(* CODESYS project JCMC40A24BCtrl-V10.project

Project tree, tasks and I/O mapping:
  Device : JCMC 40A, JiaCheng Technology, version 3.5.4.0
    application Application
      libraries: Standard, * (System); SysFile, 3.5.5.0 (System); Util, 3.5.1.0 (System); JCMC_Ctrl, 3.5.5.160 (JiaCheng Technology); CmpJCPBasicLib, 2.1.1 (JiaCheng Technology)
      task MainTask (cyclic, interval t#10ms, priority 6) calls initCan, INIT_JCMC_Ctrl_EXT, INIT_JCMC_Ctrl, PLC_PRG
      task CAN (cyclic, interval t#10ms, priority 7) calls transmit2EngineECM
      program PLC_PRG [ST]
      global variables GVL
      global variables GVL_RETAIN
      program INIT_JCMC_Ctrl [FBD]
      data type RetainFileST
      program INIT_JCMC_Ctrl_EXT [FBD]
      data type Input24BST
      data type Input40AST
      data type Output40AST
      program handleInput24B [ST]
      program handleInput40A [ST]
      data type FaultST
      program faultHandle [ST]
      data type Output24BST
      data type SystemStatusST
      data type SystemConfigureST
      program functionTest [ST]
      program resetTestST [ST]
      data type DspSystemST
      data type DspTestST
      data type CtlTestST
      program chooseWorkMode [ST]
      program panelControl [ST]
      program workflowCore [ST]
      program workflowOther [ST]: ACT, Step0_ACT_active, Step1_ACT_active, Step2_ACT_active, Step3_ACT_active, Step4_ACT_active, Step5_ACT_active
      program engineControl [ST]
      data type TipsST
      program handleOutput40A [ST]
      program handleOutput24B [ST]
      program initCan [ST]
      program receiveFromHMI [ST]
      program receiveFromEngineECM [ST]
      program receiveFromECU [ST]
      program receiveFromVoiceAlarm [ST]
      program receiveFromSiliconePanel [ST]
      data type PanelST
      data type MultipacketParameter
      program transmit2HMI [ST]
      program transmit2SiliconePanel [ST]
      program transmit2EngineECM [ST]
      program parameterConfigure [ST]
      program tipsHandle [ST]
    IoDrvJCMC40A : IoDrvJCMC40A-24B, JiaCheng Technology, version 11.22.33.158
        unmapped channels: AIN_IX0, FIN_IX1, PWM_IX2, PWM_IX3, PWMi_IX4, IX5, %IW3 AI1, %IW4 AI2, AI3, AI4, AI5, AI6, AI7, AI8, FI1, FI2, FI3, FI4, FI5, FI6, FI7, FI8, PWM3i_Cur1, PWM3i_Cur2, PWM3i_Cur3, PWM3i_Cur4, PWM8i_Cur1, PWM8i_Cur2, PWM8i_Cur3, PWM8i_Cur4, PWM_QX0, PWM_QX1, PWMi_QX2, QX3, IX0, %IB73 PWM_IX1, PWM_IX2, IX3, AI1, AI2,
          AI3, AI4, FI1, FI2, FI3, FI4, PWM3i_Cur1, PWM3i_Cur2, PWM3i_Cur3, PWM3i_Cur4, PWM3i_Cur5, PWM3i_Cur6, PWM8i_Cur1, PWM8i_Cur2, PWM_QX0, PWMi_QX1, 5V_QX2
  text list GlobalTextList
  5ce3da45-db07-42e7-a21c-a00fff4ed8f6|C:\Users\guest1\Pictures\e84f1261c6d4c0a418f2bf4200fd030d.jpg
  5ce3da45-db07-42e7-a21c-a00fff4ed8f6|C:\Users\guest1\Pictures\aaa.bmp
  5ce3da45-db07-42e7-a21c-a00fff4ed8f6|C:\Users\guest1\Pictures\320x240.bmp
  5ce3da45-db07-42e7-a21c-a00fff4ed8f6|visu\navigationspanel320x160.jpg
  5ce3da45-db07-42e7-a21c-a00fff4ed8f6|visu\navigationspanel320x160.bmp
  image pool ImagePool
*)

// Device/Application/RetainFileST
TYPE RetainFileST :(*RetanFile区域总大小 3072byte,实际可用大小3071byte,另外1byte由RTS使用*)
STRUCT
	dataB:BYTE;
	dataW:WORD;
	dataD:DWORD;
	dataArray:ARRAY[0..3064] OF BYTE;
END_STRUCT
END_TYPE

// Device/Application/Input24BST
TYPE Input24BST :
STRUCT
	returnOilFilterBlockUp: BOOL; //回油过滤堵塞
	highPressureFilterBlockUp: BOOL;  //高压油滤堵塞
	reverseCar: BOOL; //倒车
	coolingTankWaterLevel: WORD; //冷却水箱液位
	waitingStartLamp: BOOL; //等待启动灯
	alarmLamp: BOOL; //警告故障灯
	stopEngineLamp: BOOL; //停机故障灯
	generatorWork: BOOL; //发电机发电
END_STRUCT
END_TYPE

// Device/Application/Input40AST
 TYPE Input40AST :
    STRUCT 
	   dumpsterPressure: WORD;  //垃圾箱负压
	   suctionBucketPressure: WORD; //吸桶负压
	   frontWaterTankPressure: WORD; //前水箱水压
	   backWaterTankPressure: WORD; //后水箱水压
	   diaphragmPumpPressure: BOOL; //隔膜泵压力正常
	   hydraulicOilLevel: BOOL; //液压油位低
	   frontWaterTankWaterLevel: WORD; //前水箱低水位
	   backWaterTankWaterLevel: WORD; //后清水箱水位
	   backup01: BOOL; //备用
	   bilgeTankWaterLevel: BOOL; //污水箱高水位
	   mainWateraValve: BOOL; //总水阀接近开关
	   cleanValve: BOOL; //吹净阀接近开关
	   backDoor: BOOL;  //后门接近开关
	   leftRod: BOOL; //左侧撑杆接近开关
	   rightRod: BOOL; //右侧撑杆接近开关
	   waterUnloadValve: BOOL; //水路卸荷阀接近开关
    END_STRUCT
  END_TYPE

// Device/Application/Output40AST
TYPE Output40AST :
STRUCT
	connectWaterValve:BOOL; //连通水阀关闭
	closeFrontTank:BOOL; //前水箱关闭
	cLoseBackTank:BOOL; //后水箱关闭
	engineStart:BOOL; //发动机启动
	diaphragmPumpStart:BOOL; //喷雾降尘泵启动
	backup01: BOOL; //备用
	engineStop:BOOL; //发动机停止
	sweeperLowSpeed:BOOL; //扫盘低速
	sweeperMiddleSpeed:BOOL; //扫盘中速
	oilUnloadValve:BOOL; //油路卸荷阀
	leftAllSweep:BOOL; //左/全扫
	rightSweep:BOOL; //右扫
	rightAllSweep:BOOL; //右/全扫
	tankDown:BOOL; //箱体降
	tankUp:BOOL; //箱体升
	suctionNozzleUp:BOOL; //吸嘴升
	leftBackSprinkle:BOOL; //左后洒
	rightBackSprinkle:BOOL; //右后洒
	tankDoorOpen:BOOL; //箱门开
	waterPumpConnect :BOOL; //水泵啮合
	leftFrontSprinkle:BOOL; //左前冲
	rightFrontSprinkle:BOOL; //右前冲
	suctionNozzleDown:BOOL; //吸嘴降
	tankDoorClose:BOOL; //箱门关
END_STRUCT
END_TYPE
(*
VAR_OUTPUT
	//wselfSprayRodOpen: BIT;
	//leftSweeperUp: BIT;
	//rightSprayRodSwingOut: BIT;
END_VAR
*)

// Device/Application/FaultST
TYPE FaultST :
STRUCT
	alarmLamp:BOOL; //发动机警告故障
    stopEngineLamp:BOOL;   //发动机停机故障
	coolingTankWaterLevelLow:BOOL;	//冷却水箱液位低
	waterUnloadValveNotClose:BOOL;	//水路卸荷阀未关闭
	waterUnloadValveNotOpen:BOOL;	//水路卸荷阀未打开
	bilgeTankFull:BOOL;	//污水满
	returnOilFilterBlockUp:BOOL;	//回油过滤堵塞
	hHighPressureFilterBlockUp:BOOL;	//高压油滤堵塞
	hydraulicOilLevelLow:BOOL;	//液压油位低
	frontTankWaterLevelLow:BOOL;	//前水箱缺水
	backTankWaterLevelLow:BOOL;	//后水箱缺水
	tankWaterLevelLow:BOOL;	//水箱缺水
	reverseCarStop:BOOL;	//倒车故障停机
	waterFullStop:BOOL;	//污水满故障停机
	highPressurePumpOverSpeedAlarm:BOOL;	//高压水泵超速报警
	highPressurePumpOverSpeedStop:BOOL;	//高压水泵超速停止
	diaphragmPumpPressure:BOOL;	//喷雾降尘泵故障
END_STRUCT
END_TYPE

// Device/Application/Output24BST
TYPE Output24BST :
STRUCT
	waterUnloadValveOpen :BOOL; //卸荷球阀打开
	auxiliaryValveOpen :BOOL; //辅助球阀喷水
	leftSprayRodOpen :BOOL; //左侧喷杆喷水
	selfSprayRodOpen  :BOOL; //自洁喷杆喷水
	rightSprayRodOpen  :BOOL; //右侧喷杆喷水
	centreSprayRodOpen  :BOOL; //中喷杆喷水
	engineDisconect  :BOOL;  //副发分离
	backupEngineStart  :BOOL; //备用动力
	rightSweeperDown :BOOL; //右扫降
	rightSweeperUp  :BOOL; //右扫升
	leftSweeperSwingOut :BOOL; //左扫摆出
	rightSweeperSwingOut :BOOL; //右扫摆出
	leftSprayRodSwingOut:BOOL; //左侧喷杆摆出
	rightSprayRodSwingOut :BOOL; //右侧喷杆摆出
	leftSweeperDown :BOOL; //左扫盘降
	leftSweeperUp :BOOL;  //左扫盘升
END_STRUCT
END_TYPE

// Device/Application/SystemStatusST
TYPE SystemStatusST :
STRUCT
     softVersion:WORD;//软件版本	

	systemWork:BOOL;//系统工作状态
	systemEndurance:WORD;//续航时间
	engineWork:BOOL;//发动机工作状态
	systemTest:BOOL; //系统测试状态
	backupMotorOpen:BOOL;//备用动力状态
	

	
	vehicleSpeed:WORD;//车速
	vehicleEngineSpeed:WORD;//底盘发动机转速
	distance:DWORD; //车辆行程里程
	
	keyRunPosition:BOOL; //钥匙运行档标志
	engineStart:BOOL; //发动机启动标志
	standardSpeed:BOOL;	//标准速度标志
    strongSpeed:BOOL;	//强力速度标志
    engineSetSpeed:WORD; //副发动机给定转速
	engineRealSpeed:WORD;//发动机实际转速
	engineDisconect:BOOL;//副发动机分离	
	engineCoolingTemperature:SINT;//副发水温
	engineOilPressure:BYTE;//副发油压
	engineWorkTime:DWORD;//发动机工作小时
	engineFaultSPN:DWORD; //副发当前故障SPN

	waterPumpConnect:BOOL; //高压水泵啮合标志
	
	allWashSweep:BOOL;	//全洗扫状态
	leftWashSweep:BOOL;	//左洗扫状态
	rightWashSweep:BOOL;	//右洗扫状态
	allSweep:BOOL;	//全扫路状态
	leftSweep:BOOL;	//左扫路状态
	rightSweep:BOOL;	//右扫路状态
	allWash:BOOL;	//全清洗状态
	leftWash:BOOL;	//左清洗状态
	rightWash:BOOL;	//右清洗状态
	stopWash:BOOL;	//停扫状态
	
	leftSweeperRotate:BOOL;//左扫旋转标志
	rightSweeperRotate:BOOL;//右扫旋转标志
	allSweeperRotate:BOOL;//全扫旋转标志
	leftSweeperSwingOut:BOOL;//左扫盘摆出标志
	leftSweeperDown:BOOL;//左扫盘下放标志
	rightSweeperSwingOut:BOOL;//右扫盘摆出标志
	rightSweeperDown:BOOL;//右扫盘下放标志
	suctionNozzleDown:BOOL;//吸嘴下降标志
	leftSweeperUp:BOOL;//左扫盘上升标志
	rightSweeperUp:BOOL;//右扫盘上升标志
	suctionNozzleUp:BOOL;//吸嘴上升标志
	
	auxiliaryValveOpen1:BOOL; //辅助球阀喷水标志1
	auxiliaryValveOpen2:BOOL; //辅助球阀喷水标志2
	leftSprayRodOpen1:BOOL; //左侧喷杆喷水标志1
	leftSprayRodOpen2:BOOL; //左侧喷杆喷水标志2
	selfSprayRodOpen1:BOOL; //自洁喷杆喷水标志1
	selfSprayRodOpen2:BOOL; //自洁喷杆喷水标志2
	rightSprayRodOpen1 :BOOL; //右侧喷杆喷水标志1
	rightSprayRodOpen2 :BOOL; //右侧喷杆喷水标志2
	centreSprayRodOpen1 :BOOL; //中喷杆喷水标志1
	centreSprayRodOpen2 :BOOL; //中喷杆喷水标志2
	
	leftSprayRodSwingOut :BOOL; //左侧喷杆摆出标志
	rightSprayRodSwingOut :BOOL; //右侧喷杆摆出标志
    //diaphragmPumpStart:BOOL;  //喷雾降尘泵启动标志
	
	leftFlushOpen:BOOL;	//左角冲打开标志
    rightFlushOpen:BOOL;	//右角冲打开标志
    backSprayOpen:BOOL;	//后喷雾打开标志
    sprayGun:BOOL;	//手持喷枪打开标志
	selfClean:BOOL;	//	自洁打开标志
	
    leftFrontSprinkle:BOOL;	//	左前冲打开标志
	rightFrontSprinkle:BOOL;	//	右前冲打开标志
	leftBackSprinkle:BOOL;	//	左后洒打开标志
	rightBackSprinkle:BOOL;	//	右后洒打开标志
	
	tankDoorClose:BOOL;	//垃圾箱门关标志
	tankDoorOpen:BOOL;	//垃圾箱门开标志
	tankDown:BOOL;	//垃圾箱体降标志
	tankUp:BOOL;	//垃圾箱体升标志
	sweeperSpeedLow:BOOL;	//扫盘低速标志
	sweeperSpeedMiddle:BOOL;	//扫盘中速标志
	sweeperSpeedHigh:BOOL;	//扫盘高速标志
	
	manualDrainOff:BOOL; 	//手动排水标志
	autoDrainOff:BOOL; //自动排水标志
	drainOffStart:BOOL;	//排水启动标志,目前该状态属于未启用状态
	replaceSweeper:BOOL;	//更换扫刷标志
	workLamp:BOOL;//工作灯标志
	diaphragmPump:BOOL;//隔膜泵标志
	
	AIModel:BOOL;	//智能模式标志
	CleanRoad:BOOL;	//清洁路面标志
	NormalRoad:BOOL;	//一般路面标志
	DirtyRoad:BOOL;	//污染路面标志
	
	
END_STRUCT
END_TYPE

// Device/Application/SystemConfigureST
TYPE SystemConfigureST :
STRUCT
	
	configFlag:BOOL;            //配置初始化标志
	//dspDiaphragmPump:BOOL;	//喷雾降尘泵_配置_屏输入
	dspLowPressureSystem:BOOL;	//低压水路系统_配置_屏输入
   	dspEngineStandardSpeed:WORD;	//标准速度_配置_屏输入
    dspEngineStrongSpeed:WORD;	//强力速度_配置_屏输入
    dspIncreaseStep:WORD;	//加减转速_配置_屏输入
	dspWaterPumpOverSpeedAlarm:WORD;	//高压水泵超速警报_配置_屏输入
	dspWaterPumpOverSpeedStop:WORD; 	//高压水泵超速停机_配置_屏输入
	dspEngineIdlingSpeed:WORD;	//发动机怠速_配置_屏输入
    dspSweeperSpeed:WORD; //扫盘转速_配置_屏输入
    dspAIModel:BOOL;	//智能模式_配置_屏输入
    dspRoadCondition:WORD;	//路面情况_配置_屏输入
    dspEngineMaxSpeed:WORD;	//发动机最高速_配置_屏输入
	dspWaterPumpConnect:BOOL; //水泵离合器_配置_屏输入

END_STRUCT
END_TYPE

// Device/Application/DspSystemST
TYPE DspSystemST :
STRUCT
	dspAllWashSweep:BOOL;	//全洗扫_屏输入
	dspLeftWashSweep:BOOL;	//左洗扫_屏输入
	dspRightWashSweep:BOOL;	//右洗扫_屏输入
	dspAllSweep:BOOL;	//全扫路_屏输入
	dspLeftSweep:BOOL;	//左扫路_屏输入
	dspRightSweep:BOOL;	//右扫路_屏输入
	dspAllWash:BOOL;	//全清洗_屏输入
	dspLeftWash:BOOL;	//左清洗_屏输入
	dspRightWash:BOOL;	//右清洗_屏输入
	dspStopWash:BOOL;	//停扫_屏输入
	
	dspEngineStart:BOOL;	//发动机启动_屏输入
	dspEngineStop:BOOL;	//发动机停止/运行_屏输入
	
	dspSpeedUp:BOOL;	//转速增加_屏输入
	dspSpeedDown:BOOL;	//转速降低_屏输入
	dspStandardSpeed:BOOL;	//标准速度_屏输入
	dspStrongSpeed:BOOL;	//强力速度_屏输入
	dspAIModel:BOOL;	//智能模式_屏输入
	dspCleanRoad:BOOL;	//清洁路面_屏输入
	dspNormalRoad:BOOL;	//一般路面_屏输入
	dspDirtyRoad:BOOL;	//污染路面_屏输入
	
	dspTankDoorClose:BOOL;	//垃圾箱门关_屏输入
	dspTankDoorOpen:BOOL;	//垃圾箱门开_屏输入
	dspTankDown:BOOL;	//垃圾箱体降_屏输入
	dspTankUp:BOOL;	//垃圾箱体升_屏输入
	dspSweeperSpeedLow:BOOL;	//扫盘低速_屏输入
	dspSweeperSpeedMiddle:BOOL;	//扫盘中速_屏输入
	dspSweeperSpeedHigh:BOOL;	//扫盘高速_屏输入
	
	dspWaterPumpDisconnect:BOOL;//水泵离合器_屏输入
	dspLeftFlush:BOOL;	//左角冲_屏输入
	dspRightFlush:BOOL;	//右角冲_屏输入
	dspBackSpray:BOOL;	//后喷雾_屏输入
	dspSprayGun:BOOL;	//手持喷枪_屏输入
	dspSelfClean:BOOL;	//自洁_屏输入
	
	dspLeftFrontSprinkle:BOOL;	//左前冲_屏输入
	dspRightFrontSprinkle:BOOL;	//右前冲_屏输入
	dspLeftBackSprinkle:BOOL;	//左后洒_屏输入
	dspRightBackSprinkle:BOOL;	//右后洒_屏输入
	
	dspManualDrainOff:BOOL; 	//手动排水_屏输入
	dspAutoDrainOff:BOOL; //自动排水_屏输入
	dspDrainOffStart:BOOL;	//排水启动_屏输入,目前该按钮属于未启动状态
	dspLeftSprayRodDrainOff:BOOL;	//左喷杆排水_屏输入
	dspRightSprayRodDrainOff:BOOL;	//右喷杆排水_屏输入
	dspAuxiliarySystemDrainOff:BOOL;	//辅助排水_屏输入
	dspSelfCleanDrainOff:BOOL;	//自洁排水_屏输入
	dspCentreSprayRodDrainOff:BOOL;	//中喷杆排水_屏输入
	dspReplaceSweeper:BOOL;	//更换扫刷_屏输入
	dspWorkLamp:BOOL;//工作灯_屏输入
	dspDiaphragmPump:BOOL;//隔膜泵_屏输入
	
	dspTestStart:BOOL;	//功能测试_屏输入
END_STRUCT
END_TYPE

// Device/Application/DspTestST
TYPE DspTestST :
STRUCT
	dspEngineDisconnectTest:BOOL;	//副发分离_测试_屏输入
	dspConnectWaterValveTest:BOOL;	//连通水阀_测试_屏输入
	dspCloseFrontTankTest:BOOL;	//前水箱水阀_测试_屏输入
	dspCLoseBackTankTest:BOOL;	//后水箱水阀_测试_屏输入
	dspSweeperSpeedLowTest:BOOL;	//扫盘低速_测试_屏输入
	dspSweeperSpeedMiddleTest:BOOL;	//扫盘中速_测试_屏输入
	dspLeftSweeperRotateTest:BOOL;	//左扫旋转_测试_屏输入
	dspRightSweeperRotateTest:BOOL;	//右扫旋转_测试_屏输入
	dspAllSweeperRotateTest:BOOL;	//全扫旋转_测试_屏输入
	dspTankDownTest:BOOL;	//箱体降_测试_屏输入
	dspTankUpTest:BOOL;	//箱体升_测试_屏输入
	dspSuctionNozzleDownTest:BOOL;	//吸嘴降_测试_屏输入
	dspSuctionNozzleUpTest:BOOL;	//吸嘴升_测试_屏输入
	dspTankDoorOpenTest:BOOL; //箱门开_测试_屏输入
	dspTankDoorCloseTest:BOOL;	//箱门关_测试_屏输入
	dspLeftSweeperDownTest:BOOL;	//左扫盘下放_测试_屏输入
	dspLeftSweeperUpTest:BOOL;	//左扫盘回收_测试_屏输入
	dspRightSweeperDownTest:BOOL;	//右扫盘下放_测试_屏输入
	dspRightSweeperUpTest:BOOL;	//右扫盘回收_测试_屏输入
	dspLeftSweeperSwingOutTest:BOOL;	//左扫盘摆出_测试_屏输入
	dspRightSweeperSwingOutTest:BOOL;	//右扫盘摆出_测试_屏输入
	dspLeftSprayRodSwingOutTest:BOOL;	//左喷杆摆出_测试_屏输入
	dspRightSprayRodSwingOutTest:BOOL;	//右喷杆摆出_测试_屏输入
	dspLeftSprayRodOpenTest:BOOL;	//左喷杆喷水_测试_屏输入
	dspRightSprayRodOpenTest:BOOL;	//右喷杆喷水_测试_屏输入
	dspCentreSprayRodOpenTest:BOOL;	//中喷杆喷水_测试_屏输入
	dspAuxiliaryValueTest:BOOL;	//辅助球阀打开_测试_屏输入
	dspSelfCleanTest:BOOL;	//自洁打开_测试_屏输入
	dspWaterPumpConnectTest:BOOL;//高压水泵啮合_测试_屏输入
	dspDiaphragmPumpStartTest:BOOL;	//喷雾降尘泵_测试_屏输入
    dspLeftFrontSprinkleTest:BOOL;	//	左前冲_测试_屏输入
	dspRightFrontSprinkleTest:BOOL;	//	右前冲_测试_屏输入
	dspLeftBackSprinkleTest:BOOL;	//	左后洒_测试_屏输入
	dspRightBackSprinkleTest:BOOL;	//	右后洒_测试_屏输入

END_STRUCT
END_TYPE

// Device/Application/CtlTestST
TYPE CtlTestST :
STRUCT
	ctlEngineDisconnectTest:BOOL;	//副发分离_测试_控制器
    ctlConnectWaterValveTest:BOOL;	//连通水阀_测试_控制器
    ctlCloseFrontTankTest:BOOL;	//前水箱水阀_测试_控制器
    ctlCLoseBackTankTest:BOOL;	//后水箱水阀_测试_控制器
    ctlSweeperSpeedLowTest:BOOL;	//扫盘低速_测试_控制器
	ctlSweeperSpeedMiddleTest:BOOL;	//扫盘中速_测试_控制器
	ctlLeftSweeperRotateTest:BOOL;	//左扫旋转_测试_控制器
	ctlRightSweeperRotateTest:BOOL;	//右扫旋转_测试_控制器
	ctlAllSweeperRotateTest:BOOL;	//全扫旋转_测试_控制器
	ctlTankDownTest:BOOL;	//箱体降_测试_控制器
	ctlTankUpTest:BOOL;	//箱体升_测试_控制器
	ctlSuctionNozzleDownTest:BOOL;	//吸嘴降_测试_控制器
	ctlSuctionNozzleUpTest:BOOL;	//吸嘴升_测试_控制器
	ctlTankDoorOpenTest:BOOL;	//箱门开_测试_控制器
	ctlTankDoorCloseTest:BOOL;	//箱门关_测试_控制器
	ctlLeftSweeperDownTest:BOOL;	//左扫盘下放_测试_控制器
	ctlLeftSweeperUpTest:BOOL;	//左扫盘回收_测试_控制器
	ctlRightSweeperDownTest:BOOL;	//右扫盘下放_测试_控制器
	ctlRightSweeperUpTest:BOOL;	//右扫盘回收_测试_控制器
	ctlLeftSweeperSwingOutTest:BOOL;	//左扫盘摆出_测试_控制器
	ctlRightSweeperSwingOutTest:BOOL;	//右扫盘摆出_测试_控制器
	ctlLeftSprayRodSwingOutTest:BOOL;	//左喷杆摆出_测试_控制器
	ctlRightSprayRodSwingOutTest:BOOL;	//右喷杆摆出_测试_控制器
	ctlLeftSprayRodOpenTest:BOOL;	//左喷杆喷水_测试_控制器
	ctlRightSprayRodOpenTest:BOOL;	//右喷杆喷水_测试_控制器
	ctlCentreSprayRodOpenTest:BOOL;	//中喷杆喷水_测试_控制器
	ctlAuxiliaryValueTest:BOOL;	//辅助球阀打开_测试_控制器
	ctlSelfCleanTest:BOOL;	//自洁打开_测试_控制器
	ctlWaterPumpConnectTest:BOOL;	//高压水泵啮合_测试_控制器
	ctlDiaphragmPumpStartTest:BOOL;	//喷雾降尘泵_测试_控制器
	ctlLeftFrontSprinkleTest:BOOL;	//	左前冲_测试_控制器
	ctlRightFrontSprinkleTest:BOOL;	//	右前冲_测试_控制器
	ctlLeftBackSprinkleTest:BOOL;	//	左后洒_测试_控制器
	ctlRightBackSprinkleTest:BOOL;	//	右后洒_测试_控制器
END_STRUCT
END_TYPE

// Device/Application/TipsST
TYPE TipsST :
STRUCT
	closeTest:BOOL;	//请关闭测试
    reverseCar:BOOL;	//正在倒车中
	startEngineFirst:BOOL;	//请先打开发动机
	backupMotorOpen:BOOL;	//备用动力打开
	testOpen:BOOL;	//测试打开
	highPressurePumpDisconnect:BOOL;	//高压水泵未啮合
	tankDoorNotOpen:BOOL; //箱门未打开
	leftRodUp:BOOL;	//左支撑杆未放下
	rightRodUp:BOOL;	//右支撑杆未放下
	mainWateraValveNotOpen:BOOL;	//总水阀未打开
	cleanValveNotClose:BOOL;	//吹净球阀未关闭
    stopEngineFirst:BOOL; //请先关闭发动机
	
	
	//临时变量
	highPressurePumpDisconnect1:BOOL;	//左右全洗扫、清洗按钮，高压水泵未啮合
	highPressurePumpDisconnect2:BOOL;	//硅胶面板喷枪、自洁按钮，高压水泵未啮合
	highPressurePumpDisconnect3:BOOL;	//触摸屏喷枪、自洁、左前冲、右前冲、后喷雾按钮，高压水泵未啮合
	mainWateraValveNotOpen1:BOOL;	//左右全洗扫、清洗按钮，总水阀未打开
	mainWateraValveNotOpen2:BOOL;	//硅胶面板喷枪、自洁按钮，总水阀未打开
	mainWateraValveNotOpen3:BOOL;	//触摸屏喷枪、自洁、左前冲、右前冲、后喷雾按钮，总水阀未打开
	mainWateraValveNotOpen4:BOOL;	//离合器按钮，总水阀未打开
	cleanValveNotClose1:BOOL;	//左右全洗扫、清洗按钮，吹净球阀未关闭
	cleanValveNotClose2:BOOL;	//硅胶面板喷枪、自洁按钮，吹净球阀未关闭
	cleanValveNotClose3:BOOL;	//触摸屏喷枪、自洁、左前冲、右前冲、后喷雾按钮，吹净球阀未关闭
	cleanValveNotClose4:BOOL;	//离合器按钮，吹净球阀未关闭
END_STRUCT
END_TYPE

// Device/Application/PanelST
TYPE PanelST :
STRUCT
	tankDoorClose:BOOL;	//垃圾箱门关_硅胶面板输入
	tankDoorOpen:BOOL;	//垃圾箱门开_硅胶面板输入
	tankDown:BOOL;	//垃圾箱体降_硅胶面板输入
	tankUp:BOOL;	//垃圾箱体升_硅胶面板输入
	leftSweeperOutAndDown:BOOL;	//左扫盘摆出下降_硅胶面板输入
	leftSweeperUpAndIn:BOOL;	//左扫盘上升回收_硅胶面板输入
	rightSweeperOutAndDown:BOOL;	//右扫盘下放_硅胶面板输入
	rightSweeperUpAndIn:BOOL;	//右扫盘回收_硅胶面板输入
	suctionNozzleDown:BOOL;	//吸嘴降_测试_硅胶面板输入
	suctionNozzleUp:BOOL;	//吸嘴升_硅胶面板输入
	selfClean:BOOL;	//自洁打开_硅胶面板输入
	sprayGun:BOOL;	//手持喷枪_硅胶面板输入
	sprayRodOutOrIn:BOOL;  //喷杆伸缩_硅胶面板输入
	backupMotor:BOOL; //备用动力_硅胶面板输入
	workLamp:BOOL; //工作灯_硅胶面板输入
	backlight:BOOL; //背光灯_硅胶面板输入
	
	tankDoorCloseFlag:BOOL;	//垃圾箱门关_硅胶面板_返回标志
	tankDoorOpenFlag:BOOL;	//垃圾箱门开_硅胶面板_返回标志
	tankDownFlag:BOOL;	//垃圾箱体降_硅胶面板_返回标志
	tankUpFlag:BOOL;	//垃圾箱体升_硅胶面板_返回标志
	leftSweeperOutAndDownFlag:BOOL;	//左扫盘下放_硅胶面板_返回标志
	leftSweeperUpAndInFlag:BOOL;	//左扫盘回收_硅胶面板_返回标志
	rightSweeperOutAndDownFlag:BOOL;	//右扫盘下放_硅胶面板_返回标志
	rightSweeperUpAndInFlag:BOOL;	//右扫盘回收_硅胶面板_返回标志
	suctionNozzleDownFlag:BOOL;	//吸嘴降_测试_硅胶面板_返回标志
	suctionNozzleUpFlag:BOOL;	//吸嘴升_硅胶面板_返回标志
	selfCleanFlag:BOOL;	//自洁打开_硅胶面板_返回标志
	sprayGunFlag:BOOL;	//手持喷枪_硅胶面板_返回标志
	sprayRodOutOrInFlag:BOOL;  //喷杆伸缩_硅胶面板_返回标志
	backupMotorFlag:BOOL; //备用动力_硅胶面板_返回标志
	workLampFlag:BOOL; //工作灯_硅胶面板_返回标志
	backlightFlag:BOOL; //背光灯_硅胶面板_返回标志
END_STRUCT
END_TYPE

// Device/Application/MultipacketParameter
TYPE MultipacketParameter :
STRUCT
	packageTotalNum:WORD;//数据包数量，2-255
	byteTotalNum:WORD; //字节数，9-1785
	PGN:DWORD; //参数群编号
	Data: ARRAY[0..79] OF  BYTE; //数据,当packageNum>10，丢弃数据
END_STRUCT
END_TYPE

// Device/Application/GVL
VAR_GLOBAL		

	isOK: BOOL;	
// 40A板卡输入输出端口
    diDumpsterPressure AT %IW3 :WORD;  //垃圾箱负压
	diSuctionBucketPressure AT %IW4 :WORD; //吸桶负压
	diFrontWaterTankPressure AT %IW5 :WORD; //前水箱水压
	diBackWaterTankPressure AT %IW6 :WORD; //后水箱水压
	diDiaphragmPumpPressure AT %IX0.4 :BOOL; //隔膜泵压力正常
	diHydraulicOilLevel AT %IX0.5 :BOOL; //液压油位低
	diFrontWaterTankWaterLevel AT %IW9 :WORD; //前水箱低水位
	diBackWaterTankWaterLevel AT %IW10 :WORD; //后清水箱水位
	diBackup01 AT %IX1.0 :BOOL; //备用
	diBilgeTankWaterLevel AT %IX1.1 :BOOL; //污水箱高水位
	diMainWateraValve AT %IX1.2 :BOOL; //总水阀接近开关
	diCleanValve AT %IX1.3 :BOOL; //吹净阀接近开关
	diBackDoor AT %IX1.4 :BOOL;  //后门接近开关
	diLeftRod AT %IX1.5 :BOOL; //左侧撑杆接近开关
	diRightRod AT %IX1.6 :BOOL; //右侧撑杆接近开关
	diWaterUnloadValve AT %IX1.7 :BOOL; //水路卸荷阀接近开关
	doConnectWaterValve AT %QX0.0 :BOOL; //连通水阀关闭
	doCloseFrontTank AT %QX0.1 :BOOL; //前水箱关闭
	doCLoseBackTank AT %QX0.2 :BOOL; //后水箱关闭
	doEngineStart AT %QX0.3 :BOOL; //发动机启动
	doDiaphragmPumpStart AT %QX0.4 :BOOL; //隔膜泵启动
	doBackup01 AT %QX0.5 : BOOL; //备用
	doEngineStop AT %QX0.6 :BOOL; //发动机停止
	doSweeperLowSpeed AT %QX0.7 :BOOL; //扫盘低速
	doSweeperMiddleSpeed AT %QX1.0 :BOOL; //扫盘中速
	doOilUnloadValve AT %QX1.1 :BOOL; //油路卸荷阀
	doLeftAllSweep AT %QX1.2 :BOOL; //左/全扫
	doRightSweep AT %QX1.3 :BOOL; //右扫
	doRightAllSweep AT %QX1.4 :BOOL; //右/全扫
	doTankDown AT %QX1.5 :BOOL; //箱体降
	doTankUp AT %QX1.6 :BOOL; //箱体升
	doSuctionNozzleUp AT %QX1.7 :BOOL; //吸嘴升
	doLeftBackSprinkle AT %QX2.0 :BOOL; //左后洒
	doRightBackSprinkle AT %QX2.1 :BOOL; //右后洒
	doTankDoorOpen AT %QX2.2 :BOOL; //箱门开
	doWaterPumpConnect AT %QX2.3 :BOOL; //水泵啮合
	doLeftFrontSprinkle AT %QX2.4 :BOOL; //左前冲
	doRightFrontSprinkle AT %QX2.5 :BOOL; //右前冲
	doSuctionNozzleDown AT %QX2.6 :BOOL; //吸嘴降
	doTankDoorClose AT %QX2.7 :BOOL; //箱门关
	
//24B板块输入输出端口	
    diReturnOilFilterBlockUp AT %IX72.0 :BOOL; //回油过滤堵塞
	diHighPressureFilterBlockUp AT %IX72.1 :BOOL;  //高压油滤堵塞
	diReverseCar AT %IX72.2 :BOOL; //倒车
	diCoolingTankWaterLevel AT %ID22 :WORD; //冷却水箱液位
	diWaitingStartLamp AT %IX72.4 :BOOL; //等待启动灯
	diAlarmLamp AT %IX72.5 :BOOL; //警告故障灯
	diStopEngineLamp AT %IX72.6 :BOOL; //停机故障灯
	diGeneratorWork  AT %IX7.7 :BOOL; //发电机发电
	doWaterUnloadValveOpen AT %QX4.0 :BOOL; //卸荷球阀打开
	doAuxiliaryValveOpen AT %QX4.1 :BOOL; //辅助球阀喷水
	doLeftSprayRodOpen AT %QX4.2 :BOOL; //左侧喷杆喷水
	doSelfSprayRodOpen AT %QX4.3 :BOOL; //自洁喷杆喷水
	doRightSprayRodOpen AT %QX4.4 :BOOL; //右侧喷杆喷水
	doCentreSprayRodOpen AT %QX4.5 :BOOL; //中喷杆喷水
	doEngineDisconect AT %QX4.6 :BOOL;  //副发分离
	doBackupEngineStart AT %QX4.7 :BOOL; //备用动力
	doRightSweeperDown AT %QX5.0 :BOOL; //右扫降
	doRightSweeperUp AT %QX5.1 :BOOL; //右扫升
	doLeftSweeperSwingOut AT %QX5.2 :BOOL; //左扫摆出
	doRightSweeperSwingOut AT %QX5.3 :BOOL; //右扫摆出
	doLeftSprayRodSwingOut AT %QX5.4 :BOOL; //左侧喷杆摆出
	doRightSprayRodSwingOut AT %QX5.5 :BOOL; //右侧喷杆摆出
	doLeftSweeperDown AT %QX5.6 :BOOL; //左扫盘降
	doLeftSweeperUp AT %QX5.7 :BOOL;  //左扫盘升
 
    input40A: Input40AST;//处理后的40A板卡的输入信号  
    input24B: Input24BST;//处理后的40A板卡的输入信号
    output40A: Output40AST; //40A板卡输出信号
    output24B: Output24BST; //24B板卡输出信号
    dspSystemInput:DspSystemST;//车载控制屏系统输入
    dspTestInput:DspTestST; //车载控制屏测试输入
    systemStatus: SystemStatusST;//系统工作状态
    ctlTestFlag:CtlTestST; //控制器测试状态
    faultST: FaultST;  //系统故障
    tipsST:TipsST;     //系统提示
	panelInput:PanelST; //硅胶面板控制信号
END_VAR

// Device/Application/GVL_RETAIN
VAR_GLOBAL RETAIN
	bufRETAIN: DWORD:= 0;
//	bufRETAIN2: BYTE:= 0;
	pbufRetain: POINTER TO DWORD:=ADR(bufretain);
	xx: POINTER TO POINTER TO DWORD:=ADR(pbufRetain);
    systemConfig:SystemConfigureST; //系统配置

END_VAR

// Device/Application/initCan
PROGRAM initCan
VAR
	initCAN: JCMC_Ctrl.CAN;
	initCAN_EXT: JCMC_Ctrl.CAN_EXT;
END_VAR

IF JCMC_Ctrl.INIT THEN   //可以不用，调试再试验
	initCAN(CHANNEL:=1,ENABLE:=TRUE,START:=TRUE,EXTENDED_MODE:=TRUE,BAUDRATE:=250);//40A,CAN1初始化，波特率250KB，扩展帧
	initCAN(CHANNEL:=2,ENABLE:=TRUE,START:=TRUE,EXTENDED_MODE:=TRUE,BAUDRATE:=250);//40A,CAN2初始化，波特率250KB，扩展帧

	initCAN_EXT(CHANNEL:=1,ENABLE:=TRUE,START:=TRUE,EXTENDED_MODE:=TRUE,BAUDRATE:=250);//24B,CAN1初始化，波特率250KB，扩展帧,发送频率不要低于20ms
	initCAN_EXT(CHANNEL:=2,ENABLE:=TRUE,START:=TRUE,EXTENDED_MODE:=TRUE,BAUDRATE:=250);//24B,CAN2初始化，波特率250KB，扩展帧,送频率不要低于20ms
END_IF

END_PROGRAM

// Device/Application/INIT_JCMC_Ctrl_EXT
PROGRAM INIT_JCMC_Ctrl_EXT
VAR
	JCMC_Ctrl_EXT_INIT_0: JCMC_Ctrl.JCMC_Ctrl_INIT_EXT;
	isOK:BOOL:=FALSE;
END_VAR

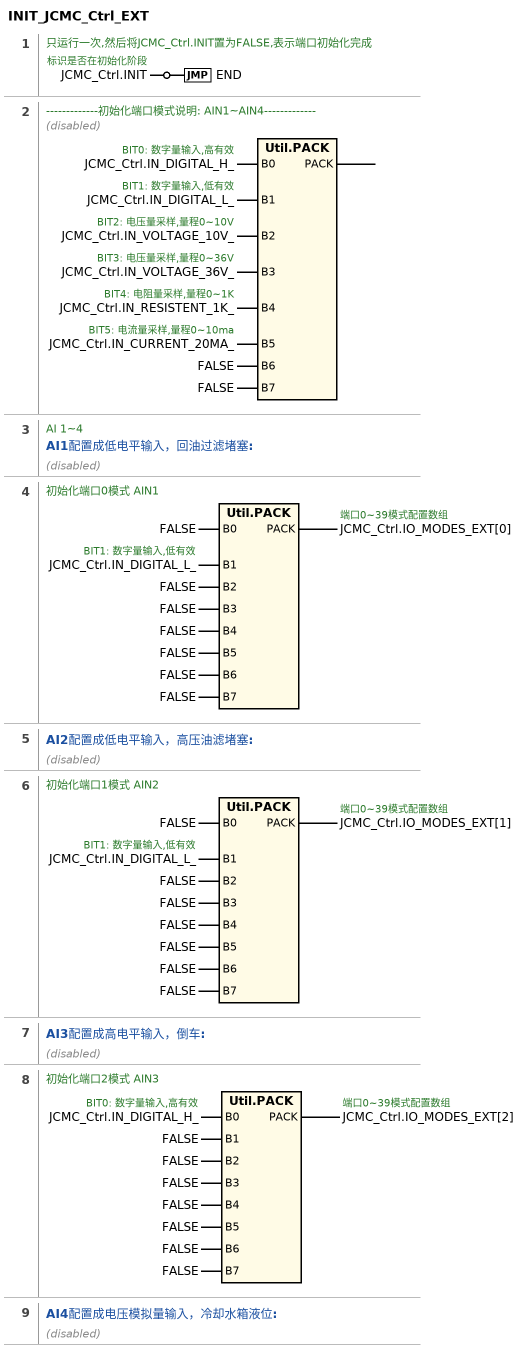
// NETWORK 1
// 只运行一次,然后将JCMC_Ctrl.INIT置为FALSE,表示端口初始化完成
//   JCMC_Ctrl.INIT: 标识是否在初始化阶段
IF NOT JCMC_Ctrl.INIT THEN JMP END; END_IF

// NETWORK 2 (disabled)
// -------------初始化端口模式说明: AIN1~AIN4-------------
//   JCMC_Ctrl.IN_DIGITAL_H_: BIT0: 数字量输入,高有效
//   JCMC_Ctrl.IN_DIGITAL_L_: BIT1: 数字量输入,低有效
//   JCMC_Ctrl.IN_VOLTAGE_10V_: BIT2: 电压量采样,量程0~10V
//   JCMC_Ctrl.IN_VOLTAGE_36V_: BIT3: 电压量采样,量程0~36V
//   JCMC_Ctrl.IN_RESISTENT_1K_: BIT4: 电阻量采样,量程0~1K
//   JCMC_Ctrl.IN_CURRENT_20MA_: BIT5: 电流量采样,量程0~10ma
// ??? := Util.PACK(B0 := JCMC_Ctrl.IN_DIGITAL_H_, B1 := JCMC_Ctrl.IN_DIGITAL_L_, B2 := JCMC_Ctrl.IN_VOLTAGE_10V_, B3 := JCMC_Ctrl.IN_VOLTAGE_36V_, B4 := JCMC_Ctrl.IN_RESISTENT_1K_, B5 := JCMC_Ctrl.IN_CURRENT_20MA_, B6 := FALSE, B7 := FALSE);

// NETWORK 3 (disabled)
// AI 1~4
// label: AI1配置成低电平输入，回油过滤堵塞

// NETWORK 4
// 初始化端口0模式 AIN1
//   JCMC_Ctrl.IN_DIGITAL_L_: BIT1: 数字量输入,低有效
//   JCMC_Ctrl.IO_MODES_EXT[0]: 端口0~39模式配置数组
JCMC_Ctrl.IO_MODES_EXT[0] := Util.PACK(B0 := FALSE, B1 := JCMC_Ctrl.IN_DIGITAL_L_, B2 := FALSE, B3 := FALSE, B4 := FALSE, B5 := FALSE, B6 := FALSE, B7 := FALSE);

// NETWORK 5 (disabled)
// label: AI2配置成低电平输入，高压油滤堵塞

// NETWORK 6
// 初始化端口1模式 AIN2
//   JCMC_Ctrl.IN_DIGITAL_L_: BIT1: 数字量输入,低有效
//   JCMC_Ctrl.IO_MODES_EXT[1]: 端口0~39模式配置数组
JCMC_Ctrl.IO_MODES_EXT[1] := Util.PACK(B0 := FALSE, B1 := JCMC_Ctrl.IN_DIGITAL_L_, B2 := FALSE, B3 := FALSE, B4 := FALSE, B5 := FALSE, B6 := FALSE, B7 := FALSE);

// NETWORK 7 (disabled)
// label: AI3配置成高电平输入，倒车

// NETWORK 8
// 初始化端口2模式 AIN3
//   JCMC_Ctrl.IN_DIGITAL_H_: BIT0: 数字量输入,高有效
//   JCMC_Ctrl.IO_MODES_EXT[2]: 端口0~39模式配置数组
JCMC_Ctrl.IO_MODES_EXT[2] := Util.PACK(B0 := JCMC_Ctrl.IN_DIGITAL_H_, B1 := FALSE, B2 := FALSE, B3 := FALSE, B4 := FALSE, B5 := FALSE, B6 := FALSE, B7 := FALSE);

// NETWORK 9 (disabled)
// label: AI4配置成电压模拟量输入，冷却水箱液位

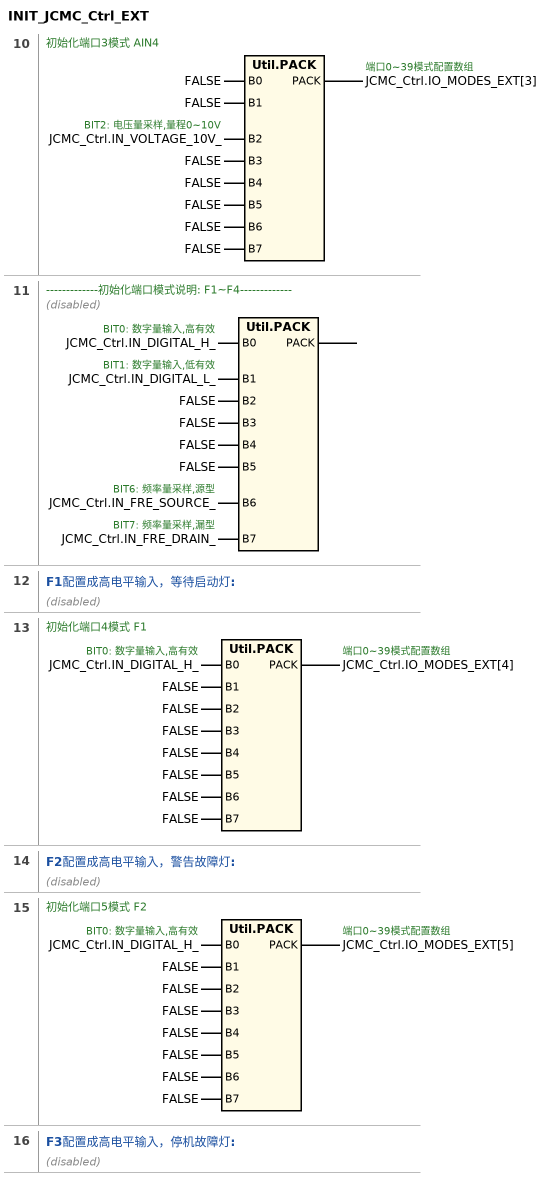
// NETWORK 10
// 初始化端口3模式 AIN4
//   JCMC_Ctrl.IN_VOLTAGE_10V_: BIT2: 电压量采样,量程0~10V
//   JCMC_Ctrl.IO_MODES_EXT[3]: 端口0~39模式配置数组
JCMC_Ctrl.IO_MODES_EXT[3] := Util.PACK(B0 := FALSE, B1 := FALSE, B2 := JCMC_Ctrl.IN_VOLTAGE_10V_, B3 := FALSE, B4 := FALSE, B5 := FALSE, B6 := FALSE, B7 := FALSE);

// NETWORK 11 (disabled)
// -------------初始化端口模式说明: F1~F4-------------
//   JCMC_Ctrl.IN_DIGITAL_H_: BIT0: 数字量输入,高有效
//   JCMC_Ctrl.IN_DIGITAL_L_: BIT1: 数字量输入,低有效
//   JCMC_Ctrl.IN_FRE_SOURCE_: BIT6: 频率量采样,源型
//   JCMC_Ctrl.IN_FRE_DRAIN_: BIT7: 频率量采样,漏型
// ??? := Util.PACK(B0 := JCMC_Ctrl.IN_DIGITAL_H_, B1 := JCMC_Ctrl.IN_DIGITAL_L_, B2 := FALSE, B3 := FALSE, B4 := FALSE, B5 := FALSE, B6 := JCMC_Ctrl.IN_FRE_SOURCE_, B7 := JCMC_Ctrl.IN_FRE_DRAIN_);

// NETWORK 12 (disabled)
// label: F1配置成高电平输入，等待启动灯

// NETWORK 13
// 初始化端口4模式 F1
//   JCMC_Ctrl.IN_DIGITAL_H_: BIT0: 数字量输入,高有效
//   JCMC_Ctrl.IO_MODES_EXT[4]: 端口0~39模式配置数组
JCMC_Ctrl.IO_MODES_EXT[4] := Util.PACK(B0 := JCMC_Ctrl.IN_DIGITAL_H_, B1 := FALSE, B2 := FALSE, B3 := FALSE, B4 := FALSE, B5 := FALSE, B6 := FALSE, B7 := FALSE);

// NETWORK 14 (disabled)
// label: F2配置成高电平输入，警告故障灯

// NETWORK 15
// 初始化端口5模式 F2
//   JCMC_Ctrl.IN_DIGITAL_H_: BIT0: 数字量输入,高有效
//   JCMC_Ctrl.IO_MODES_EXT[5]: 端口0~39模式配置数组
JCMC_Ctrl.IO_MODES_EXT[5] := Util.PACK(B0 := JCMC_Ctrl.IN_DIGITAL_H_, B1 := FALSE, B2 := FALSE, B3 := FALSE, B4 := FALSE, B5 := FALSE, B6 := FALSE, B7 := FALSE);

// NETWORK 16 (disabled)
// label: F3配置成高电平输入，停机故障灯

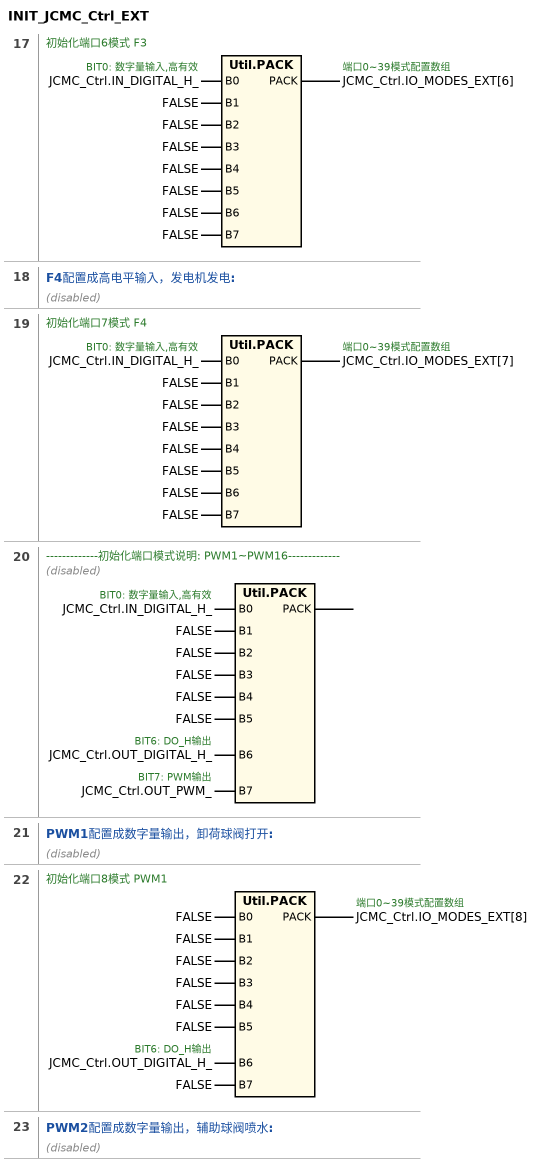
// NETWORK 17
// 初始化端口6模式 F3
//   JCMC_Ctrl.IN_DIGITAL_H_: BIT0: 数字量输入,高有效
//   JCMC_Ctrl.IO_MODES_EXT[6]: 端口0~39模式配置数组
JCMC_Ctrl.IO_MODES_EXT[6] := Util.PACK(B0 := JCMC_Ctrl.IN_DIGITAL_H_, B1 := FALSE, B2 := FALSE, B3 := FALSE, B4 := FALSE, B5 := FALSE, B6 := FALSE, B7 := FALSE);

// NETWORK 18 (disabled)
// label: F4配置成高电平输入，发电机发电

// NETWORK 19
// 初始化端口7模式 F4
//   JCMC_Ctrl.IN_DIGITAL_H_: BIT0: 数字量输入,高有效
//   JCMC_Ctrl.IO_MODES_EXT[7]: 端口0~39模式配置数组
JCMC_Ctrl.IO_MODES_EXT[7] := Util.PACK(B0 := JCMC_Ctrl.IN_DIGITAL_H_, B1 := FALSE, B2 := FALSE, B3 := FALSE, B4 := FALSE, B5 := FALSE, B6 := FALSE, B7 := FALSE);

// NETWORK 20 (disabled)
// -------------初始化端口模式说明: PWM1~PWM16-------------
//   JCMC_Ctrl.IN_DIGITAL_H_: BIT0: 数字量输入,高有效
//   JCMC_Ctrl.OUT_DIGITAL_H_: BIT6: DO_H输出
//   JCMC_Ctrl.OUT_PWM_: BIT7: PWM输出
// ??? := Util.PACK(B0 := JCMC_Ctrl.IN_DIGITAL_H_, B1 := FALSE, B2 := FALSE, B3 := FALSE, B4 := FALSE, B5 := FALSE, B6 := JCMC_Ctrl.OUT_DIGITAL_H_, B7 := JCMC_Ctrl.OUT_PWM_);

// NETWORK 21 (disabled)
// label: PWM1配置成数字量输出，卸荷球阀打开

// NETWORK 22
// 初始化端口8模式 PWM1
//   JCMC_Ctrl.OUT_DIGITAL_H_: BIT6: DO_H输出
//   JCMC_Ctrl.IO_MODES_EXT[8]: 端口0~39模式配置数组
JCMC_Ctrl.IO_MODES_EXT[8] := Util.PACK(B0 := FALSE, B1 := FALSE, B2 := FALSE, B3 := FALSE, B4 := FALSE, B5 := FALSE, B6 := JCMC_Ctrl.OUT_DIGITAL_H_, B7 := FALSE);

// NETWORK 23 (disabled)
// label: PWM2配置成数字量输出，辅助球阀喷水

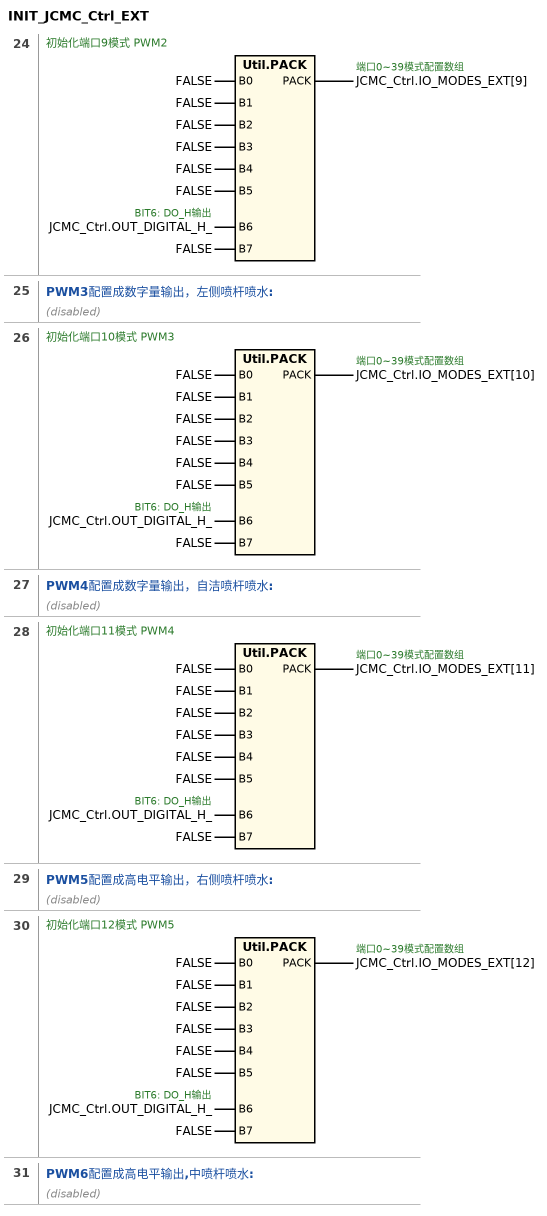
// NETWORK 24
// 初始化端口9模式 PWM2
//   JCMC_Ctrl.OUT_DIGITAL_H_: BIT6: DO_H输出
//   JCMC_Ctrl.IO_MODES_EXT[9]: 端口0~39模式配置数组
JCMC_Ctrl.IO_MODES_EXT[9] := Util.PACK(B0 := FALSE, B1 := FALSE, B2 := FALSE, B3 := FALSE, B4 := FALSE, B5 := FALSE, B6 := JCMC_Ctrl.OUT_DIGITAL_H_, B7 := FALSE);

// NETWORK 25 (disabled)
// label: PWM3配置成数字量输出，左侧喷杆喷水

// NETWORK 26
// 初始化端口10模式 PWM3
//   JCMC_Ctrl.OUT_DIGITAL_H_: BIT6: DO_H输出
//   JCMC_Ctrl.IO_MODES_EXT[10]: 端口0~39模式配置数组
JCMC_Ctrl.IO_MODES_EXT[10] := Util.PACK(B0 := FALSE, B1 := FALSE, B2 := FALSE, B3 := FALSE, B4 := FALSE, B5 := FALSE, B6 := JCMC_Ctrl.OUT_DIGITAL_H_, B7 := FALSE);

// NETWORK 27 (disabled)
// label: PWM4配置成数字量输出，自洁喷杆喷水

// NETWORK 28
// 初始化端口11模式 PWM4
//   JCMC_Ctrl.OUT_DIGITAL_H_: BIT6: DO_H输出
//   JCMC_Ctrl.IO_MODES_EXT[11]: 端口0~39模式配置数组
JCMC_Ctrl.IO_MODES_EXT[11] := Util.PACK(B0 := FALSE, B1 := FALSE, B2 := FALSE, B3 := FALSE, B4 := FALSE, B5 := FALSE, B6 := JCMC_Ctrl.OUT_DIGITAL_H_, B7 := FALSE);

// NETWORK 29 (disabled)
// label: PWM5配置成高电平输出，右侧喷杆喷水

// NETWORK 30
// 初始化端口12模式 PWM5
//   JCMC_Ctrl.OUT_DIGITAL_H_: BIT6: DO_H输出
//   JCMC_Ctrl.IO_MODES_EXT[12]: 端口0~39模式配置数组
JCMC_Ctrl.IO_MODES_EXT[12] := Util.PACK(B0 := FALSE, B1 := FALSE, B2 := FALSE, B3 := FALSE, B4 := FALSE, B5 := FALSE, B6 := JCMC_Ctrl.OUT_DIGITAL_H_, B7 := FALSE);

// NETWORK 31 (disabled)
// label: PWM6配置成高电平输出,中喷杆喷水

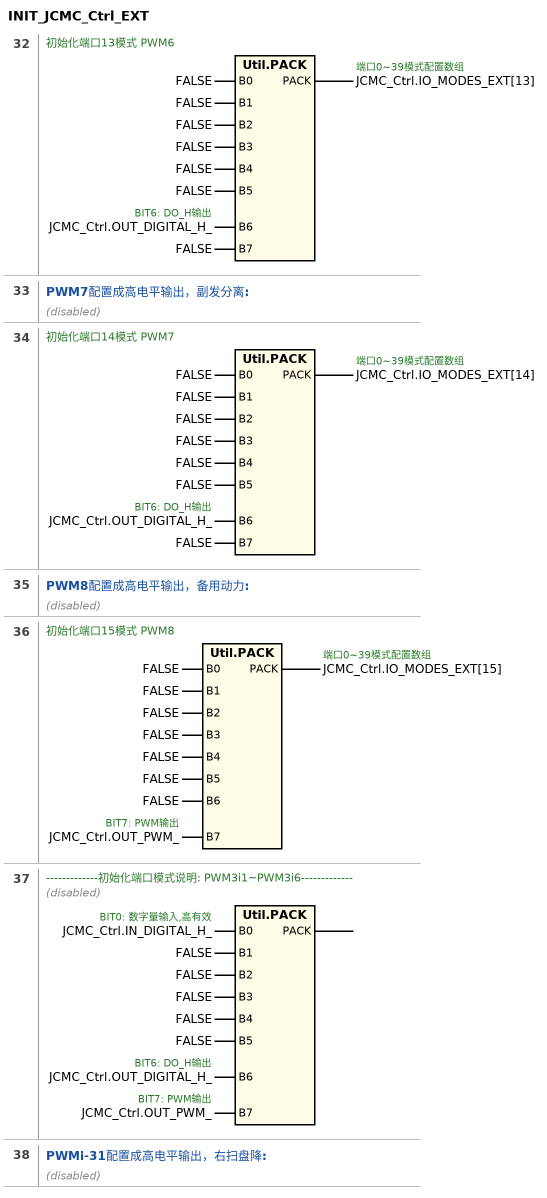
// NETWORK 32
// 初始化端口13模式 PWM6
//   JCMC_Ctrl.OUT_DIGITAL_H_: BIT6: DO_H输出
//   JCMC_Ctrl.IO_MODES_EXT[13]: 端口0~39模式配置数组
JCMC_Ctrl.IO_MODES_EXT[13] := Util.PACK(B0 := FALSE, B1 := FALSE, B2 := FALSE, B3 := FALSE, B4 := FALSE, B5 := FALSE, B6 := JCMC_Ctrl.OUT_DIGITAL_H_, B7 := FALSE);

// NETWORK 33 (disabled)
// label: PWM7配置成高电平输出，副发分离

// NETWORK 34
// 初始化端口14模式 PWM7
//   JCMC_Ctrl.OUT_DIGITAL_H_: BIT6: DO_H输出
//   JCMC_Ctrl.IO_MODES_EXT[14]: 端口0~39模式配置数组
JCMC_Ctrl.IO_MODES_EXT[14] := Util.PACK(B0 := FALSE, B1 := FALSE, B2 := FALSE, B3 := FALSE, B4 := FALSE, B5 := FALSE, B6 := JCMC_Ctrl.OUT_DIGITAL_H_, B7 := FALSE);

// NETWORK 35 (disabled)
// label: PWM8配置成高电平输出，备用动力

// NETWORK 36
// 初始化端口15模式 PWM8
//   JCMC_Ctrl.OUT_PWM_: BIT7: PWM输出
//   JCMC_Ctrl.IO_MODES_EXT[15]: 端口0~39模式配置数组
JCMC_Ctrl.IO_MODES_EXT[15] := Util.PACK(B0 := FALSE, B1 := FALSE, B2 := FALSE, B3 := FALSE, B4 := FALSE, B5 := FALSE, B6 := FALSE, B7 := JCMC_Ctrl.OUT_PWM_);

// NETWORK 37 (disabled)
// -------------初始化端口模式说明: PWM3i1~PWM3i6-------------
//   JCMC_Ctrl.IN_DIGITAL_H_: BIT0: 数字量输入,高有效
//   JCMC_Ctrl.OUT_DIGITAL_H_: BIT6: DO_H输出
//   JCMC_Ctrl.OUT_PWM_: BIT7: PWM输出
// ??? := Util.PACK(B0 := JCMC_Ctrl.IN_DIGITAL_H_, B1 := FALSE, B2 := FALSE, B3 := FALSE, B4 := FALSE, B5 := FALSE, B6 := JCMC_Ctrl.OUT_DIGITAL_H_, B7 := JCMC_Ctrl.OUT_PWM_);

// NETWORK 38 (disabled)
// label: PWMi-31配置成高电平输出，右扫盘降

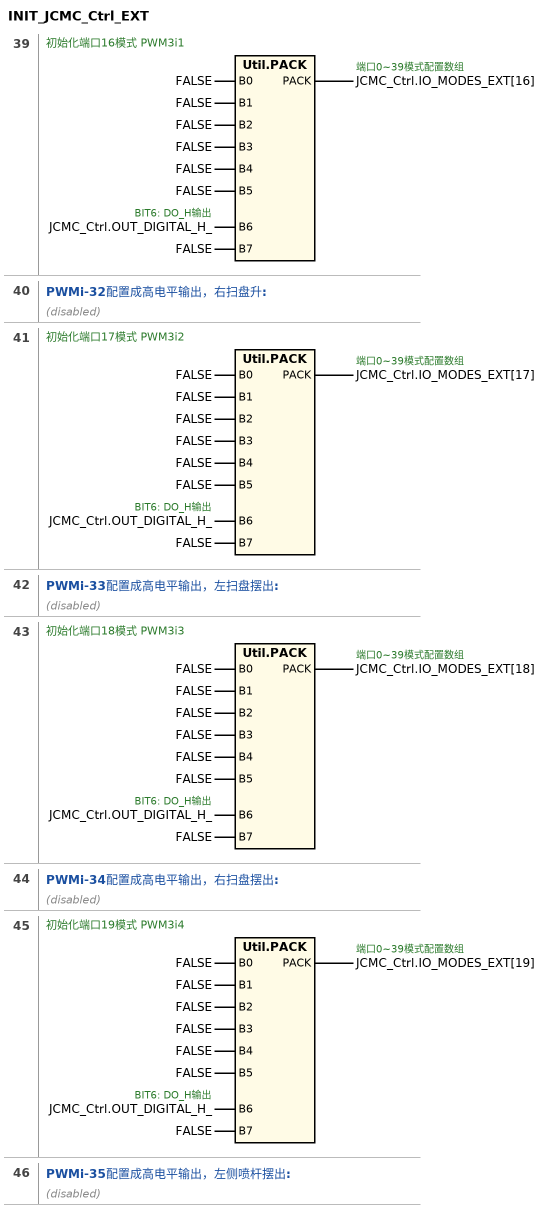
// NETWORK 39
// 初始化端口16模式 PWM3i1
//   JCMC_Ctrl.OUT_DIGITAL_H_: BIT6: DO_H输出
//   JCMC_Ctrl.IO_MODES_EXT[16]: 端口0~39模式配置数组
JCMC_Ctrl.IO_MODES_EXT[16] := Util.PACK(B0 := FALSE, B1 := FALSE, B2 := FALSE, B3 := FALSE, B4 := FALSE, B5 := FALSE, B6 := JCMC_Ctrl.OUT_DIGITAL_H_, B7 := FALSE);

// NETWORK 40 (disabled)
// label: PWMi-32配置成高电平输出，右扫盘升

// NETWORK 41
// 初始化端口17模式 PWM3i2
//   JCMC_Ctrl.OUT_DIGITAL_H_: BIT6: DO_H输出
//   JCMC_Ctrl.IO_MODES_EXT[17]: 端口0~39模式配置数组
JCMC_Ctrl.IO_MODES_EXT[17] := Util.PACK(B0 := FALSE, B1 := FALSE, B2 := FALSE, B3 := FALSE, B4 := FALSE, B5 := FALSE, B6 := JCMC_Ctrl.OUT_DIGITAL_H_, B7 := FALSE);

// NETWORK 42 (disabled)
// label: PWMi-33配置成高电平输出，左扫盘摆出

// NETWORK 43
// 初始化端口18模式 PWM3i3
//   JCMC_Ctrl.OUT_DIGITAL_H_: BIT6: DO_H输出
//   JCMC_Ctrl.IO_MODES_EXT[18]: 端口0~39模式配置数组
JCMC_Ctrl.IO_MODES_EXT[18] := Util.PACK(B0 := FALSE, B1 := FALSE, B2 := FALSE, B3 := FALSE, B4 := FALSE, B5 := FALSE, B6 := JCMC_Ctrl.OUT_DIGITAL_H_, B7 := FALSE);

// NETWORK 44 (disabled)
// label: PWMi-34配置成高电平输出，右扫盘摆出

// NETWORK 45
// 初始化端口19模式 PWM3i4
//   JCMC_Ctrl.OUT_DIGITAL_H_: BIT6: DO_H输出
//   JCMC_Ctrl.IO_MODES_EXT[19]: 端口0~39模式配置数组
JCMC_Ctrl.IO_MODES_EXT[19] := Util.PACK(B0 := FALSE, B1 := FALSE, B2 := FALSE, B3 := FALSE, B4 := FALSE, B5 := FALSE, B6 := JCMC_Ctrl.OUT_DIGITAL_H_, B7 := FALSE);

// NETWORK 46 (disabled)
// label: PWMi-35配置成高电平输出，左侧喷杆摆出

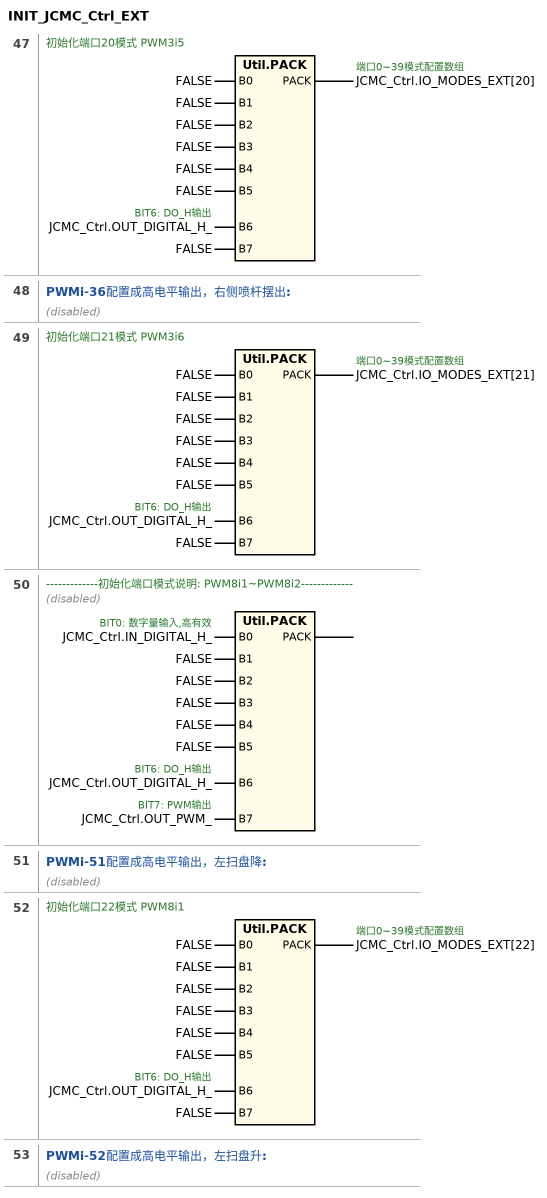
// NETWORK 47
// 初始化端口20模式 PWM3i5
//   JCMC_Ctrl.OUT_DIGITAL_H_: BIT6: DO_H输出
//   JCMC_Ctrl.IO_MODES_EXT[20]: 端口0~39模式配置数组
JCMC_Ctrl.IO_MODES_EXT[20] := Util.PACK(B0 := FALSE, B1 := FALSE, B2 := FALSE, B3 := FALSE, B4 := FALSE, B5 := FALSE, B6 := JCMC_Ctrl.OUT_DIGITAL_H_, B7 := FALSE);

// NETWORK 48 (disabled)
// label: PWMi-36配置成高电平输出，右侧喷杆摆出

// NETWORK 49
// 初始化端口21模式 PWM3i6
//   JCMC_Ctrl.OUT_DIGITAL_H_: BIT6: DO_H输出
//   JCMC_Ctrl.IO_MODES_EXT[21]: 端口0~39模式配置数组
JCMC_Ctrl.IO_MODES_EXT[21] := Util.PACK(B0 := FALSE, B1 := FALSE, B2 := FALSE, B3 := FALSE, B4 := FALSE, B5 := FALSE, B6 := JCMC_Ctrl.OUT_DIGITAL_H_, B7 := FALSE);

// NETWORK 50 (disabled)
// -------------初始化端口模式说明: PWM8i1~PWM8i2-------------
//   JCMC_Ctrl.IN_DIGITAL_H_: BIT0: 数字量输入,高有效
//   JCMC_Ctrl.OUT_DIGITAL_H_: BIT6: DO_H输出
//   JCMC_Ctrl.OUT_PWM_: BIT7: PWM输出
// ??? := Util.PACK(B0 := JCMC_Ctrl.IN_DIGITAL_H_, B1 := FALSE, B2 := FALSE, B3 := FALSE, B4 := FALSE, B5 := FALSE, B6 := JCMC_Ctrl.OUT_DIGITAL_H_, B7 := JCMC_Ctrl.OUT_PWM_);

// NETWORK 51 (disabled)
// label: PWMi-51配置成高电平输出，左扫盘降

// NETWORK 52
// 初始化端口22模式 PWM8i1
//   JCMC_Ctrl.OUT_DIGITAL_H_: BIT6: DO_H输出
//   JCMC_Ctrl.IO_MODES_EXT[22]: 端口0~39模式配置数组
JCMC_Ctrl.IO_MODES_EXT[22] := Util.PACK(B0 := FALSE, B1 := FALSE, B2 := FALSE, B3 := FALSE, B4 := FALSE, B5 := FALSE, B6 := JCMC_Ctrl.OUT_DIGITAL_H_, B7 := FALSE);

// NETWORK 53 (disabled)
// label: PWMi-52配置成高电平输出，左扫盘升

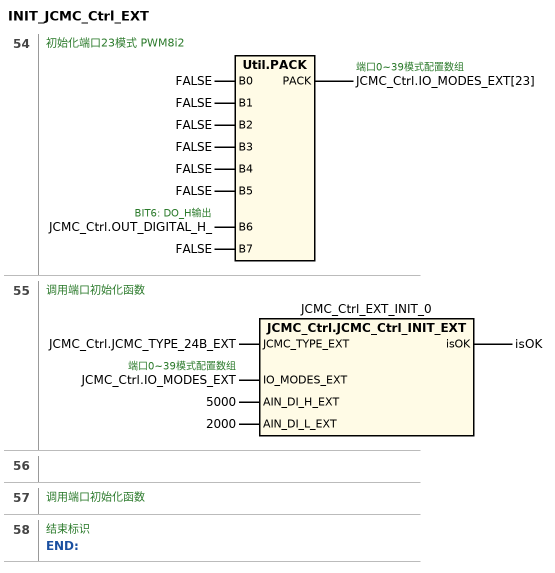
// NETWORK 54
// 初始化端口23模式 PWM8i2
//   JCMC_Ctrl.OUT_DIGITAL_H_: BIT6: DO_H输出
//   JCMC_Ctrl.IO_MODES_EXT[23]: 端口0~39模式配置数组
JCMC_Ctrl.IO_MODES_EXT[23] := Util.PACK(B0 := FALSE, B1 := FALSE, B2 := FALSE, B3 := FALSE, B4 := FALSE, B5 := FALSE, B6 := JCMC_Ctrl.OUT_DIGITAL_H_, B7 := FALSE);

// NETWORK 55
// 调用端口初始化函数
//   JCMC_Ctrl.IO_MODES_EXT: 端口0~39模式配置数组
JCMC_Ctrl_EXT_INIT_0(
    JCMC_TYPE_EXT := JCMC_Ctrl.JCMC_TYPE_24B_EXT,
    IO_MODES_EXT := JCMC_Ctrl.IO_MODES_EXT,
    AIN_DI_H_EXT := 5000,
    AIN_DI_L_EXT := 2000); // JCMC_Ctrl.JCMC_Ctrl_INIT_EXT
isOK := JCMC_Ctrl_EXT_INIT_0.isOK;

// NETWORK 56

// NETWORK 57
// 调用端口初始化函数

// NETWORK 58
// 结束标识
END: ;

END_PROGRAM

// Device/Application/INIT_JCMC_Ctrl
PROGRAM INIT_JCMC_Ctrl
VAR
	JCMC_Ctrl_INIT_0: JCMC_Ctrl.JCMC_Ctrl_INIT;
END_VAR

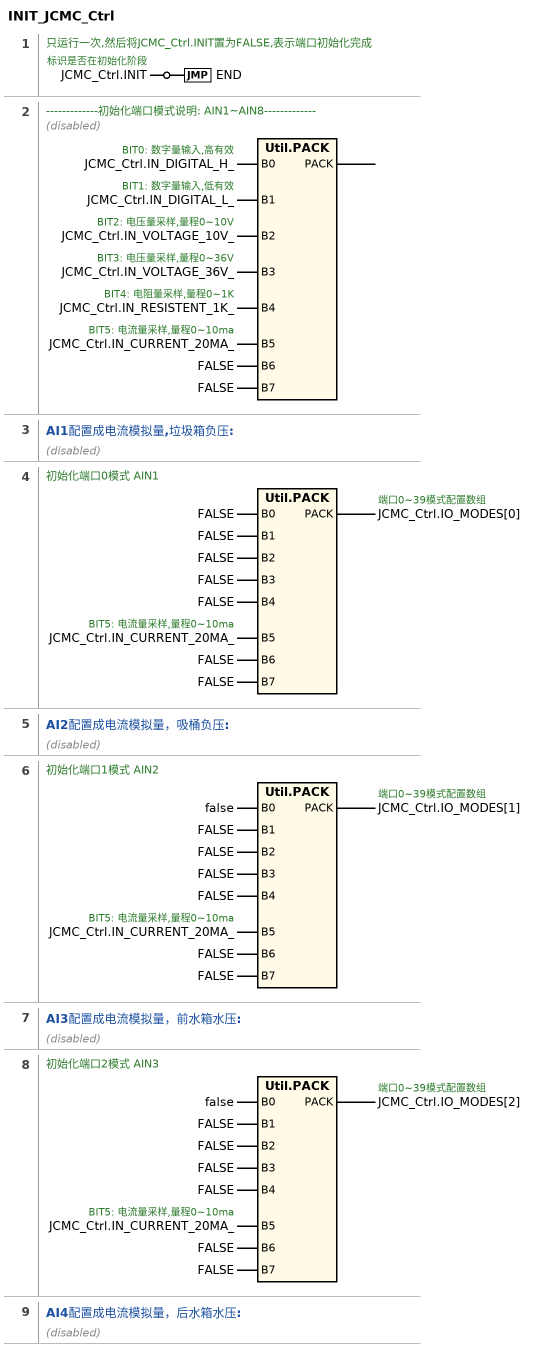
// NETWORK 1
// 只运行一次,然后将JCMC_Ctrl.INIT置为FALSE,表示端口初始化完成
//   JCMC_Ctrl.INIT: 标识是否在初始化阶段
IF NOT JCMC_Ctrl.INIT THEN JMP END; END_IF

// NETWORK 2 (disabled)
// -------------初始化端口模式说明: AIN1~AIN8-------------
//   JCMC_Ctrl.IN_DIGITAL_H_: BIT0: 数字量输入,高有效
//   JCMC_Ctrl.IN_DIGITAL_L_: BIT1: 数字量输入,低有效
//   JCMC_Ctrl.IN_VOLTAGE_10V_: BIT2: 电压量采样,量程0~10V
//   JCMC_Ctrl.IN_VOLTAGE_36V_: BIT3: 电压量采样,量程0~36V
//   JCMC_Ctrl.IN_RESISTENT_1K_: BIT4: 电阻量采样,量程0~1K
//   JCMC_Ctrl.IN_CURRENT_20MA_: BIT5: 电流量采样,量程0~10ma
// ??? := Util.PACK(B0 := JCMC_Ctrl.IN_DIGITAL_H_, B1 := JCMC_Ctrl.IN_DIGITAL_L_, B2 := JCMC_Ctrl.IN_VOLTAGE_10V_, B3 := JCMC_Ctrl.IN_VOLTAGE_36V_, B4 := JCMC_Ctrl.IN_RESISTENT_1K_, B5 := JCMC_Ctrl.IN_CURRENT_20MA_, B6 := FALSE, B7 := FALSE);

// NETWORK 3 (disabled)
// label: AI1配置成电流模拟量,垃圾箱负压

// NETWORK 4
// 初始化端口0模式 AIN1
//   JCMC_Ctrl.IN_CURRENT_20MA_: BIT5: 电流量采样,量程0~10ma
//   JCMC_Ctrl.IO_MODES[0]: 端口0~39模式配置数组
JCMC_Ctrl.IO_MODES[0] := Util.PACK(B0 := FALSE, B1 := FALSE, B2 := FALSE, B3 := FALSE, B4 := FALSE, B5 := JCMC_Ctrl.IN_CURRENT_20MA_, B6 := FALSE, B7 := FALSE);

// NETWORK 5 (disabled)
// label: AI2配置成电流模拟量，吸桶负压

// NETWORK 6
// 初始化端口1模式 AIN2
//   JCMC_Ctrl.IN_CURRENT_20MA_: BIT5: 电流量采样,量程0~10ma
//   JCMC_Ctrl.IO_MODES[1]: 端口0~39模式配置数组
JCMC_Ctrl.IO_MODES[1] := Util.PACK(B0 := false, B1 := FALSE, B2 := FALSE, B3 := FALSE, B4 := FALSE, B5 := JCMC_Ctrl.IN_CURRENT_20MA_, B6 := FALSE, B7 := FALSE);

// NETWORK 7 (disabled)
// label: AI3配置成电流模拟量，前水箱水压

// NETWORK 8
// 初始化端口2模式 AIN3
//   JCMC_Ctrl.IN_CURRENT_20MA_: BIT5: 电流量采样,量程0~10ma
//   JCMC_Ctrl.IO_MODES[2]: 端口0~39模式配置数组
JCMC_Ctrl.IO_MODES[2] := Util.PACK(B0 := false, B1 := FALSE, B2 := FALSE, B3 := FALSE, B4 := FALSE, B5 := JCMC_Ctrl.IN_CURRENT_20MA_, B6 := FALSE, B7 := FALSE);

// NETWORK 9 (disabled)
// label: AI4配置成电流模拟量，后水箱水压

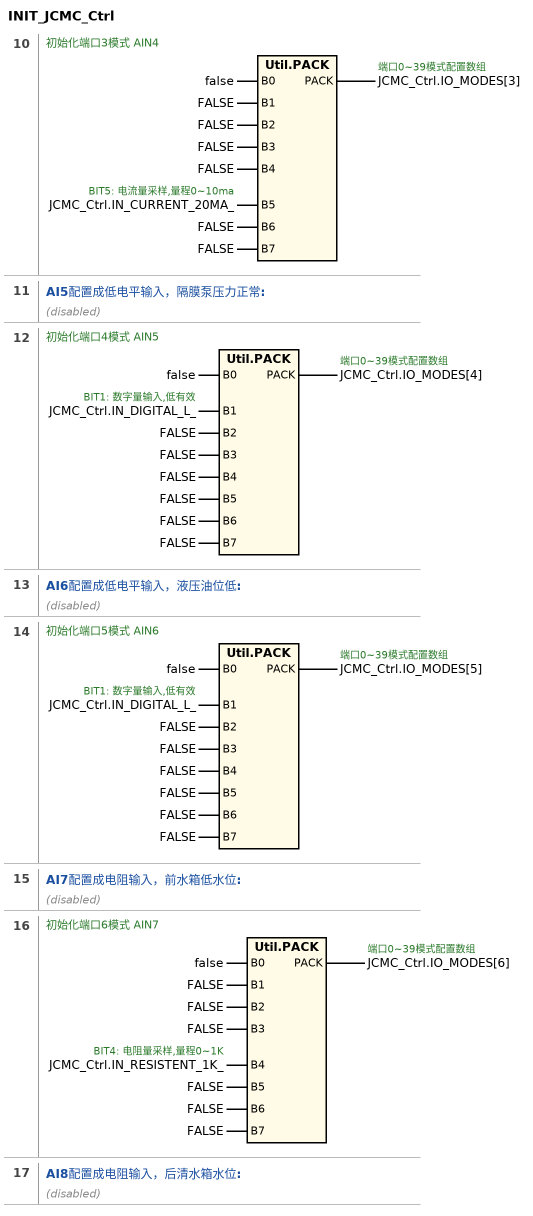
// NETWORK 10
// 初始化端口3模式 AIN4
//   JCMC_Ctrl.IN_CURRENT_20MA_: BIT5: 电流量采样,量程0~10ma
//   JCMC_Ctrl.IO_MODES[3]: 端口0~39模式配置数组
JCMC_Ctrl.IO_MODES[3] := Util.PACK(B0 := false, B1 := FALSE, B2 := FALSE, B3 := FALSE, B4 := FALSE, B5 := JCMC_Ctrl.IN_CURRENT_20MA_, B6 := FALSE, B7 := FALSE);

// NETWORK 11 (disabled)
// label: AI5配置成低电平输入，隔膜泵压力正常

// NETWORK 12
// 初始化端口4模式 AIN5
//   JCMC_Ctrl.IN_DIGITAL_L_: BIT1: 数字量输入,低有效
//   JCMC_Ctrl.IO_MODES[4]: 端口0~39模式配置数组
JCMC_Ctrl.IO_MODES[4] := Util.PACK(B0 := false, B1 := JCMC_Ctrl.IN_DIGITAL_L_, B2 := FALSE, B3 := FALSE, B4 := FALSE, B5 := FALSE, B6 := FALSE, B7 := FALSE);

// NETWORK 13 (disabled)
// label: AI6配置成低电平输入，液压油位低

// NETWORK 14
// 初始化端口5模式 AIN6
//   JCMC_Ctrl.IN_DIGITAL_L_: BIT1: 数字量输入,低有效
//   JCMC_Ctrl.IO_MODES[5]: 端口0~39模式配置数组
JCMC_Ctrl.IO_MODES[5] := Util.PACK(B0 := false, B1 := JCMC_Ctrl.IN_DIGITAL_L_, B2 := FALSE, B3 := FALSE, B4 := FALSE, B5 := FALSE, B6 := FALSE, B7 := FALSE);

// NETWORK 15 (disabled)
// label: AI7配置成电阻输入，前水箱低水位

// NETWORK 16
// 初始化端口6模式 AIN7
//   JCMC_Ctrl.IN_RESISTENT_1K_: BIT4: 电阻量采样,量程0~1K
//   JCMC_Ctrl.IO_MODES[6]: 端口0~39模式配置数组
JCMC_Ctrl.IO_MODES[6] := Util.PACK(B0 := false, B1 := FALSE, B2 := FALSE, B3 := FALSE, B4 := JCMC_Ctrl.IN_RESISTENT_1K_, B5 := FALSE, B6 := FALSE, B7 := FALSE);

// NETWORK 17 (disabled)
// label: AI8配置成电阻输入，后清水箱水位

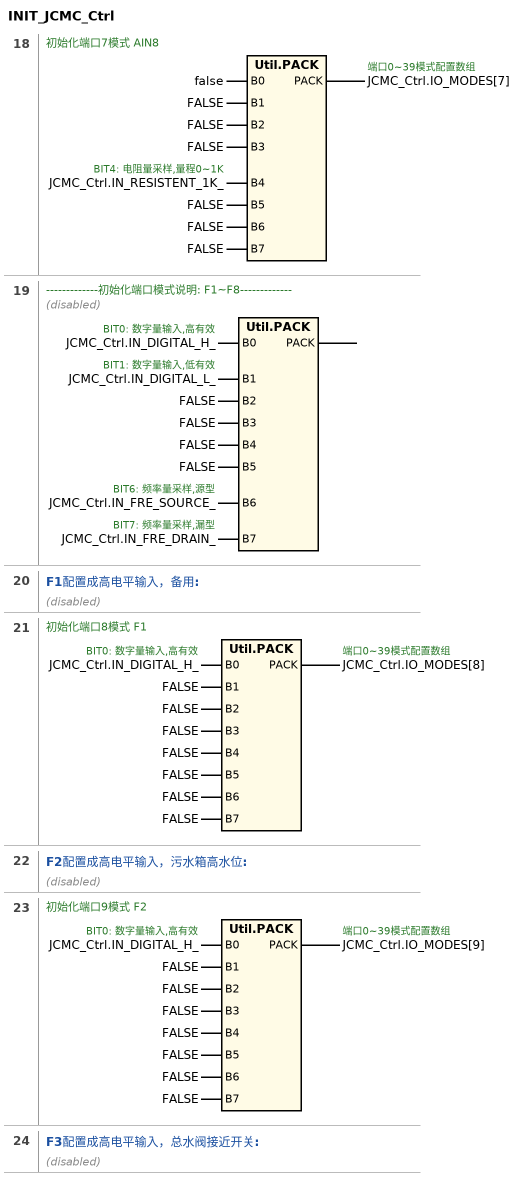
// NETWORK 18
// 初始化端口7模式 AIN8
//   JCMC_Ctrl.IN_RESISTENT_1K_: BIT4: 电阻量采样,量程0~1K
//   JCMC_Ctrl.IO_MODES[7]: 端口0~39模式配置数组
JCMC_Ctrl.IO_MODES[7] := Util.PACK(B0 := false, B1 := FALSE, B2 := FALSE, B3 := FALSE, B4 := JCMC_Ctrl.IN_RESISTENT_1K_, B5 := FALSE, B6 := FALSE, B7 := FALSE);

// NETWORK 19 (disabled)
// -------------初始化端口模式说明: F1~F8-------------
//   JCMC_Ctrl.IN_DIGITAL_H_: BIT0: 数字量输入,高有效
//   JCMC_Ctrl.IN_DIGITAL_L_: BIT1: 数字量输入,低有效
//   JCMC_Ctrl.IN_FRE_SOURCE_: BIT6: 频率量采样,源型
//   JCMC_Ctrl.IN_FRE_DRAIN_: BIT7: 频率量采样,漏型
// ??? := Util.PACK(B0 := JCMC_Ctrl.IN_DIGITAL_H_, B1 := JCMC_Ctrl.IN_DIGITAL_L_, B2 := FALSE, B3 := FALSE, B4 := FALSE, B5 := FALSE, B6 := JCMC_Ctrl.IN_FRE_SOURCE_, B7 := JCMC_Ctrl.IN_FRE_DRAIN_);

// NETWORK 20 (disabled)
// label: F1配置成高电平输入，备用

// NETWORK 21
// 初始化端口8模式 F1
//   JCMC_Ctrl.IN_DIGITAL_H_: BIT0: 数字量输入,高有效
//   JCMC_Ctrl.IO_MODES[8]: 端口0~39模式配置数组
JCMC_Ctrl.IO_MODES[8] := Util.PACK(B0 := JCMC_Ctrl.IN_DIGITAL_H_, B1 := FALSE, B2 := FALSE, B3 := FALSE, B4 := FALSE, B5 := FALSE, B6 := FALSE, B7 := FALSE);

// NETWORK 22 (disabled)
// label: F2配置成高电平输入，污水箱高水位

// NETWORK 23
// 初始化端口9模式 F2
//   JCMC_Ctrl.IN_DIGITAL_H_: BIT0: 数字量输入,高有效
//   JCMC_Ctrl.IO_MODES[9]: 端口0~39模式配置数组
JCMC_Ctrl.IO_MODES[9] := Util.PACK(B0 := JCMC_Ctrl.IN_DIGITAL_H_, B1 := FALSE, B2 := FALSE, B3 := FALSE, B4 := FALSE, B5 := FALSE, B6 := FALSE, B7 := FALSE);

// NETWORK 24 (disabled)
// label: F3配置成高电平输入，总水阀接近开关

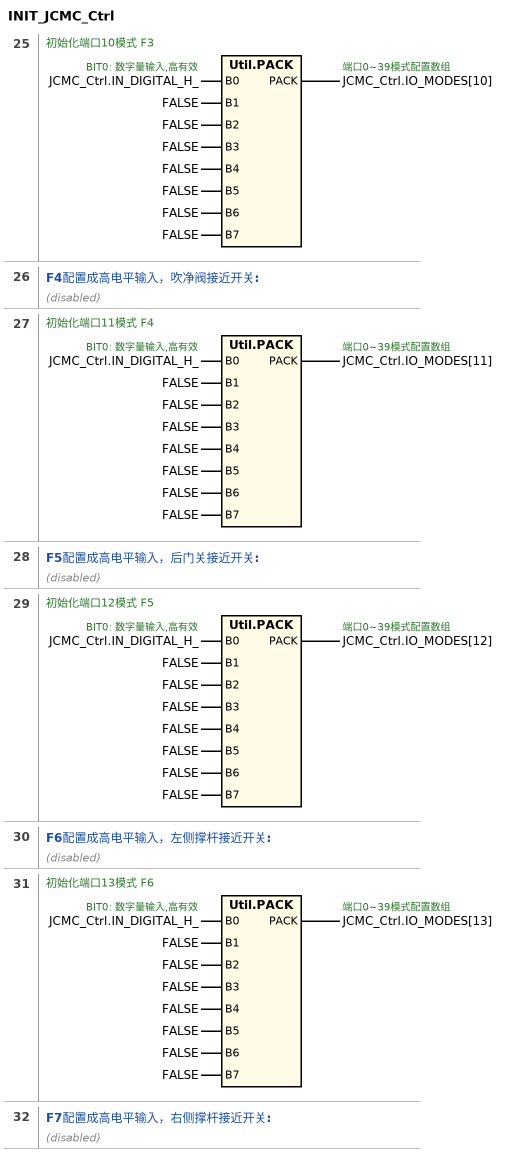
// NETWORK 25
// 初始化端口10模式 F3
//   JCMC_Ctrl.IN_DIGITAL_H_: BIT0: 数字量输入,高有效
//   JCMC_Ctrl.IO_MODES[10]: 端口0~39模式配置数组
JCMC_Ctrl.IO_MODES[10] := Util.PACK(B0 := JCMC_Ctrl.IN_DIGITAL_H_, B1 := FALSE, B2 := FALSE, B3 := FALSE, B4 := FALSE, B5 := FALSE, B6 := FALSE, B7 := FALSE);

// NETWORK 26 (disabled)
// label: F4配置成高电平输入，吹净阀接近开关

// NETWORK 27
// 初始化端口11模式 F4
//   JCMC_Ctrl.IN_DIGITAL_H_: BIT0: 数字量输入,高有效
//   JCMC_Ctrl.IO_MODES[11]: 端口0~39模式配置数组
JCMC_Ctrl.IO_MODES[11] := Util.PACK(B0 := JCMC_Ctrl.IN_DIGITAL_H_, B1 := FALSE, B2 := FALSE, B3 := FALSE, B4 := FALSE, B5 := FALSE, B6 := FALSE, B7 := FALSE);

// NETWORK 28 (disabled)
// label: F5配置成高电平输入，后门关接近开关

// NETWORK 29
// 初始化端口12模式 F5
//   JCMC_Ctrl.IN_DIGITAL_H_: BIT0: 数字量输入,高有效
//   JCMC_Ctrl.IO_MODES[12]: 端口0~39模式配置数组
JCMC_Ctrl.IO_MODES[12] := Util.PACK(B0 := JCMC_Ctrl.IN_DIGITAL_H_, B1 := FALSE, B2 := FALSE, B3 := FALSE, B4 := FALSE, B5 := FALSE, B6 := FALSE, B7 := FALSE);

// NETWORK 30 (disabled)
// label: F6配置成高电平输入，左侧撑杆接近开关

// NETWORK 31
// 初始化端口13模式 F6
//   JCMC_Ctrl.IN_DIGITAL_H_: BIT0: 数字量输入,高有效
//   JCMC_Ctrl.IO_MODES[13]: 端口0~39模式配置数组
JCMC_Ctrl.IO_MODES[13] := Util.PACK(B0 := JCMC_Ctrl.IN_DIGITAL_H_, B1 := FALSE, B2 := FALSE, B3 := FALSE, B4 := FALSE, B5 := FALSE, B6 := FALSE, B7 := FALSE);

// NETWORK 32 (disabled)
// label: F7配置成高电平输入，右侧撑杆接近开关

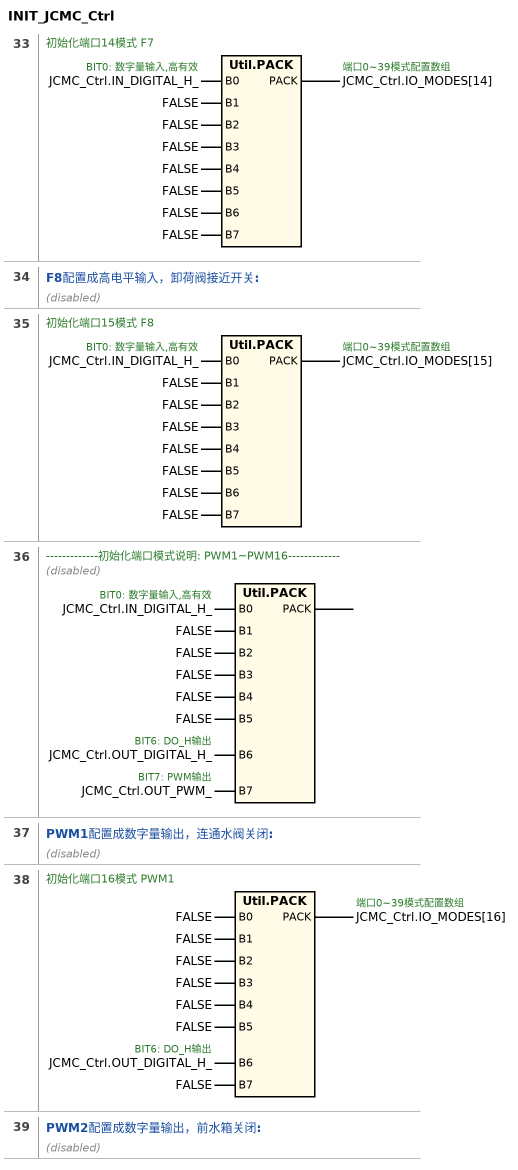
// NETWORK 33
// 初始化端口14模式 F7
//   JCMC_Ctrl.IN_DIGITAL_H_: BIT0: 数字量输入,高有效
//   JCMC_Ctrl.IO_MODES[14]: 端口0~39模式配置数组
JCMC_Ctrl.IO_MODES[14] := Util.PACK(B0 := JCMC_Ctrl.IN_DIGITAL_H_, B1 := FALSE, B2 := FALSE, B3 := FALSE, B4 := FALSE, B5 := FALSE, B6 := FALSE, B7 := FALSE);

// NETWORK 34 (disabled)
// label: F8配置成高电平输入，卸荷阀接近开关

// NETWORK 35
// 初始化端口15模式 F8
//   JCMC_Ctrl.IN_DIGITAL_H_: BIT0: 数字量输入,高有效
//   JCMC_Ctrl.IO_MODES[15]: 端口0~39模式配置数组
JCMC_Ctrl.IO_MODES[15] := Util.PACK(B0 := JCMC_Ctrl.IN_DIGITAL_H_, B1 := FALSE, B2 := FALSE, B3 := FALSE, B4 := FALSE, B5 := FALSE, B6 := FALSE, B7 := FALSE);

// NETWORK 36 (disabled)
// -------------初始化端口模式说明: PWM1~PWM16-------------
//   JCMC_Ctrl.IN_DIGITAL_H_: BIT0: 数字量输入,高有效
//   JCMC_Ctrl.OUT_DIGITAL_H_: BIT6: DO_H输出
//   JCMC_Ctrl.OUT_PWM_: BIT7: PWM输出
// ??? := Util.PACK(B0 := JCMC_Ctrl.IN_DIGITAL_H_, B1 := FALSE, B2 := FALSE, B3 := FALSE, B4 := FALSE, B5 := FALSE, B6 := JCMC_Ctrl.OUT_DIGITAL_H_, B7 := JCMC_Ctrl.OUT_PWM_);

// NETWORK 37 (disabled)
// label: PWM1配置成数字量输出，连通水阀关闭

// NETWORK 38
// 初始化端口16模式 PWM1
//   JCMC_Ctrl.OUT_DIGITAL_H_: BIT6: DO_H输出
//   JCMC_Ctrl.IO_MODES[16]: 端口0~39模式配置数组
JCMC_Ctrl.IO_MODES[16] := Util.PACK(B0 := FALSE, B1 := FALSE, B2 := FALSE, B3 := FALSE, B4 := FALSE, B5 := FALSE, B6 := JCMC_Ctrl.OUT_DIGITAL_H_, B7 := FALSE);

// NETWORK 39 (disabled)
// label: PWM2配置成数字量输出，前水箱关闭

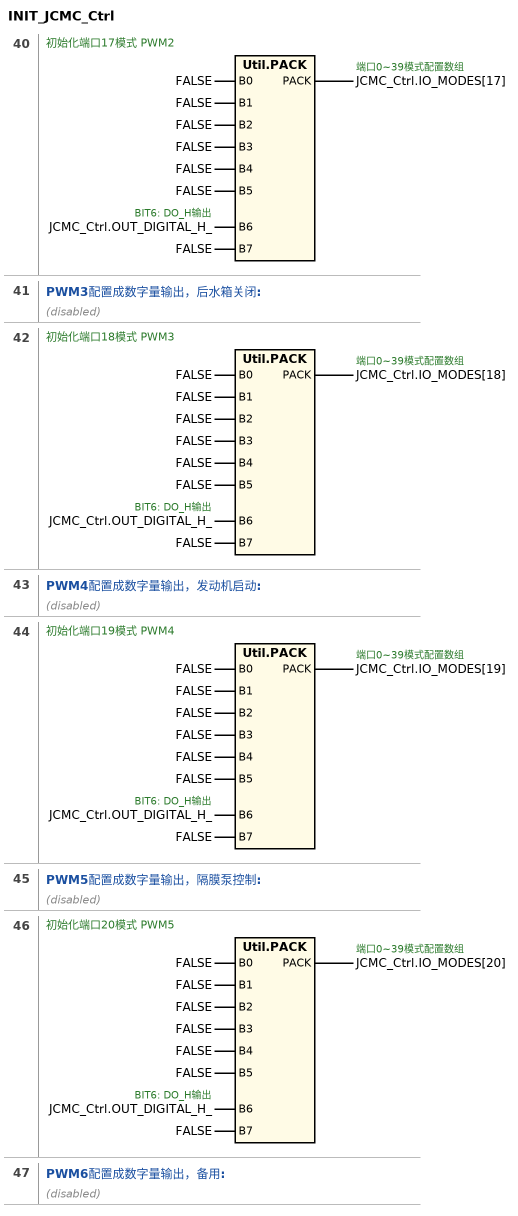
// NETWORK 40
// 初始化端口17模式 PWM2
//   JCMC_Ctrl.OUT_DIGITAL_H_: BIT6: DO_H输出
//   JCMC_Ctrl.IO_MODES[17]: 端口0~39模式配置数组
JCMC_Ctrl.IO_MODES[17] := Util.PACK(B0 := FALSE, B1 := FALSE, B2 := FALSE, B3 := FALSE, B4 := FALSE, B5 := FALSE, B6 := JCMC_Ctrl.OUT_DIGITAL_H_, B7 := FALSE);

// NETWORK 41 (disabled)
// label: PWM3配置成数字量输出，后水箱关闭

// NETWORK 42
// 初始化端口18模式 PWM3
//   JCMC_Ctrl.OUT_DIGITAL_H_: BIT6: DO_H输出
//   JCMC_Ctrl.IO_MODES[18]: 端口0~39模式配置数组
JCMC_Ctrl.IO_MODES[18] := Util.PACK(B0 := FALSE, B1 := FALSE, B2 := FALSE, B3 := FALSE, B4 := FALSE, B5 := FALSE, B6 := JCMC_Ctrl.OUT_DIGITAL_H_, B7 := FALSE);

// NETWORK 43 (disabled)
// label: PWM4配置成数字量输出，发动机启动

// NETWORK 44
// 初始化端口19模式 PWM4
//   JCMC_Ctrl.OUT_DIGITAL_H_: BIT6: DO_H输出
//   JCMC_Ctrl.IO_MODES[19]: 端口0~39模式配置数组
JCMC_Ctrl.IO_MODES[19] := Util.PACK(B0 := FALSE, B1 := FALSE, B2 := FALSE, B3 := FALSE, B4 := FALSE, B5 := FALSE, B6 := JCMC_Ctrl.OUT_DIGITAL_H_, B7 := FALSE);

// NETWORK 45 (disabled)
// label: PWM5配置成数字量输出，隔膜泵控制

// NETWORK 46
// 初始化端口20模式 PWM5
//   JCMC_Ctrl.OUT_DIGITAL_H_: BIT6: DO_H输出
//   JCMC_Ctrl.IO_MODES[20]: 端口0~39模式配置数组
JCMC_Ctrl.IO_MODES[20] := Util.PACK(B0 := FALSE, B1 := FALSE, B2 := FALSE, B3 := FALSE, B4 := FALSE, B5 := FALSE, B6 := JCMC_Ctrl.OUT_DIGITAL_H_, B7 := FALSE);

// NETWORK 47 (disabled)
// label: PWM6配置成数字量输出，备用

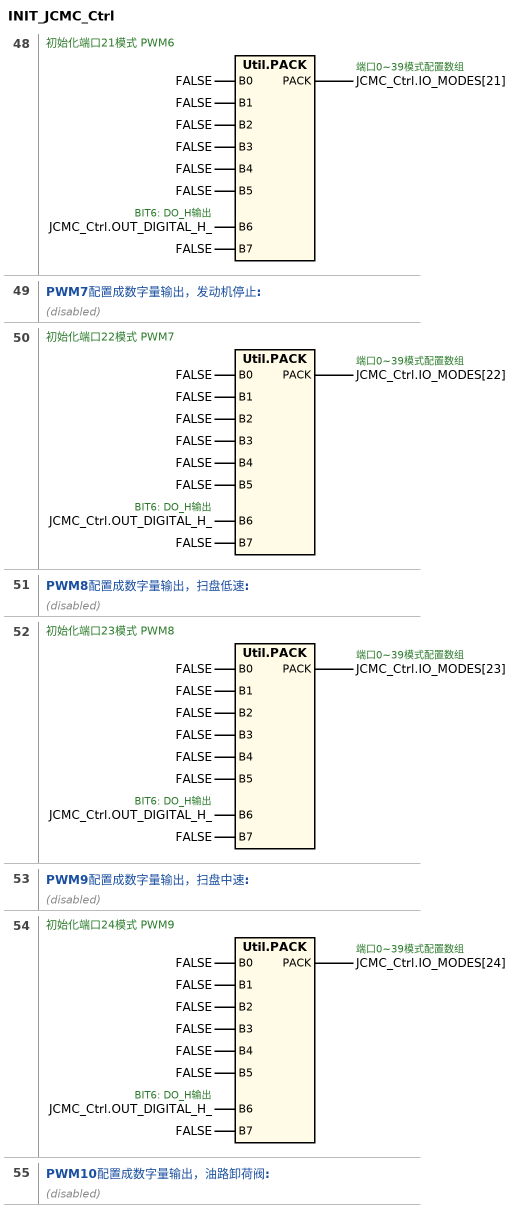
// NETWORK 48
// 初始化端口21模式 PWM6
//   JCMC_Ctrl.OUT_DIGITAL_H_: BIT6: DO_H输出
//   JCMC_Ctrl.IO_MODES[21]: 端口0~39模式配置数组
JCMC_Ctrl.IO_MODES[21] := Util.PACK(B0 := FALSE, B1 := FALSE, B2 := FALSE, B3 := FALSE, B4 := FALSE, B5 := FALSE, B6 := JCMC_Ctrl.OUT_DIGITAL_H_, B7 := FALSE);

// NETWORK 49 (disabled)
// label: PWM7配置成数字量输出，发动机停止

// NETWORK 50
// 初始化端口22模式 PWM7
//   JCMC_Ctrl.OUT_DIGITAL_H_: BIT6: DO_H输出
//   JCMC_Ctrl.IO_MODES[22]: 端口0~39模式配置数组
JCMC_Ctrl.IO_MODES[22] := Util.PACK(B0 := FALSE, B1 := FALSE, B2 := FALSE, B3 := FALSE, B4 := FALSE, B5 := FALSE, B6 := JCMC_Ctrl.OUT_DIGITAL_H_, B7 := FALSE);

// NETWORK 51 (disabled)
// label: PWM8配置成数字量输出，扫盘低速

// NETWORK 52
// 初始化端口23模式 PWM8
//   JCMC_Ctrl.OUT_DIGITAL_H_: BIT6: DO_H输出
//   JCMC_Ctrl.IO_MODES[23]: 端口0~39模式配置数组
JCMC_Ctrl.IO_MODES[23] := Util.PACK(B0 := FALSE, B1 := FALSE, B2 := FALSE, B3 := FALSE, B4 := FALSE, B5 := FALSE, B6 := JCMC_Ctrl.OUT_DIGITAL_H_, B7 := FALSE);

// NETWORK 53 (disabled)
// label: PWM9配置成数字量输出，扫盘中速

// NETWORK 54
// 初始化端口24模式 PWM9
//   JCMC_Ctrl.OUT_DIGITAL_H_: BIT6: DO_H输出
//   JCMC_Ctrl.IO_MODES[24]: 端口0~39模式配置数组
JCMC_Ctrl.IO_MODES[24] := Util.PACK(B0 := FALSE, B1 := FALSE, B2 := FALSE, B3 := FALSE, B4 := FALSE, B5 := FALSE, B6 := JCMC_Ctrl.OUT_DIGITAL_H_, B7 := FALSE);

// NETWORK 55 (disabled)
// label: PWM10配置成数字量输出，油路卸荷阀

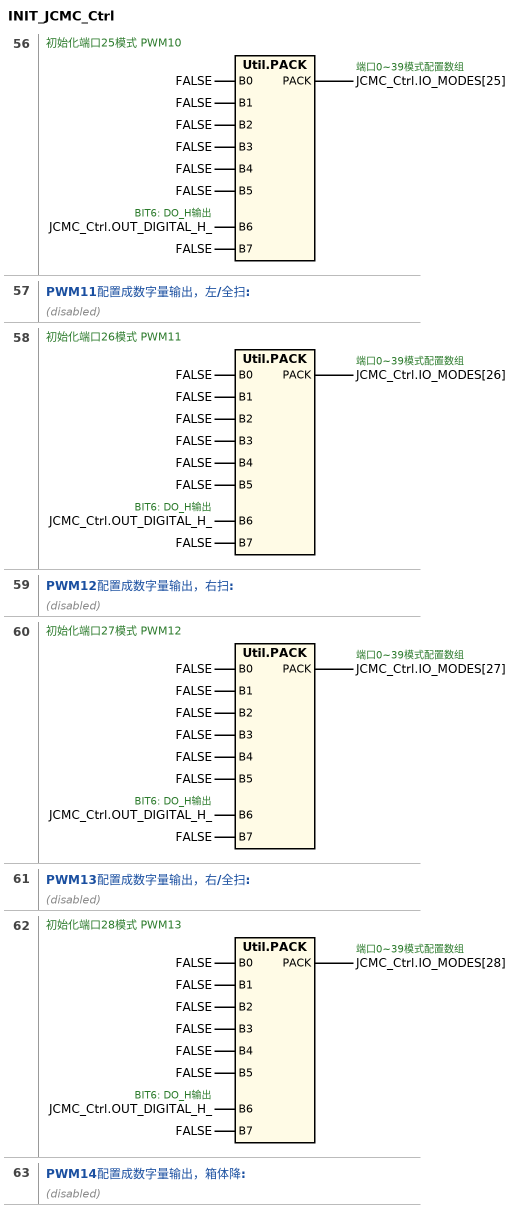
// NETWORK 56
// 初始化端口25模式 PWM10
//   JCMC_Ctrl.OUT_DIGITAL_H_: BIT6: DO_H输出
//   JCMC_Ctrl.IO_MODES[25]: 端口0~39模式配置数组
JCMC_Ctrl.IO_MODES[25] := Util.PACK(B0 := FALSE, B1 := FALSE, B2 := FALSE, B3 := FALSE, B4 := FALSE, B5 := FALSE, B6 := JCMC_Ctrl.OUT_DIGITAL_H_, B7 := FALSE);

// NETWORK 57 (disabled)
// label: PWM11配置成数字量输出，左/全扫

// NETWORK 58
// 初始化端口26模式 PWM11
//   JCMC_Ctrl.OUT_DIGITAL_H_: BIT6: DO_H输出
//   JCMC_Ctrl.IO_MODES[26]: 端口0~39模式配置数组
JCMC_Ctrl.IO_MODES[26] := Util.PACK(B0 := FALSE, B1 := FALSE, B2 := FALSE, B3 := FALSE, B4 := FALSE, B5 := FALSE, B6 := JCMC_Ctrl.OUT_DIGITAL_H_, B7 := FALSE);

// NETWORK 59 (disabled)
// label: PWM12配置成数字量输出，右扫

// NETWORK 60
// 初始化端口27模式 PWM12
//   JCMC_Ctrl.OUT_DIGITAL_H_: BIT6: DO_H输出
//   JCMC_Ctrl.IO_MODES[27]: 端口0~39模式配置数组
JCMC_Ctrl.IO_MODES[27] := Util.PACK(B0 := FALSE, B1 := FALSE, B2 := FALSE, B3 := FALSE, B4 := FALSE, B5 := FALSE, B6 := JCMC_Ctrl.OUT_DIGITAL_H_, B7 := FALSE);

// NETWORK 61 (disabled)
// label: PWM13配置成数字量输出，右/全扫

// NETWORK 62
// 初始化端口28模式 PWM13
//   JCMC_Ctrl.OUT_DIGITAL_H_: BIT6: DO_H输出
//   JCMC_Ctrl.IO_MODES[28]: 端口0~39模式配置数组
JCMC_Ctrl.IO_MODES[28] := Util.PACK(B0 := FALSE, B1 := FALSE, B2 := FALSE, B3 := FALSE, B4 := FALSE, B5 := FALSE, B6 := JCMC_Ctrl.OUT_DIGITAL_H_, B7 := FALSE);

// NETWORK 63 (disabled)
// label: PWM14配置成数字量输出，箱体降

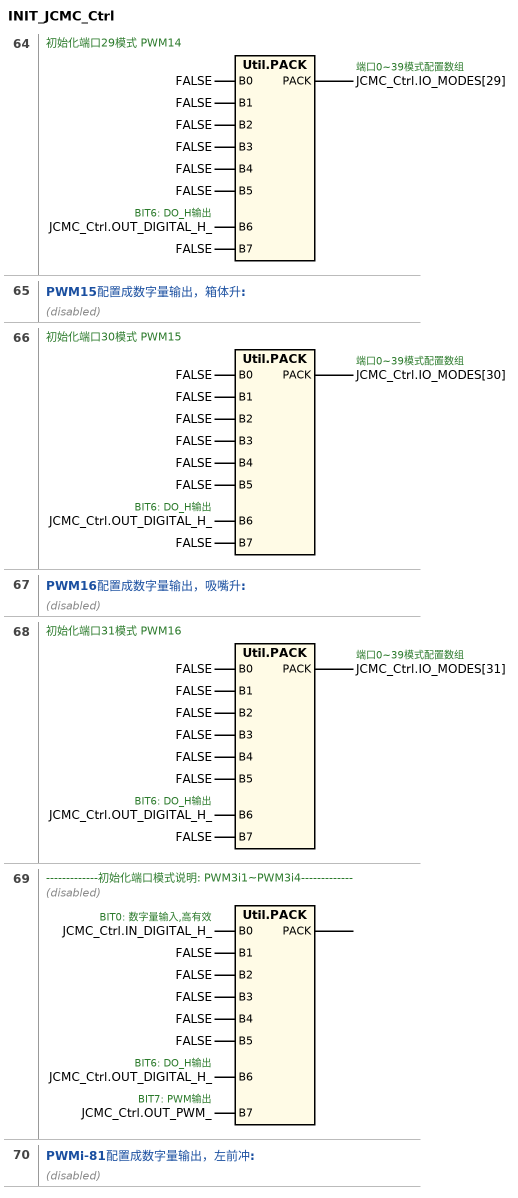
// NETWORK 64
// 初始化端口29模式 PWM14
//   JCMC_Ctrl.OUT_DIGITAL_H_: BIT6: DO_H输出
//   JCMC_Ctrl.IO_MODES[29]: 端口0~39模式配置数组
JCMC_Ctrl.IO_MODES[29] := Util.PACK(B0 := FALSE, B1 := FALSE, B2 := FALSE, B3 := FALSE, B4 := FALSE, B5 := FALSE, B6 := JCMC_Ctrl.OUT_DIGITAL_H_, B7 := FALSE);

// NETWORK 65 (disabled)
// label: PWM15配置成数字量输出，箱体升

// NETWORK 66
// 初始化端口30模式 PWM15
//   JCMC_Ctrl.OUT_DIGITAL_H_: BIT6: DO_H输出
//   JCMC_Ctrl.IO_MODES[30]: 端口0~39模式配置数组
JCMC_Ctrl.IO_MODES[30] := Util.PACK(B0 := FALSE, B1 := FALSE, B2 := FALSE, B3 := FALSE, B4 := FALSE, B5 := FALSE, B6 := JCMC_Ctrl.OUT_DIGITAL_H_, B7 := FALSE);

// NETWORK 67 (disabled)
// label: PWM16配置成数字量输出，吸嘴升

// NETWORK 68
// 初始化端口31模式 PWM16
//   JCMC_Ctrl.OUT_DIGITAL_H_: BIT6: DO_H输出
//   JCMC_Ctrl.IO_MODES[31]: 端口0~39模式配置数组
JCMC_Ctrl.IO_MODES[31] := Util.PACK(B0 := FALSE, B1 := FALSE, B2 := FALSE, B3 := FALSE, B4 := FALSE, B5 := FALSE, B6 := JCMC_Ctrl.OUT_DIGITAL_H_, B7 := FALSE);

// NETWORK 69 (disabled)
// -------------初始化端口模式说明: PWM3i1~PWM3i4-------------
//   JCMC_Ctrl.IN_DIGITAL_H_: BIT0: 数字量输入,高有效
//   JCMC_Ctrl.OUT_DIGITAL_H_: BIT6: DO_H输出
//   JCMC_Ctrl.OUT_PWM_: BIT7: PWM输出
// ??? := Util.PACK(B0 := JCMC_Ctrl.IN_DIGITAL_H_, B1 := FALSE, B2 := FALSE, B3 := FALSE, B4 := FALSE, B5 := FALSE, B6 := JCMC_Ctrl.OUT_DIGITAL_H_, B7 := JCMC_Ctrl.OUT_PWM_);

// NETWORK 70 (disabled)
// label: PWMi-81配置成数字量输出，左前冲

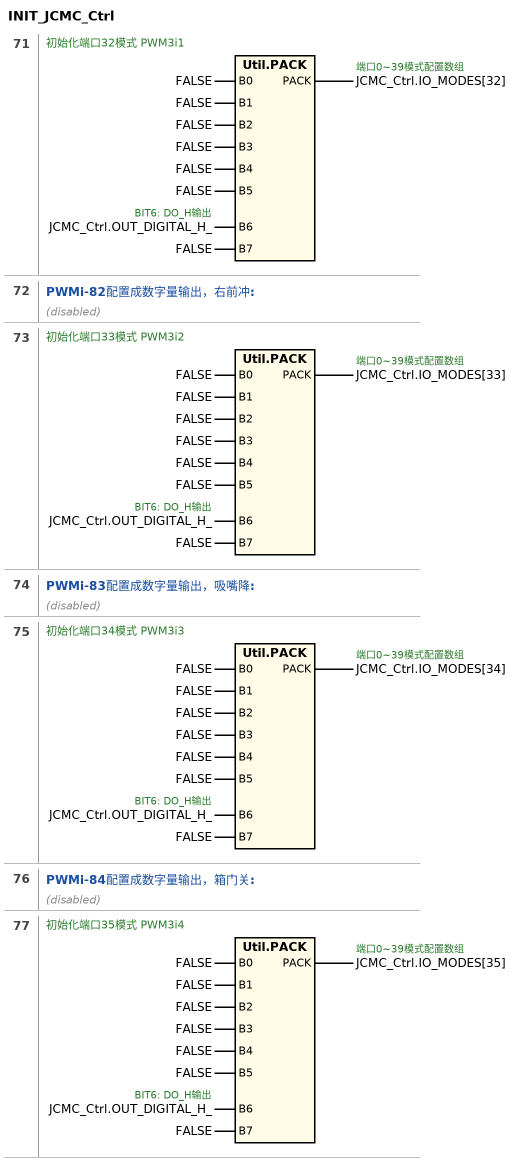
// NETWORK 71
// 初始化端口32模式 PWM3i1
//   JCMC_Ctrl.OUT_DIGITAL_H_: BIT6: DO_H输出
//   JCMC_Ctrl.IO_MODES[32]: 端口0~39模式配置数组
JCMC_Ctrl.IO_MODES[32] := Util.PACK(B0 := FALSE, B1 := FALSE, B2 := FALSE, B3 := FALSE, B4 := FALSE, B5 := FALSE, B6 := JCMC_Ctrl.OUT_DIGITAL_H_, B7 := FALSE);

// NETWORK 72 (disabled)
// label: PWMi-82配置成数字量输出，右前冲

// NETWORK 73
// 初始化端口33模式 PWM3i2
//   JCMC_Ctrl.OUT_DIGITAL_H_: BIT6: DO_H输出
//   JCMC_Ctrl.IO_MODES[33]: 端口0~39模式配置数组
JCMC_Ctrl.IO_MODES[33] := Util.PACK(B0 := FALSE, B1 := FALSE, B2 := FALSE, B3 := FALSE, B4 := FALSE, B5 := FALSE, B6 := JCMC_Ctrl.OUT_DIGITAL_H_, B7 := FALSE);

// NETWORK 74 (disabled)
// label: PWMi-83配置成数字量输出，吸嘴降

// NETWORK 75
// 初始化端口34模式 PWM3i3
//   JCMC_Ctrl.OUT_DIGITAL_H_: BIT6: DO_H输出
//   JCMC_Ctrl.IO_MODES[34]: 端口0~39模式配置数组
JCMC_Ctrl.IO_MODES[34] := Util.PACK(B0 := FALSE, B1 := FALSE, B2 := FALSE, B3 := FALSE, B4 := FALSE, B5 := FALSE, B6 := JCMC_Ctrl.OUT_DIGITAL_H_, B7 := FALSE);

// NETWORK 76 (disabled)
// label: PWMi-84配置成数字量输出，箱门关

// NETWORK 77
// 初始化端口35模式 PWM3i4
//   JCMC_Ctrl.OUT_DIGITAL_H_: BIT6: DO_H输出
//   JCMC_Ctrl.IO_MODES[35]: 端口0~39模式配置数组
JCMC_Ctrl.IO_MODES[35] := Util.PACK(B0 := FALSE, B1 := FALSE, B2 := FALSE, B3 := FALSE, B4 := FALSE, B5 := FALSE, B6 := JCMC_Ctrl.OUT_DIGITAL_H_, B7 := FALSE);

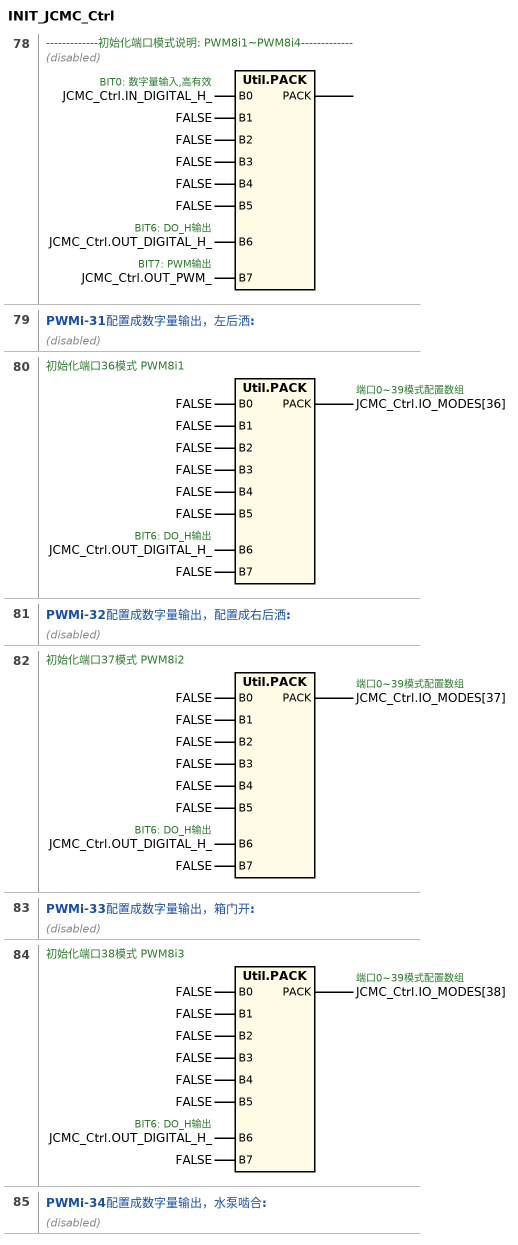
// NETWORK 78 (disabled)
// -------------初始化端口模式说明: PWM8i1~PWM8i4-------------
//   JCMC_Ctrl.IN_DIGITAL_H_: BIT0: 数字量输入,高有效
//   JCMC_Ctrl.OUT_DIGITAL_H_: BIT6: DO_H输出
//   JCMC_Ctrl.OUT_PWM_: BIT7: PWM输出
// ??? := Util.PACK(B0 := JCMC_Ctrl.IN_DIGITAL_H_, B1 := FALSE, B2 := FALSE, B3 := FALSE, B4 := FALSE, B5 := FALSE, B6 := JCMC_Ctrl.OUT_DIGITAL_H_, B7 := JCMC_Ctrl.OUT_PWM_);

// NETWORK 79 (disabled)
// label: PWMi-31配置成数字量输出，左后洒

// NETWORK 80
// 初始化端口36模式 PWM8i1
//   JCMC_Ctrl.OUT_DIGITAL_H_: BIT6: DO_H输出
//   JCMC_Ctrl.IO_MODES[36]: 端口0~39模式配置数组
JCMC_Ctrl.IO_MODES[36] := Util.PACK(B0 := FALSE, B1 := FALSE, B2 := FALSE, B3 := FALSE, B4 := FALSE, B5 := FALSE, B6 := JCMC_Ctrl.OUT_DIGITAL_H_, B7 := FALSE);

// NETWORK 81 (disabled)
// label: PWMi-32配置成数字量输出，配置成右后洒

// NETWORK 82
// 初始化端口37模式 PWM8i2
//   JCMC_Ctrl.OUT_DIGITAL_H_: BIT6: DO_H输出
//   JCMC_Ctrl.IO_MODES[37]: 端口0~39模式配置数组
JCMC_Ctrl.IO_MODES[37] := Util.PACK(B0 := FALSE, B1 := FALSE, B2 := FALSE, B3 := FALSE, B4 := FALSE, B5 := FALSE, B6 := JCMC_Ctrl.OUT_DIGITAL_H_, B7 := FALSE);

// NETWORK 83 (disabled)
// label: PWMi-33配置成数字量输出，箱门开

// NETWORK 84
// 初始化端口38模式 PWM8i3
//   JCMC_Ctrl.OUT_DIGITAL_H_: BIT6: DO_H输出
//   JCMC_Ctrl.IO_MODES[38]: 端口0~39模式配置数组
JCMC_Ctrl.IO_MODES[38] := Util.PACK(B0 := FALSE, B1 := FALSE, B2 := FALSE, B3 := FALSE, B4 := FALSE, B5 := FALSE, B6 := JCMC_Ctrl.OUT_DIGITAL_H_, B7 := FALSE);

// NETWORK 85 (disabled)
// label: PWMi-34配置成数字量输出，水泵啮合

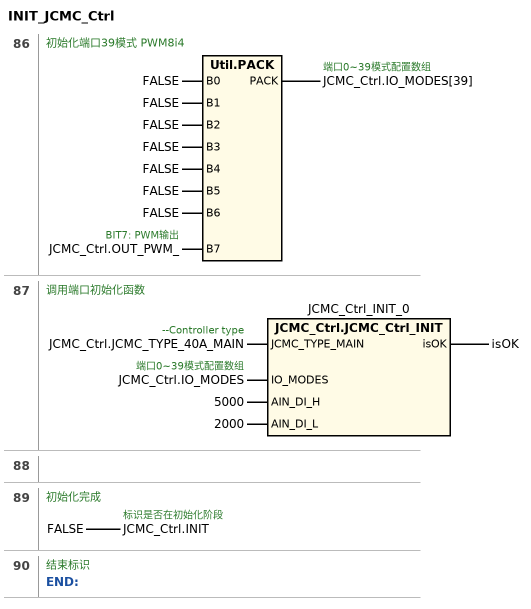
// NETWORK 86
// 初始化端口39模式 PWM8i4
//   JCMC_Ctrl.OUT_PWM_: BIT7: PWM输出
//   JCMC_Ctrl.IO_MODES[39]: 端口0~39模式配置数组
JCMC_Ctrl.IO_MODES[39] := Util.PACK(B0 := FALSE, B1 := FALSE, B2 := FALSE, B3 := FALSE, B4 := FALSE, B5 := FALSE, B6 := FALSE, B7 := JCMC_Ctrl.OUT_PWM_);

// NETWORK 87
// 调用端口初始化函数
//   JCMC_Ctrl.JCMC_TYPE_40A_MAIN: --Controller type
//   JCMC_Ctrl.IO_MODES: 端口0~39模式配置数组
JCMC_Ctrl_INIT_0(
    JCMC_TYPE_MAIN := JCMC_Ctrl.JCMC_TYPE_40A_MAIN,
    IO_MODES := JCMC_Ctrl.IO_MODES,
    AIN_DI_H := 5000,
    AIN_DI_L := 2000); // JCMC_Ctrl.JCMC_Ctrl_INIT
isOK := JCMC_Ctrl_INIT_0.isOK;

// NETWORK 88

// NETWORK 89
// 初始化完成
//   JCMC_Ctrl.INIT: 标识是否在初始化阶段
JCMC_Ctrl.INIT := FALSE;

// NETWORK 90
// 结束标识
END: ;

END_PROGRAM

// Device/Application/PLC_PRG
PROGRAM PLC_PRG
VAR
	sysTick: DWORD:=0;
END_VAR

sysTick := sysTick + 1;

parameterConfigure();    //系统配置
handleInput40A();   //40A板卡输入信号处理
handleInput24B();   //24B板卡输入信号处理
receiveFromHMI();  //接收HMI信息
receiveFromEngineECM();//接收副发动机信息
receiveFromECU();//接收底盘ECU信息
receiveFromSiliconePanel();//接收硅胶面板信息

faultHandle();   //系统故障处理
engineControl(); //发动机启停控制
IF systemStatus.systemTest THEN
	functionTest();  //功能测试
	ELSE
	resetTestST();  //复位测试状态
END_IF
chooseWorkMode(); //选择工作模式
workflowCore();  //核心工艺流程
workflowOther(); //其他流程控制
panelControl();//硅胶面板控制

tipsHandle();//提示信息处理
handleOutput40A();//40A板卡输出信号处理
handleOutput24B();//24B板卡输出信号处理
transmit2HMI();//发送给HMI信息
transmit2SiliconePanel();//发送给硅胶面板信息

END_PROGRAM

// Device/Application/parameterConfigure
PROGRAM parameterConfigure
VAR
	runOneTime:BOOL :=FALSE;
END_VAR

IF (NOT runOneTime) THEN
    systemStatus.softVersion:= 101;	//12位表示小版本，第3位表示大版本，其他高位保留
	IF NOT systemConfig.configFlag THEN	
	//systemConfig.dspDiaphragmPump:= 1;  //喷雾降尘泵配置，默认打开
	systemConfig.dspWaterPumpConnect:= 0;  //水泵离合器配置，默认关闭
	systemConfig.dspLowPressureSystem:=1;	//低压水路系统配置，默认打开
   	systemConfig.dspEngineStandardSpeed:=1450;	//标准速度配置
    systemConfig.dspEngineStrongSpeed:=1750;	//强力速度_配置_屏输入
    systemConfig.dspIncreaseStep:=50;	//加减转速_配置_屏输入
	systemConfig.dspWaterPumpOverSpeedAlarm:=1850;	//高压水泵超速警报_配置_屏输入
	systemConfig.dspWaterPumpOverSpeedStop:=1950; 	//高压水泵超速停机_配置_屏输入
	systemConfig.dspEngineIdlingSpeed:=850;	//发动机怠速_配置_屏输入
    systemConfig.dspSweeperSpeed:=0; //扫盘转速_配置_屏输入,默认高速
	systemConfig.dspAIModel:=0; //智能模式_配置_屏输入,默认关闭
	systemConfig.dspRoadCondition:=0;////路面情况_配置_屏输入,默认一般路面
	systemConfig.dspEngineMaxSpeed:=2500;	//发动机最高速_配置_屏输入
	systemConfig.configFlag:=TRUE;
	END_IF
	runOneTime:= TRUE;
END_IF

END_PROGRAM

// Device/Application/handleInput40A
PROGRAM handleInput40A
VAR
	ton1:TON; //总水阀接近开关滤波
	ton2:TON; //总水阀接近开关滤波
	ton3:TON; //吹净阀接近开关滤波
	ton4:TON; //吹净阀接近开关滤波
	ton5:TON; //后门接近开关滤波
	ton6:TON; //后门接近开关滤波
	ton7:TON; //左撑杆接近开关滤波
	ton8:TON; //左撑杆接近开关滤波
	ton9:TON; //右撑杆接近开关滤波
	ton10:TON; //右撑杆接近开关滤波
	ton11:TON; //水路卸荷阀接近开关滤波
	ton12:TON; //水路卸荷阀接近开关滤波
	ton13:TON; //污水箱高水位滤波
	ton14:TON; //液压油位低
END_VAR

       input40A.dumpsterPressure:= 625*(diDumpsterPressure-4000);  //垃圾箱负压(帕斯卡），4-20ma转换
	   input40A.suctionBucketPressure:= 625*(diSuctionBucketPressure-4000); //吸桶负压(帕斯卡），4-20ma转换
	   input40A.frontWaterTankPressure:= 1250*(diFrontWaterTankPressure-4000); //前水箱水压(帕斯卡），4-20ma转换
	   input40A.backWaterTankPressure:= 1250*(diBackWaterTankPressure-4000); //后水箱水压(帕斯卡），4-20ma转换
	   input40A.diaphragmPumpPressure:= diDiaphragmPumpPressure; //隔膜泵压力正常	   
	   ton14(IN:=diHydraulicOilLevel,PT:=T#5S,Q=>input40A.hydraulicOilLevel); //液压油位低,5s滤波
	   input40A.frontWaterTankWaterLevel:= diFrontWaterTankWaterLevel; //前水箱低水位,0-10k
	   input40A.backWaterTankWaterLevel:= diBackWaterTankWaterLevel; //后清水箱水位,0-10k
	   input40A.backup01:= diBackup01; //备用	   
	   ton13(IN:=diBilgeTankWaterLevel,PT:=T#6S,Q=>input40A.bilgeTankWaterLevel);//污水箱高水位,6s滤波
       //总水阀接近开关,1S滤波
	   ton1(IN:=diMainWateraValve,PT:=T#1S);
	   ton2(IN:=NOT diMainWateraValve,PT:=T#1S);
	   input40A.mainWateraValve:= (ton1.Q OR input40A.mainWateraValve) AND (NOT ton2.Q); 
	   //吹净阀接近开关,1S滤波
	   ton3(IN:=diCleanValve,PT:=T#1S);
	   ton4(IN:=NOT diCleanValve,PT:=T#1S);
	   input40A.cleanValve:= (ton3.Q OR input40A.cleanValve) AND (NOT ton4.Q); 
	   //后门接近开关,1S滤波
	   ton5(IN:=diBackDoor,PT:=T#1S);
	   ton6(IN:=NOT diBackDoor,PT:=T#1S);
	   input40A.backDoor:= (ton5.Q OR input40A.backDoor) AND (NOT ton6.Q);  
	   //左侧撑杆接近开关,1S滤波
	   ton7(IN:=diLeftRod,PT:=T#1S);
	   ton8(IN:=NOT diLeftRod,PT:=T#1S);
	   input40A.leftRod:= (ton7.Q OR input40A.leftRod) AND (NOT ton8.Q);
	   //右侧撑杆接近开关,1S滤波
	   ton9(IN:=diRightRod,PT:=T#1S);
	   ton10(IN:=NOT diRightRod,PT:=T#1S);
	   input40A.rightRod:= (ton9.Q OR input40A.rightRod) AND (NOT ton10.Q); 
	   //水路卸荷阀接近开关,1s滤波
	   ton11(IN:=diWaterUnloadValve,PT:=T#1S);
	   ton12(IN:=NOT diWaterUnloadValve,PT:=T#1S);
	   input40A.waterUnloadValve:= (ton11.Q OR input40A.waterUnloadValve) AND (NOT ton12.Q);

END_PROGRAM

// Device/Application/handleInput24B
PROGRAM handleInput24B
VAR
	ton1:TON; //回油过滤堵塞
	ton2:TON; //高压油滤堵塞
END_VAR

    ton1(IN:=diReturnOilFilterBlockUp,PT:=T#5S,Q=>input24B.returnOilFilterBlockUp); //回油过滤堵塞,5S滤波
	ton2(IN:=diHighPressureFilterBlockUp,PT:=T#5S,Q=>input24B.highPressureFilterBlockUp);  //高压油滤堵塞,5s滤波
	input24B.reverseCar:= diReverseCar; //倒车
	input24B.coolingTankWaterLevel:=diCoolingTankWaterLevel; //冷却水箱液位,0-10v信号,0.75-1.75水位正常，3.25-4.25V水位低，>4.5对电短路，<0.5开路对地
	input24B.waitingStartLamp:= diWaitingStartLamp; //等待启动灯
	input24B.alarmLamp:=diAlarmLamp; //警告故障灯
	input24B.stopEngineLamp:= diStopEngineLamp; //停机故障灯
	input24B.generatorWork:= diGeneratorWork; //发电机发电

END_PROGRAM

// Device/Application/receiveFromHMI
PROGRAM receiveFromHMI
VAR
	rcvCAN1: JCMC_Ctrl.CAN_RECEIVE;//触摸屏发送报文1，控制器CAN1接收，0x0C002A4F
	rcvCAN2: JCMC_Ctrl.CAN_RECEIVE;//触摸屏发送报文2，控制器CAN1接收，0x0C012A4F
	rcvCAN3: JCMC_Ctrl.CAN_RECEIVE;//触摸屏发送报文3，控制器CAN1接收，0x0C032A4F
	rcvCAN4: JCMC_Ctrl.CAN_RECEIVE;//触摸屏发送报文4，控制器CAN1接收，0x0C042A4F
	rcvCAN5: JCMC_Ctrl.CAN_RECEIVE;//触摸屏发送报文5，控制器CAN1接收，0x0C052A4F
	
	rcvBuf1:JCMC_Ctrl.CanMsgST;//0x0C002A4F报文数据
	rcvBuf2:JCMC_Ctrl.CanMsgST;//0x0C012A4F报文数据
	rcvBuf3:JCMC_Ctrl.CanMsgST;//0x0C032A4F报文数据
	rcvBuf4:JCMC_Ctrl.CanMsgST;//0x0C042A4F报文数据
	rcvBuf5:JCMC_Ctrl.CanMsgST;//0x0C052A4F报文数据
END_VAR

//JCMC_Ctrl.CAN_RECEIVE该功能块的作用，从控制器CAN缓存池里面取出等于设置ID号的数据，缓存池里面可以存32个ID号的数据，每个ID号的数据不大于3条，每执行一次该功能块，缓存池数据减少一条。
//触摸屏发送报文1，控制器CAN1接收，0x0C002A4F
rcvBuf1.ID:=16#0C002A4F;
rcvCAN1(CHANNEL:=1, CONFIG:=TRUE,CLEAR:=FALSE,ID:=rcvBuf1.ID);//CAN1,不清空缓存

IF (rcvCAN1.AVAILABLE>0)  THEN
	 rcvBuf1.Data:=rcvCAN1.DATA;
	 //解析0x0C002A4F报文数据
	dspSystemInput.dspAllWashSweep := rcvBuf1.Data[0].0;	//全洗扫_屏输入
	dspSystemInput.dspLeftWashSweep:= rcvBuf1.Data[0].1;	//左洗扫_屏输入
	dspSystemInput.dspRightWashSweep:= rcvBuf1.Data[0].2;	//右洗扫_屏输入
	dspSystemInput.dspAllSweep:= rcvBuf1.Data[0].3;	//全扫路_屏输入
	dspSystemInput.dspLeftSweep:= rcvBuf1.Data[0].4;	//左扫路_屏输入
	dspSystemInput.dspRightSweep:= rcvBuf1.Data[0].5;	//右扫路_屏输入
	dspSystemInput.dspAllWash:= rcvBuf1.Data[0].6;	//全清洗_屏输入
	dspSystemInput.dspLeftWash:= rcvBuf1.Data[0].7;	//左清洗_屏输入

	dspSystemInput.dspRightWash:= rcvBuf1.Data[1].0;	//右清洗_屏输入
	dspSystemInput.dspStopWash:= rcvBuf1.Data[1].1;	//停扫_屏输入
	dspSystemInput.dspEngineStart:= rcvBuf1.Data[1].2;	//发动机启动_屏输入
	dspSystemInput.dspEngineStop:= rcvBuf1.Data[1].3;	//发动机停止/运行_屏输入	
	dspSystemInput.dspSpeedUp:= rcvBuf1.Data[1].4;	//转速增加_屏输入
	dspSystemInput.dspSpeedDown:= rcvBuf1.Data[1].5;	//转速降低_屏输入
	dspSystemInput.dspStandardSpeed:= rcvBuf1.Data[1].6;	//标准速度_屏输入
	dspSystemInput.dspStrongSpeed:= rcvBuf1.Data[1].7;	//强力速度_屏输入

	dspSystemInput.dspTankDoorClose:= rcvBuf1.Data[2].0;	//垃圾箱门关_屏输入
	dspSystemInput.dspTankDoorOpen:= rcvBuf1.Data[2].1;	//垃圾箱门开_屏输入
	dspSystemInput.dspTankUp:= rcvBuf1.Data[2].2;	//垃圾箱体升_屏输入
	dspSystemInput.dspTankDown:= rcvBuf1.Data[2].3;	//垃圾箱体降_屏输入
	dspSystemInput.dspSelfClean:= rcvBuf1.Data[2].5;	//自洁_屏输入

	dspSystemInput.dspSweeperSpeedLow:=rcvBuf1.Data[3].0;	//扫盘低速_屏输入
	dspSystemInput.dspSweeperSpeedMiddle:=rcvBuf1.Data[3].1;	//扫盘中速_屏输入
	dspSystemInput.dspSweeperSpeedHigh:=rcvBuf1.Data[3].2;	//扫盘高速_屏输入
	dspSystemInput.dspLeftFlush:=rcvBuf1.Data[3].4;	//左角冲_屏输入
	dspSystemInput.dspRightFlush:=rcvBuf1.Data[3].5;	//右角冲_屏输入
	dspSystemInput.dspBackSpray:=rcvBuf1.Data[3].6;	//后喷雾_屏输入
	dspSystemInput.dspSprayGun:=rcvBuf1.Data[3].7;	//手持喷枪_屏输入

	dspSystemInput.dspDrainOffStart:=rcvBuf1.Data[4].0;	//排水启动_屏输入,目前该按钮属于未启动状态
	dspSystemInput.dspAutoDrainOff:=rcvBuf1.Data[4].1;	 //自动排水_屏输入	
	dspSystemInput.dspManualDrainOff:=rcvBuf1.Data[4].2;	//手动排水_屏输入	
	dspSystemInput.dspLeftSprayRodDrainOff:=rcvBuf1.Data[4].3;	//左喷杆排水_屏输入
	dspSystemInput.dspRightSprayRodDrainOff:=rcvBuf1.Data[4].4;	//右喷杆排水_屏输入
	dspSystemInput.dspAuxiliarySystemDrainOff:=rcvBuf1.Data[4].5;	//辅助排水_屏输入
	dspSystemInput.dspSelfCleanDrainOff:=rcvBuf1.Data[4].6;	//自洁排水_屏输入
	dspSystemInput.dspCentreSprayRodDrainOff:=rcvBuf1.Data[4].7;	//中喷杆排水_屏输入

	dspSystemInput.dspLeftFrontSprinkle:=rcvBuf1.Data[5].0;	//左前冲_屏输入
	dspSystemInput.dspRightFrontSprinkle:=rcvBuf1.Data[5].1;	//右前冲_屏输入
	dspSystemInput.dspLeftBackSprinkle:=rcvBuf1.Data[5].2;	//左后洒_屏输入
	dspSystemInput.dspRightBackSprinkle:=rcvBuf1.Data[5].3;	//右后洒_屏输入

	dspSystemInput.dspTestStart:=rcvBuf1.Data[6].0;	//功能测试_屏输入
	dspSystemInput.dspReplaceSweeper:=rcvBuf1.Data[6].1;	//更换扫刷_屏输入
	dspSystemInput.dspAIModel:=rcvBuf1.Data[6].2;	//智能模式_屏输入
	dspSystemInput.dspCleanRoad:=rcvBuf1.Data[6].3;	//清洁路面_屏输入
	dspSystemInput.dspNormalRoad:=rcvBuf1.Data[6].4;	//一般路面_屏输入
	dspSystemInput.dspDirtyRoad:=rcvBuf1.Data[6].5;	//污染路面_屏输入
END_IF 
//IF rcvCAN1.OVERFLOW = 1 THEN
//		rcvCAN1(CHANNEL:=1, CONFIG:=TRUE,CLEAR:=FALSE,ID:=rcvBuf1.ID);
//END_IF



//触摸屏发送报文2，控制器CAN1接收，0x0C012A4F
rcvBuf2.ID:=16#0C012A4F;
rcvCAN2(CHANNEL:=1, CONFIG:=TRUE,CLEAR:=FALSE,ID:=rcvBuf2.ID);//CAN1,不清空缓存

IF (rcvCAN2.AVAILABLE>0)  THEN
	 rcvBuf2.Data:=rcvCAN2.DATA;
	 //解析0x0C012A4F报文数据
 	dspTestInput.dspEngineDisconnectTest:=rcvBuf2.Data[0].0;	//副发分离_测试_屏输入
 
	dspTestInput.dspSweeperSpeedMiddleTest:=rcvBuf2.Data[1].0;	//扫盘中速_测试_屏输入
	dspTestInput.dspSweeperSpeedLowTest:=rcvBuf2.Data[1].1;	//扫盘低速_测试_屏输入
	dspTestInput.dspLeftSweeperRotateTest:=rcvBuf2.Data[1].2;	//左扫旋转_测试_屏输入
	dspTestInput.dspRightSweeperRotateTest:=rcvBuf2.Data[1].3;	//右扫旋转_测试_屏输入
	dspTestInput.dspAllSweeperRotateTest:=rcvBuf2.Data[1].4;	//全扫旋转_测试_屏输入
	dspTestInput.dspTankDownTest:=rcvBuf2.Data[1].5;	//箱体降_测试_屏输入
	dspTestInput.dspTankUpTest:=rcvBuf2.Data[1].6;	//箱体升_测试_屏输入
	dspTestInput.dspSuctionNozzleDownTest:=rcvBuf2.Data[1].7;	//吸嘴降_测试_屏输入

	dspTestInput.dspSuctionNozzleUpTest:=rcvBuf2.Data[2].0;	//吸嘴升_测试_屏输入
	dspTestInput.dspTankDoorOpenTest:=rcvBuf2.Data[2].1; //箱门开_测试_屏输入
	dspTestInput.dspTankDoorCloseTest:=rcvBuf2.Data[2].2;	//箱门关_测试_屏输入

	dspTestInput.dspLeftSweeperDownTest:=rcvBuf2.Data[3].0;	//左扫盘下放_测试_屏输入
	dspTestInput.dspLeftSweeperUpTest:=rcvBuf2.Data[3].1;	//左扫盘回收_测试_屏输入
	dspTestInput.dspRightSweeperDownTest:=rcvBuf2.Data[3].2;	//右扫盘下放_测试_屏输入
	dspTestInput.dspRightSweeperUpTest:=rcvBuf2.Data[3].3;	//右扫盘回收_测试_屏输入
	dspTestInput.dspLeftSprayRodSwingOutTest:=rcvBuf2.Data[3].4;	//左喷杆摆出_测试_屏输入
	dspTestInput.dspRightSprayRodSwingOutTest:=rcvBuf2.Data[3].5;	//右喷杆摆出_测试_屏输入
	dspTestInput.dspLeftSprayRodOpenTest:=rcvBuf2.Data[3].6;	//左喷杆喷水_测试_屏输入
	dspTestInput.dspRightSprayRodOpenTest:=rcvBuf2.Data[3].7;	//右喷杆喷水_测试_屏输入

	dspTestInput.dspCentreSprayRodOpenTest:=rcvBuf2.Data[4].0;	//中喷杆喷水_测试_屏输入
	dspTestInput.dspAuxiliaryValueTest:=rcvBuf2.Data[4].1;	//辅助球阀打开_测试_屏输入	
	dspTestInput.dspSelfCleanTest:=rcvBuf2.Data[4].2;	//自洁打开_测试_屏输入
	dspTestInput.dspWaterPumpConnectTest:=rcvBuf2.Data[4].3;//高压水泵啮合_测试_屏输入
	dspTestInput.dspDiaphragmPumpStartTest:=rcvBuf2.Data[4].4;	//喷雾降尘泵_测试_屏输入

	dspTestInput.dspConnectWaterValveTest:=rcvBuf2.Data[6].0;	//连通水阀_测试_屏输入
	dspTestInput.dspCloseFrontTankTest:=rcvBuf2.Data[6].1;	//前水箱水阀_测试_屏输入
	dspTestInput.dspCLoseBackTankTest:=rcvBuf2.Data[6].2;	//后水箱水阀_测试_屏输入
	dspTestInput.dspLeftFrontSprinkleTest:=rcvBuf2.Data[6].3;	//	左前冲_测试_屏输入
	dspTestInput.dspRightFrontSprinkleTest:=rcvBuf2.Data[6].4;	//	右前冲_测试_屏输入
	dspTestInput.dspLeftBackSprinkleTest:=rcvBuf2.Data[6].5;	//	左后洒_测试_屏输入
	dspTestInput.dspRightBackSprinkleTest:=rcvBuf2.Data[6].6;	//	右后洒_测试_屏输入
	dspTestInput.dspLeftSweeperSwingOutTest:=rcvBuf2.Data[6].7;	//左扫盘摆出_测试_屏输入
	
	dspTestInput.dspRightSweeperSwingOutTest:=rcvBuf2.Data[7].0;	//右扫盘摆出_测试_屏输入
END_IF 
//IF rcvCAN2.OVERFLOW = 1 THEN
//		rcvCAN2(CHANNEL:=1, CONFIG:=TRUE,CLEAR:=FALSE,ID:=rcvBuf2.ID);
//END_IF


	
//触摸屏发送报文3，控制器CAN1接收，0x0C032A4F
rcvBuf3.ID:=16#0C032A4F;
rcvCAN3(CHANNEL:=1, CONFIG:=TRUE,CLEAR:=FALSE,ID:=rcvBuf3.ID);//CAN1,不清空缓存

IF (rcvCAN3.AVAILABLE>0)  THEN
	 rcvBuf3.Data:=rcvCAN3.DATA;
	 //解析0x0C032A4F报文数据	
	systemConfig.dspIncreaseStep:=rcvBuf3.Data[4]+256*rcvBuf3.Data[5];	//加减转速_配置_屏输入
	//systemConfig.dspDiaphragmPump:=rcvBuf3.Data[6].0;	//喷雾降尘泵_配置_屏输入
	systemConfig.dspWaterPumpConnect:=rcvBuf3.Data[6].0;	//水泵离合器_配置_屏输入
	systemConfig.dspLowPressureSystem:=rcvBuf3.Data[6].1;	//低压水路系统_配置_屏输入	
	systemConfig.dspAIModel:=rcvBuf3.Data[6].2;	//智能模式_配置_屏输入
END_IF 
//IF rcvCAN3.OVERFLOW = 1 THEN
//		rcvCAN3(CHANNEL:=1, CONFIG:=TRUE,CLEAR:=FALSE,ID:=rcvBuf3.ID);
//END_IF



//触摸屏发送报文4，控制器CAN1接收，0x0C042A4F
rcvBuf4.ID:=16#0C042A4F;
rcvCAN4(CHANNEL:=1, CONFIG:=TRUE,CLEAR:=FALSE,ID:=rcvBuf4.ID);//CAN1,不清空缓存

IF (rcvCAN4.AVAILABLE>0)  THEN
	 rcvBuf4.Data:=rcvCAN4.DATA;
	 //解析0x0C042A4F报文数据
	systemConfig.dspEngineStandardSpeed:=(rcvBuf4.Data[0]+256*rcvBuf4.Data[1])/8;	//标准速度_配置_屏输入
	systemConfig.dspEngineStrongSpeed:=(rcvBuf4.Data[2]+256*rcvBuf4.Data[3])/8;	//强力速度_配置_屏输入
	systemConfig.dspSweeperSpeed:=rcvBuf4.Data[4]+256*rcvBuf4.Data[5]; //扫盘转速_配置_屏输入	
	systemConfig.dspRoadCondition:=rcvBuf4.Data[6]+256*rcvBuf4.Data[7];	//路面情况_配置_屏输入  
END_IF 
//IF rcvCAN4.OVERFLOW = 1 THEN
//		rcvCAN4(CHANNEL:=1, CONFIG:=TRUE,CLEAR:=FALSE,ID:=rcvBuf4.ID);
//END_IF	
	
  

//触摸屏发送报文5，控制器CAN1接收，0x0C052A4F
rcvBuf5.ID:=16#0C052A4F;
rcvCAN5(CHANNEL:=1, CONFIG:=TRUE,CLEAR:=FALSE,ID:=rcvBuf5.ID);//CAN1,不清空缓存

IF (rcvCAN5.AVAILABLE>0)  THEN
	 rcvBuf5.Data:=rcvCAN5.DATA;
	 //解析0x0C052A4F报文数据
	systemConfig.dspWaterPumpOverSpeedAlarm:=(rcvBuf5.Data[0]+256*rcvBuf5.Data[1])/8;	//高压水泵超速警报_配置_屏输入
	systemConfig.dspWaterPumpOverSpeedStop:=(rcvBuf5.Data[2]+256*rcvBuf5.Data[3])/8; 	//高压水泵超速停机_配置_屏输入
	systemConfig.dspEngineMaxSpeed:=(rcvBuf5.Data[4]+256*rcvBuf5.Data[5])/8;	//发动机最高速_配置_屏输入
	systemConfig.dspEngineIdlingSpeed:=(rcvBuf5.Data[6]+256*rcvBuf5.Data[7])/8;	//发动机怠速_配置_屏输入
END_IF 
//IF rcvCAN5.OVERFLOW = 1 THEN
//		rcvCAN5(CHANNEL:=1, CONFIG:=TRUE,CLEAR:=FALSE,ID:=rcvBuf5.ID);
//END_IF

END_PROGRAM

// Device/Application/receiveFromEngineECM
PROGRAM receiveFromEngineECM
VAR
	rcvCAN1: JCMC_Ctrl.CAN_RECEIVE;//副发ECM发送报文1，控制器CAN1接收，0x0CF00400
	rcvCAN2: JCMC_Ctrl.CAN_RECEIVE;//副发ECM发送报文2，控制器CAN1接收，0x18FEEE00
	rcvCAN3: JCMC_Ctrl.CAN_RECEIVE;//副发ECM发送报文3，控制器CAN1接收，0x18FEEF00
	rcvCAN4: JCMC_Ctrl.CAN_RECEIVE;//副发ECM发送报文4，控制器CAN1接收，0x18FEE500
	rcvCAN5: JCMC_Ctrl.CAN_RECEIVE;//副发ECM发送报文5，控制器CAN1接收，0x18FECA00
	rcvCAN6: JCMC_Ctrl.CAN_RECEIVE;//副发ECM发送报文6，控制器CAN1接收，0x18ECFF00
	rcvCAN7: JCMC_Ctrl.CAN_RECEIVE;//副发ECM发送报文7，控制器CAN1接收，0x18EBFF00
	
	rcvBuf1:JCMC_Ctrl.CanMsgST;//0x0CF00400报文数据
	rcvBuf2:JCMC_Ctrl.CanMsgST;//0x18FEEE00报文数据
	rcvBuf3:JCMC_Ctrl.CanMsgST;//0x18FEEF00报文数据
	rcvBuf4:JCMC_Ctrl.CanMsgST;//0x18FEE500报文数据
	rcvBuf5:JCMC_Ctrl.CanMsgST;//0x18FECA00报文数据
	rcvBuf6:JCMC_Ctrl.CanMsgST;//0x18ECFF00报文数据
	rcvBuf7:JCMC_Ctrl.CanMsgST;//0x18EBFF00报文数据
	
	multipacketParams: MultipacketParameter;//多包传输参数
	packageNum:WORD;//报文编号
	counter:word;//计数器
	
END_VAR

//JCMC_Ctrl.CAN_RECEIVE该功能块的作用，从控制器CAN缓存池里面取出等于设置ID号的数据，缓存池里面可以存32个ID号的数据，每个ID号的数据不大于3条，每执行一次该功能块，缓存池数据减少一条。
//副发ECM发送报文1，控制器CAN1接收，0x0CF00400
rcvBuf1.ID:=16#0CF00400;
rcvCAN1(CHANNEL:=1, CONFIG:=TRUE,CLEAR:=FALSE,ID:=rcvBuf1.ID);//CAN1,不清空缓存

IF (rcvCAN1.AVAILABLE>0)  THEN
	 rcvBuf1.Data:=rcvCAN1.DATA;
	 //解析0x0CF00400报文数据,获取副发动机转速
     systemStatus.engineRealSpeed:=(rcvBuf1.Data[3]+256*rcvBuf1.Data[4])/8;	//副发动机转速r/m
	 
END_IF 
//IF rcvCAN1.OVERFLOW = 1 THEN
//		rcvCAN1(CHANNEL:=1, CONFIG:=TRUE,CLEAR:=FALSE,ID:=rcvBuf1.ID);
//END_IF



//副发ECM发送报文2，控制器CAN1接收，0x18FEEE00
rcvBuf2.ID:=16#18FEEE00;
rcvCAN2(CHANNEL:=1, CONFIG:=TRUE,CLEAR:=FALSE,ID:=rcvBuf2.ID);//CAN1,不清空缓存

IF (rcvCAN2.AVAILABLE>0)  THEN
	 rcvBuf2.Data:=rcvCAN2.DATA;
	 //0x18FEEE00报文数据,获取冷却液温度
     systemStatus.engineCoolingTemperature:=BYTE_TO_SINT(rcvBuf2.Data[0]-40); //副发水温
END_IF 
//IF rcvCAN2.OVERFLOW = 1 THEN
//		rcvCAN2(CHANNEL:=1, CONFIG:=TRUE,CLEAR:=FALSE,ID:=rcvBuf2.ID);
//END_IF




//副发ECM发送报文3，控制器CAN1接收，0x18FEEF00
rcvBuf3.ID:=16#18FEEF00;
rcvCAN3(CHANNEL:=1, CONFIG:=TRUE,CLEAR:=FALSE,ID:=rcvBuf3.ID);//CAN1,不清空缓存

IF (rcvCAN3.AVAILABLE>0)  THEN
	 rcvBuf3.Data:=rcvCAN3.DATA;
	 //0x18FEEF00报文数据,获取发动机机油压力
     systemStatus.engineOilPressure:=4*rcvBuf3.Data[3]; //副发油压
END_IF 
//IF rcvCAN3.OVERFLOW = 1 THEN
//		rcvCAN3(CHANNEL:=1, CONFIG:=TRUE,CLEAR:=FALSE,ID:=rcvBuf3.ID);
//END_IF



//副发ECM发送报文4，控制器CAN1接收，0x18FEE500
rcvBuf4.ID:=16#18FEE500;
rcvCAN4(CHANNEL:=1, CONFIG:=TRUE,CLEAR:=FALSE,ID:=rcvBuf4.ID);//CAN1,不清空缓存

IF (rcvCAN4.AVAILABLE>0)  THEN
	 rcvBuf4.Data:=rcvCAN4.DATA;
	 //0x18FEE500报文数据,获取发动机工作时间
systemStatus.engineWorkTime:=rcvBuf4.Data[0]+256*rcvBuf4.Data[1]+256*256*rcvBuf4.Data[2]+256*256*256*rcvBuf4.Data[3];//由于该数据只是转发给触摸屏，在此不做进一步解析
END_IF 
//IF rcvCAN4.OVERFLOW = 1 THEN
//		rcvCAN4(CHANNEL:=1, CONFIG:=TRUE,CLEAR:=FALSE,ID:=rcvBuf4.ID);
//END_IF



//副发ECM发送报文5，控制器CAN1接收，0x18FECA00
rcvBuf5.ID:=16#18FECA00;
rcvCAN5(CHANNEL:=1, CONFIG:=TRUE,CLEAR:=FALSE,ID:=rcvBuf5.ID);//CAN1,不清空缓存

IF (rcvCAN5.AVAILABLE>0)  THEN
	 rcvBuf5.Data:=rcvCAN5.DATA;
	 //0x18FECA00报文数据,获取故障SPN码
     systemStatus.engineFaultSPN:= rcvBuf5.Data[2]+256*rcvBuf5.Data[3]+ 256*256*(SHR(rcvBuf5.Data[4],5));
END_IF 
//IF rcvCAN5.OVERFLOW = 1 THEN
//		rcvCAN5(CHANNEL:=1, CONFIG:=TRUE,CLEAR:=FALSE,ID:=rcvBuf5.ID);
//END_IF



//副发ECM发送报文6，控制器CAN1接收，0x18ECFF00
rcvBuf6.ID:=16#18ECFF00;
rcvCAN6(CHANNEL:=1, CONFIG:=TRUE,CLEAR:=TRUE,ID:=rcvBuf6.ID);//CAN1,清空缓存

IF (rcvCAN6.AVAILABLE>0)  THEN
	 rcvBuf6.Data:=rcvCAN6.DATA;
	 //0x18ECFF00报文数据,获取多包传输参数
	multipacketParams.byteTotalNum:= rcvBuf6.Data[1]+256*rcvBuf6.Data[2];//字节数
	multipacketParams.packageTotalNum:=rcvBuf6.Data[3];//数据包数
	multipacketParams.PGN:=rcvBuf6.Data[5]+256*rcvBuf6.Data[6]+256*256*rcvBuf6.Data[7];//获取PGN
	FOR counter:=1 TO 80 BY 1 DO   //清空data
		multipacketParams.Data[counter-1]:= 0;
	END_FOR
END_IF 
//IF rcvCAN6.OVERFLOW = 1 THEN
//		rcvCAN6(CHANNEL:=1, CONFIG:=TRUE,CLEAR:=FALSE,ID:=rcvBuf6.ID);
//END_IF



//副发ECM发送报文7，控制器CAN1接收，0x18EBFF00
rcvBuf7.ID:=16#18EBFF00;
rcvCAN7(CHANNEL:=1, CONFIG:=TRUE,CLEAR:=FALSE,ID:=rcvBuf7.ID);//CAN1,不清空缓存

IF (rcvCAN7.AVAILABLE>0)  THEN
	 rcvBuf7.Data:=rcvCAN7.DATA;
	 //解析0x18EBFF00报文数据
	packageNum:= rcvBuf7.Data[0];
	
END_IF 
//IF rcvCAN7.OVERFLOW = 1 THEN
//		rcvCAN7(CHANNEL:=1, CONFIG:=TRUE,CLEAR:=FALSE,ID:=rcvBuf7.ID);
//END_IF

END_PROGRAM

// Device/Application/receiveFromECU
PROGRAM receiveFromECU
VAR
	rcvCAN1: JCMC_Ctrl.CAN_RECEIVE;//底盘发送报文1，控制器CAN2接收，0x0CF00400
	rcvCAN2: JCMC_Ctrl.CAN_RECEIVE;//底盘发送报文2，控制器CAN2接收，0x0CFE6CEE
	rcvCAN3: JCMC_Ctrl.CAN_RECEIVE;//底盘发送报文3，控制器CAN2接收，0x18FEC1EE
	
	rcvBuf1:JCMC_Ctrl.CanMsgST;//0x0CF00400报文数据
	rcvBuf2:JCMC_Ctrl.CanMsgST;//0x0CFE6CEE报文数据
	rcvBuf3:JCMC_Ctrl.CanMsgST;//0x18FEC1EE报文数据

END_VAR

//JCMC_Ctrl.CAN_RECEIVE该功能块的作用，从控制器CAN缓存池里面取出等于设置ID号的数据，缓存池里面可以存32个ID号的数据，每个ID号的数据不大于3条，每执行一次该功能块，缓存池数据减少一条。
//底盘发送报文1，控制器CAN2接收，0x0CF00400
rcvBuf1.ID:=16#0CF00400;
rcvCAN1(CHANNEL:=2, CONFIG:=TRUE,CLEAR:=FALSE,ID:=rcvBuf1.ID);//CAN1,不清空缓存

IF (rcvCAN1.AVAILABLE>0)  THEN
	 rcvBuf1.Data:=rcvCAN1.DATA;
END_IF 
//IF rcvCAN1.OVERFLOW = 1 THEN
//		rcvCAN1(CHANNEL:=2, CONFIG:=TRUE,CLEAR:=FALSE,ID:=rcvBuf1.ID);
//END_IF

//解析0x0CF00400报文数据,获取底盘发动机转速
systemStatus.vehicleEngineSpeed:=(rcvBuf1.Data[3]+256*rcvBuf1.Data[4])/8;	//底盘发动机转速r/m

//底盘发送报文2，控制器CAN2接收，0x0CFE6CEE
rcvBuf2.ID:=16#0CFE6CEE;
rcvCAN2(CHANNEL:=2, CONFIG:=TRUE,CLEAR:=FALSE,ID:=rcvBuf2.ID);//CAN1,不清空缓存

IF (rcvCAN2.AVAILABLE>0)  THEN
	 rcvBuf2.Data:=rcvCAN2.DATA;
END_IF 
//IF rcvCAN2.OVERFLOW = 1 THEN
//		rcvCAN2(CHANNEL:=2, CONFIG:=TRUE,CLEAR:=FALSE,ID:=rcvBuf2.ID);
//END_IF

//解析0x0CFE6CEE报文数据,获取车速
systemStatus.vehicleSpeed:=(rcvBuf2.Data[6]+256*rcvBuf2.Data[7])/256; //车速km/h

//底盘发送报文3，控制器CAN2接收，0x18FEC1EE
rcvBuf3.ID:=16#18FEC1EE;
rcvCAN3(CHANNEL:=2, CONFIG:=TRUE,CLEAR:=FALSE,ID:=rcvBuf3.ID);//CAN1,不清空缓存

IF (rcvCAN3.AVAILABLE>0)  THEN
	 rcvBuf3.Data:=rcvCAN3.DATA;
END_IF 
IF rcvCAN3.OVERFLOW = 1 THEN
		rcvCAN3(CHANNEL:=2, CONFIG:=TRUE,CLEAR:=FALSE,ID:=rcvBuf3.ID);
END_IF

//解析0x18FEC1EE报文数据,获取行驶里程
systemStatus.distance:= 5*(rcvBuf3.Data[0]+256*rcvBuf3.Data[1]+256*256*rcvBuf3.Data[2]+256*256*256*rcvBuf3.Data[3]);//行驶里程m

END_PROGRAM

// Device/Application/receiveFromSiliconePanel
PROGRAM receiveFromSiliconePanel
VAR
	rcvCAN1: JCMC_Ctrl.CAN_RECEIVE;//硅胶面板发送报文1，控制器CAN1接收，0x0C112AF0
	rcvBuf1:JCMC_Ctrl.CanMsgST;//0x0C112AF0报文数据
END_VAR

//JCMC_Ctrl.CAN_RECEIVE该功能块的作用，从控制器CAN缓存池里面取出等于设置ID号的数据，缓存池里面可以存32个ID号的数据，每个ID号的数据不大于3条，每执行一次该功能块，缓存池数据减少一条。
//硅胶面板发送报文1，控制器CAN1接收，0x0C112AF0
rcvBuf1.ID:=16#0C112AF0;
rcvCAN1(CHANNEL:=1, CONFIG:=TRUE,CLEAR:=FALSE,ID:=rcvBuf1.ID);//CAN1,不清空缓存

IF (rcvCAN1.AVAILABLE>0)  THEN
	 rcvBuf1.Data:=rcvCAN1.DATA;
	 //解析0x0C112AF0报文数据
	panelInput.tankDoorOpen:=rcvBuf1.Data[0].0;	//垃圾箱门开_硅胶面板输入
	panelInput.tankDoorClose:=rcvBuf1.Data[0].2;	//垃圾箱门关_硅胶面板输入
	panelInput.tankUp:=rcvBuf1.Data[0].4;	//垃圾箱体升_硅胶面板输入
	panelInput.tankDown:=rcvBuf1.Data[0].6;	//垃圾箱体降_硅胶面板输入

	panelInput.leftSweeperUpAndIn:=rcvBuf1.Data[1].0;	//左扫盘升_硅胶面板输入
	panelInput.leftSweeperOutAndDown:=rcvBuf1.Data[1].2;	//左扫盘下放_硅胶面板输入
	panelInput.rightSweeperUpAndIn:=rcvBuf1.Data[1].4;	//右扫盘升_硅胶面板输入
	panelInput.rightSweeperOutAndDown:=rcvBuf1.Data[1].6;	//右扫盘下放_硅胶面板输入

	panelInput.suctionNozzleUp:=rcvBuf1.Data[2].0;	//吸嘴升_硅胶面板输入
	panelInput.suctionNozzleDown:=rcvBuf1.Data[2].2;	//吸嘴降_测试_硅胶面板输入
	panelInput.selfClean:=rcvBuf1.Data[2].4;	//自洁打开_硅胶面板输入
	panelInput.sprayGun:=rcvBuf1.Data[2].6;	//手持喷枪_硅胶面板输入

	panelInput.sprayRodOutOrIn:=rcvBuf1.Data[3].0;  //喷杆伸缩_硅胶面板输入
	panelInput.backupMotor:=rcvBuf1.Data[3].2; //备用动力_硅胶面板输入
	panelInput.workLamp:=rcvBuf1.Data[3].4; //工作灯_硅胶面板输入
	panelInput.backlight:=rcvBuf1.Data[3].6; //背光灯_硅胶面板输入
END_IF 
//IF rcvCAN1.OVERFLOW = 1 THEN
//		rcvCAN1(CHANNEL:=1, CONFIG:=TRUE,CLEAR:=FALSE,ID:=rcvBuf1.ID);
//END_IF

END_PROGRAM

// Device/Application/faultHandle
PROGRAM faultHandle
VAR
	ton1:TON; //水路卸荷阀定时器
	ton2:TON; //水路卸荷阀定时器
	ton3:TON; //高压水泵超速报警定时器
	ton4:TON; //高压水泵超速停机定时器
	ton5:TON; //喷雾降尘泵定时器
	tp1:TP; //倒车上升沿触发，保持1S
	tp2:TP; //污水满上升沿触发,保持1S
	
END_VAR

    faultST.alarmLamp:=input24B.waitingStartLamp; //发动机警告故障
    faultST.stopEngineLamp:=input24B.stopEngineLamp;   //发动机停机故障
	//冷却水箱液位低,3.25-4.25V水位低
	IF (input24B.coolingTankWaterLevel>3250 AND input24B.coolingTankWaterLevel<4250) THEN		
		faultST.coolingTankWaterLevelLow:=TRUE;
		ELSE
			faultST.coolingTankWaterLevelLow:=FALSE;
	END_IF
	
	//水路卸荷阀未关闭
	ton1(IN:= ((NOT output24B.waterUnloadValveOpen) AND (NOT input40A.waterUnloadValve)),PT:=T#7S);	
	faultST.waterUnloadValveNotClose:=ton1.Q;	
	//水路卸荷阀未打开
	ton2(IN:= (output24B.waterUnloadValveOpen AND  input40A.waterUnloadValve),PT:=T#7S);	
	faultST.waterUnloadValveNotOpen:=ton2.Q;		
	faultST.bilgeTankFull:=input40A.bilgeTankWaterLevel;	//污水满
	faultST.returnOilFilterBlockUp:=input24B.returnOilFilterBlockUp;	//回油过滤堵塞
	faultST.hHighPressureFilterBlockUp:=input24B.highPressureFilterBlockUp;	//高压油滤堵塞
	faultST.hydraulicOilLevelLow:=input40A.hydraulicOilLevel;	//液压油位低
	//前水箱缺水,电阻大于8000欧姆认为缺水
	IF input40A.frontWaterTankWaterLevel> 8000 THEN
		faultST.frontTankWaterLevelLow:=TRUE;
		ELSE
		faultSt.frontTankWaterLevelLow:=FALSE;
	END_IF	
    //后水箱缺水,电阻大于8000欧姆认为缺水
    IF input40A.backWaterTankWaterLevel > 8000 THEN        	
	     faultST.backTankWaterLevelLow:=TRUE;
       ELSE 
    	faultST.backTankWaterLevelLow:=FALSE;
	END_IF
	tp1(IN:=(input24B.reverseCar AND systemStatus.systemWork),PT:=T#1S,Q=>faultST.reverseCarStop);	//倒车故障停机
	tp2(IN:=(input40A.bilgeTankWaterLevel AND systemStatus.systemWork),PT:=T#1S,Q=>faultST.waterFullStop);//污水满故障停机	
	//高压水泵超速报警,大于系统配置的超速报警值时
	ton3(IN:= ((systemStatus.engineRealSpeed > systemconfig.dspWaterPumpOverSpeedAlarm) AND output40A.waterPumpConnect ),PT:=T#5S);
	faultST.highPressurePumpOverSpeedAlarm:=ton3.Q;	
	//高压水泵超速停止,大于系统配置的超速停机值时
	ton4(IN:= ((systemStatus.engineRealSpeed > systemconfig.dspWaterPumpOverSpeedStop) AND output40A.waterPumpConnect ),PT:=T#3S);
	faultST.highPressurePumpOverSpeedStop:=ton4.Q;	
	//喷雾降尘泵故障,工作压力不正常时
	ton5(IN:=(NOT input40A.diaphragmPumpPressure AND output40A.diaphragmPumpStart),PT:=T#10S);	
	faultST.diaphragmPumpPressure:=ton5.Q;

END_PROGRAM

// Device/Application/engineControl
PROGRAM engineControl
VAR
	rTrigger1:R_TRIG;//发动机运行/停止_屏输入上升沿触发
	fTrigger1:F_TRIG;//钥匙开关运行/停止下降沿触发
	ton1:TON;//启动持续时间限定定时器
	ton2:TON;//启动延时定时器
	ton3:TON;//水泵离合器延时定时器
	tp1:TP;//离合器延时啮合定时器1
	tp2:TP;//离合器延时啮合定时器2
	engineStartTemp:BOOL;//发动机启动中间变量
	waterPumpWorkCondition :BOOL; //水泵啮合限定条件
	
END_VAR

//高压水泵啮合限定条件，吹净球阀关闭，总水阀打开，没有水路卸荷阀未打开故障,没有缺水故障，没有超速故障
 //waterPumpWorkCondition:= input40A.cleanValve AND input40A.mainWateraValve AND (NOT faultST.waterUnloadValveNotOpen)
//	   AND (NOT faultST.frontTankWaterLevelLow) AND (NOT faultST.backTankWaterLevelLow) AND (NOT faultST.highPressurePumpOverSpeedStop);
	   
rTrigger1(CLK:=dspSystemInput.dspEngineStop);
//控制钥匙开关运行/停止档位置
IF rTrigger1.Q THEN
	systemStatus.keyRunPosition:= systemStatus.keyRunPosition;
END_IF

//发动机启动控制，必须在运行档位，如果按住启动触发时间超过25S,断开启动，发动机运转正常后，断开启动
ton1(IN:= dspSystemInput.dspEngineStart AND systemStatus.keyRunPosition,PT:=T#25S);
engineStartTemp:= dspSystemInput.dspEngineStart AND systemStatus.keyRunPosition AND (NOT systemStatus.engineWork) AND (NOT ton1.Q) AND (NOT dspSystemInput.dspEngineStop);
//启动触发3S后启动马达得电
ton2(IN:=engineStartTemp,PT:=T#3S);
systemStatus.engineStart := ton2.Q;

//启动触发后12S后，水泵离合器啮合操作（水泵离合器必须静止啮合）
//ton3(IN:=engineStartTemp,PT:=T#12S);
//systemStatus.waterPumpConnect:=ton3.Q AND waterPumpWorkCondition;

//启动触发15s内副发离合器分离
tp1(IN:= engineStartTemp,PT:=T#15S);
//发动机停机触发30内副发离合器分离
fTrigger1(CLK:=systemStatus.keyRunPosition);
tp2(IN:=fTrigger1.Q,PT:=T#30S);
systemStatus.engineDisconect:= tp1.Q  OR (tp2.Q  AND (NOT engineStartTemp));

END_PROGRAM

// Device/Application/functionTest
PROGRAM functionTest
VAR
	temp01:BOOL;//临时状态
	rTrigger1:R_TRIG;//副发分离_测试_上升沿触发器
	rTrigger2:R_TRIG;//连通水阀_测试_上升沿触发器
	rTrigger3:R_TRIG;//前水箱水阀_测试_上升沿触发器
	rTrigger4:R_TRIG;//后水箱水阀_测试_上升沿触发器
	rTrigger5:R_TRIG;//扫盘低速_测试_上升沿触发器
	rTrigger6:R_TRIG;//扫盘中速_测试_上升沿触发器
	rTrigger7:R_TRIG;//左扫旋转_测试_上升沿触发器
	rTrigger8:R_TRIG;//右扫旋转_测试_上升沿触发器
	rTrigger9:R_TRIG;//全扫旋转_测试_上升沿触发器
	rTrigger10:R_TRIG;//箱体降_测试_上升沿触发器
	rTrigger11:R_TRIG;//箱体升_测试_上升沿触发器
	rTrigger12:R_TRIG;//吸嘴降_测试_上升沿触发器
	rTrigger13:R_TRIG;//吸嘴升_测试_上升沿触发器
	rTrigger14:R_TRIG;//箱门开_测试_上升沿触发器
	rTrigger15:R_TRIG;//箱门关_测试_上升沿触发器
	rTrigger16:R_TRIG;//左扫盘下放_测试_上升沿触发器
	rTrigger17:R_TRIG;//左扫盘回收_测试_上升沿触发器
	rTrigger18:R_TRIG;//右扫盘下放_测试_上升沿触发器
	rTrigger19:R_TRIG;//右扫盘回收_测试_上升沿触发器
	rTrigger20:R_TRIG;//左扫盘摆出_测试_上升沿触发器
	rTrigger21:R_TRIG;//右扫盘摆出_测试_上升沿触发器
	rTrigger22:R_TRIG;//左喷杆摆出_测试_上升沿触发器
	rTrigger23:R_TRIG;//右喷杆摆出_测试_上升沿触发器
	rTrigger24:R_TRIG;//左喷杆喷水_测试_上升沿触发器
	rTrigger25:R_TRIG;//右喷杆喷水_测试_上升沿触发器
	rTrigger26:R_TRIG;//中喷杆喷水_测试_上升沿触发器
	rTrigger27:R_TRIG;//辅助球阀打开_测试_上升沿触发器
	rTrigger28:R_TRIG;//自洁打开_测试_上升沿触发器
	rTrigger29:R_TRIG;//高压水泵啮合_测试_上升沿触发器
	rTrigger30:R_TRIG;//喷雾降尘泵_测试_上升沿触发器
	rTrigger31:R_TRIG;//左前冲_测试_上升沿触发器
	rTrigger32:R_TRIG;//右前冲_测试_上升沿触发器
	rTrigger33:R_TRIG;//左后洒_测试_上升沿触发器
	rTrigger34:R_TRIG;//右后洒_测试_上升沿触发器
	ton1:TON; //高压水泵定时器
	ton2:TON; //喷雾降尘泵定时器

END_VAR

//副发动机分离测试
rTrigger1(CLK:=dspTestInput.dspEngineDisconnectTest);
temp01:=ctlTestFlag.ctlEngineDisconnectTest;
(*IF ( rTrigger1.Q  AND systemStatus.engineWork AND (NOT temp01) ) THEN
	ctlTestFlag.ctlEngineDisconnectTest:= TRUE;
END_IF
IF ( rTrigger1.Q  AND systemStatus.engineWork AND  temp01 ) THEN
	ctlTestFlag.ctlEngineDisconnectTest:= FALSE;
END_IF *)
IF (rTrigger1.Q  AND systemStatus.engineWork) THEN
	 ctlTestFlag.ctlEngineDisconnectTest:= NOT ctlTestFlag.ctlEngineDisconnectTest;
END_IF
//连通水阀测试
rTrigger2(CLK:=dspTestInput.dspConnectWaterValveTest);
IF ( rTrigger2.Q ) THEN
	ctlTestFlag.ctlConnectWaterValveTest := NOT ctlTestFlag.ctlConnectWaterValveTest;
END_IF
//前水箱水阀测试
rTrigger3(CLK:=dspTestInput.dspCloseFrontTankTest);
IF ( rTrigger3.Q) THEN
	ctlTestFlag.ctlCloseFrontTankTest:= NOT ctlTestFlag.ctlCloseFrontTankTest;
END_IF
//后水箱水阀测试
rTrigger4(CLK:=dspTestInput.dspCLoseBackTankTest);
IF (rTrigger4.Q) THEN
	ctlTestFlag.ctlCLoseBackTankTest:= NOT ctlTestFlag.ctlCLoseBackTankTest;
END_IF
//扫盘低速测试
rTrigger5(CLK:=dspTestInput.dspSweeperSpeedLowTest);
IF (rTrigger5.Q ) THEN
	ctlTestFlag.ctlSweeperSpeedLowTest:= NOT ctlTestFlag.ctlSweeperSpeedLowTest; 
	IF ctlTestFlag.ctlSweeperSpeedLowTest THEN
	ctlTestFlag.ctlSweeperSpeedMiddleTest:= FALSE;
	END_IF
END_IF
//扫盘中速测试
rTrigger6(CLK:=dspTestInput.dspSweeperSpeedMiddleTest);
IF rTrigger6.Q THEN
	ctlTestFlag.ctlSweeperSpeedMiddleTest:= NOT ctlTestFlag.ctlSweeperSpeedMiddleTest;
	IF ctlTestFlag.ctlSweeperSpeedMiddleTest THEN
	ctlTestFlag.ctlSweeperSpeedLowTest:= FALSE; 
	END_IF
END_IF
//左扫旋转测试
rTrigger7(CLK:=dspTestInput.dspLeftSweeperRotateTest);
IF rTrigger7.Q THEN
	ctlTestFlag.ctlLeftSweeperRotateTest:= NOT ctlTestFlag.ctlLeftSweeperRotateTest;
	IF ctlTestFlag.ctlLeftSweeperRotateTest THEN
	  ctlTestFlag.ctlAllSweeperRotateTest:= FALSE;
	  ctlTestFlag.ctlRightSweeperRotateTest:= FALSE;
	END_IF
END_IF
//右扫旋转测试
rTrigger8(CLK:=dspTestInput.dspRightSweeperRotateTest);
IF rTrigger8.Q  THEN
	ctlTestFlag.ctlRightSweeperRotateTest:= NOT ctlTestFlag.ctlRightSweeperRotateTest;
	IF ctlTestFlag.ctlRightSweeperRotateTest THEN
		ctlTestFlag.ctlAllSweeperRotateTest:= FALSE;
		ctlTestFlag.ctlLeftSweeperRotateTest:= FALSE;
	END_IF
END_IF
//全扫旋转测试
rTrigger9(CLK:=dspTestInput.dspAllSweeperRotateTest);
IF rTrigger9.Q THEN
	ctlTestFlag.ctlAllSweeperRotateTest:= NOT ctlTestFlag.ctlAllSweeperRotateTest;
	IF ctlTestFlag.ctlAllSweeperRotateTest THEN
		ctlTestFlag.ctlLeftSweeperRotateTest:= FALSE;
		ctlTestFlag.ctlRightSweeperRotateTest:= FALSE;
	END_IF
END_IF
//箱体降测试,撑杆需放下
ctlTestFlag.ctlTankDownTest:= dspTestInput.dspTankDownTest AND input40A.leftRod AND input40A.rightRod AND (NOT dspTestInput.dspTankUpTest);
//箱体升测试
ctlTestFlag.ctlTankUpTest := dspTestInput.dspTankUpTest AND (NOT dspTestInput.dspTankDownTest);
//吸嘴降测试
ctlTestFlag.ctlSuctionNozzleDownTest:= dspTestInput.dspSuctionNozzleDownTest AND (NOT systemStatus.systemWork ) AND (NOT dspTestInput.dspSuctionNozzleUpTest);
//吸嘴升测试‘
ctlTestFlag.ctlSuctionNozzleUpTest := dspTestInput.dspSuctionNozzleUpTest AND (NOT systemStatus.systemWork ) AND (NOT dspTestInput.dspSuctionNozzleDownTest);
//箱门开测试
ctlTestFlag.ctlTankDoorOpenTest := dspTestInput.dspTankDoorOpenTest AND (NOT dspTestInput.dspTankDoorCloseTest);
//箱门关测试
ctlTestFlag.ctlTankDoorCloseTest := dspTestInput.dspTankDoorCloseTest AND (NOT dspTestInput.dspTankDoorOpenTest);
//左扫盘下放测试
ctlTestFlag.ctlLeftSweeperDownTest := dspTestInput.dspLeftSweeperDownTest AND (NOT dspTestInput.dspLeftSweeperUpTest);
//左扫盘回收测试
ctlTestFlag.ctlRightSweeperUpTest := dspTestInput.dspLeftSweeperUpTest AND (NOT dspTestInput.dspLeftSweeperDownTest);
//右扫盘下放测试
ctlTestFlag.ctlRightSweeperDownTest:= dspTestInput.dspRightSweeperDownTest AND (NOT dspTestInput.dspRightSweeperDownTest);
//右扫盘回收测试
ctlTestFlag.ctlRightSweeperUpTest := dspTestInput.dspRightSweeperDownTest AND (NOT dspTestInput.dspRightSweeperDownTest);
//左扫盘摆出测试
rTrigger20(CLK:=dspTestInput.dspLeftSweeperSwingOutTest);
IF rTrigger20.Q THEN
	ctlTestFlag.ctlLeftSweeperSwingOutTest:= NOT ctlTestFlag.ctlLeftSweeperSwingOutTest;
END_IF
//右扫盘摆出测试
rTrigger21(CLK:=dspTestInput.dspRightSweeperSwingOutTest);
IF rTrigger21.Q THEN
	ctlTestFlag.ctlRightSweeperSwingOutTest := NOT ctlTestFlag.ctlRightSweeperSwingOutTest;
END_IF
//左喷杆摆出测试,与硅胶面板的喷杆伸缩按钮互锁
rTrigger22(CLK:=dspTestInput.dspLeftSprayRodSwingOutTest);
IF rTrigger22.Q THEN
	IF ctlTestFlag.ctlLeftSprayRodSwingOutTest THEN 
		ctlTestFlag.ctlLeftSprayRodSwingOutTest:=FALSE;
	ELSE
		ctlTestFlag.ctlLeftSprayRodSwingOutTest:=NOT panelInput.sprayRodOutOrInFlag;	
	END_IF
END_IF
//右喷杆摆出测试,与硅胶面板的喷杆伸缩按钮互锁
rTrigger23(CLK:=dspTestInput.dspRightSprayRodSwingOutTest);
IF rTrigger23.Q THEN
	IF ctlTestFlag.ctlRightSprayRodSwingOutTest THEN 
		ctlTestFlag.ctlRightSprayRodSwingOutTest:=FALSE;
	ELSE
		ctlTestFlag.ctlRightSprayRodSwingOutTest:=NOT panelInput.sprayRodOutOrInFlag;	
	END_IF
END_IF
//左喷杆喷水测试
rTrigger24(CLK:=dspTestInput.dspLeftSprayRodOpenTest);
IF rTrigger24.Q THEN
	ctlTestFlag.ctlLeftSprayRodOpenTest := NOT ctlTestFlag.ctlLeftSprayRodOpenTest;
END_IF
//右喷杆喷水测试
rTrigger25(CLK:= dspTestInput.dspRightSprayRodOpenTest);
IF rTrigger25.Q THEN
	ctlTestFlag.ctlRightSprayRodOpenTest := NOT ctlTestFlag.ctlRightSprayRodOpenTest;
END_IF
//中喷杆喷水测试
rTrigger26(CLK:= dspTestInput.dspCentreSprayRodOpenTest);
IF rTrigger26.Q THEN
	ctlTestFlag.ctlCentreSprayRodOpenTest := NOT ctlTestFlag.ctlCentreSprayRodOpenTest;
END_IF
//辅助球阀打开测试
rTrigger27(CLK:= dspTestInput.dspAuxiliaryValueTest);
IF rTrigger27.Q THEN
	ctlTestFlag.ctlAuxiliaryValueTest := NOT ctlTestFlag.ctlAuxiliaryValueTest;
END_IF
//自洁打开测试
rTrigger28(CLK:= dspTestInput.dspSelfCleanTest);
IF rTrigger28.Q THEN
	ctlTestFlag.ctlSelfCleanTest := NOT ctlTestFlag.ctlSelfCleanTest;
END_IF
//高压水泵啮合测试
rTrigger29(CLK:= dspTestInput.dspWaterPumpConnectTest);
IF (rTrigger29.Q AND (NOT systemStatus.engineWork)) THEN
	ctlTestFlag.ctlWaterPumpConnectTest := NOT ctlTestFlag.ctlWaterPumpConnectTest;
END_IF
ton1(IN:=(ctlTestFlag.ctlWaterPumpConnectTest AND systemStatus.engineWork AND (faultST.frontTankWaterLevelLow OR faultST.backTankWaterLevelLow)),PT:=T#15S);
IF ton1.Q THEN
	ctlTestFlag.ctlWaterPumpConnectTest:= FALSE; //缺水，15后停机
END_IF
//喷雾降尘泵测试
rTrigger30(CLK:= dspTestInput.dspDiaphragmPumpStartTest);
IF rTrigger30.Q THEN
	ctlTestFlag.ctlDiaphragmPumpStartTest := NOT ctlTestFlag.ctlDiaphragmPumpStartTest;
END_IF
ton2(IN:=(ctlTestFlag.ctlDiaphragmPumpStartTest AND faultST.frontTankWaterLevelLow AND faultST.backTankWaterLevelLow),PT:=T#90S);
IF rTrigger30.Q THEN
	ctlTestFlag.ctlDiaphragmPumpStartTest := FALSE; //缺水，90s后停机
END_IF
//左前冲测试
rTrigger31(CLK:=dspTestInput.dspLeftFrontSprinkleTest);
IF rTrigger31.Q THEN
	ctlTestFlag.ctlLeftFrontSprinkleTest:= NOT ctlTestFlag.ctlLeftFrontSprinkleTest;
END_IF
//右前冲测试
rTrigger32(CLK:=dspTestInput.dspRightFrontSprinkleTest);
IF rTrigger32.Q THEN
	ctlTestFlag.ctlRightFrontSprinkleTest:= NOT ctlTestFlag.ctlRightFrontSprinkleTest;
END_IF
//左后洒测试
rTrigger33(CLK:=dspTestInput.dspLeftBackSprinkleTest);
IF rTrigger33.Q THEN
	ctlTestFlag.ctlLeftBackSprinkleTest:= NOT ctlTestFlag.ctlLeftBackSprinkleTest;
END_IF
//右后洒测试
rTrigger34(CLK:=dspTestInput.dspRightBackSprinkleTest);
IF rTrigger34.Q THEN
	ctlTestFlag.ctlRightBackSprinkleTest:= NOT ctlTestFlag.ctlRightBackSprinkleTest;
END_IF

END_PROGRAM

// Device/Application/resetTestST
PROGRAM resetTestST
VAR
END_VAR

ctlTestFlag.ctlAllSweeperRotateTest := FALSE;
ctlTestFlag.ctlAuxiliaryValueTest := FALSE;
ctlTestFlag.ctlCentreSprayRodOpenTest := FALSE;
ctlTestFlag.ctlCLoseBackTankTest := FALSE;
ctlTestFlag.ctlCloseFrontTankTest := FALSE;
ctlTestFlag.ctlConnectWaterValveTest := FALSE;
ctlTestFlag.ctlDiaphragmPumpStartTest := FALSE;
ctlTestFlag.ctlEngineDisconnectTest := FALSE;
ctlTestFlag.ctlLeftSprayRodOpenTest := FALSE;
ctlTestFlag.ctlLeftSprayRodSwingOutTest:= FALSE;
ctlTestFlag.ctlLeftSweeperDownTest := FALSE;
ctlTestFlag.ctlLeftSweeperRotateTest :=FALSE;
ctlTestFlag.ctlLeftSweeperSwingOutTest :=FALSE;
ctlTestFlag.ctlLeftSweeperUpTest := FALSE;
ctlTestFlag.ctlRightSprayRodOpenTest:= FALSE;
ctlTestFlag.ctlRightSprayRodSwingOutTest:=FALSE;
ctlTestFlag.ctlRightSweeperDownTest:=FALSE;
ctlTestFlag.ctlRightSweeperRotateTest:=FALSE;
ctlTestFlag.ctlRightSweeperSwingOutTest:= FALSE;
ctlTestFlag.ctlRightSweeperUpTest := FALSE;
ctlTestFlag.ctlSelfCleanTest := FALSE;
ctlTestFlag.ctlSuctionNozzleDownTest:=FALSE;
ctlTestFlag.ctlSuctionNozzleUpTest:=FALSE;
ctlTestFlag.ctlSweeperSpeedLowTest:=FALSE;
ctlTestFlag.ctlSweeperSpeedMiddleTest:=FALSE;
ctlTestFlag.ctlTankDoorCloseTest:=FALSE;
ctlTestFlag.ctlTankDoorOpenTest:= FALSE;
ctlTestFlag.ctlTankDownTest:= FALSE;
ctlTestFlag.ctlTankUpTest:=FALSE;
ctltEstFlag.ctlWaterPumpConnectTest:=FALSE;

END_PROGRAM

// Device/Application/chooseWorkMode
PROGRAM chooseWorkMode
VAR
	sweepModeCondition:BOOL;//扫路工作模式限定条件
	washSweepModeCondition:BOOL;//洗扫清洗工作模式限定条件
	dspModeInputTemp1:BOOL; //全洗扫模式中间变量
	dspModeInputTemp2:BOOL; //左洗扫模式中间变量
	dspModeInputTemp3:BOOL; //右洗扫模式中间变量
	dspModeInputTemp4:BOOL; //全扫路模式中间变量
	dspModeInputTemp5:BOOL; //左扫路模式中间变量
	dspModeInputTemp6:BOOL; //右扫路模式中间变量
	dspModeInputTemp7:BOOL; //全清洗模式中间变量
	dspModeInputTemp8:BOOL; //左清洗模式中间变量
	dspModeInputTemp9:BOOL; //右清洗模式中间变量
	dspModeInputTemp10:BOOL; //停扫模式中间变量
	
	rTrigger1:R_TRIG;//全洗扫_屏输入触发器
	rTrigger2:R_TRIG;//左洗扫_屏输入触发器
	rTrigger3:R_TRIG;//右洗扫_屏输入触发器
	rTrigger4:R_TRIG;//全扫路_屏输入触发器
	rTrigger5:R_TRIG;//左扫路_屏输入触发器
	rTrigger6:R_TRIG;//右扫路_屏输入触发器
	rTrigger7:R_TRIG;//全清洗_屏输入触发器
	rTrigger8:R_TRIG;//左清洗_屏输入触发器
	rTrigger9:R_TRIG;//右清洗_屏输入触发器
	rTrigger10:R_TRIG;//停扫_屏输入触发器
	rTrigger11:R_TRIG;//污水满停扫触发器
	rTrigger12:R_TRIG;//倒车停扫触发器
	
	fTrigger1:F_TRIG;//高压水泵啮合下降沿触发
	
    ton1:TON;//停扫定时器
	
	tp1:TP;//请关闭测试保持定时器
	tp2:TP;//请先请先打开发动机保持定时器
	tp3:TP;//高压水泵未啮合保持定时器
	tp4:TP;//总水阀未打开保持定时器
	tp5:TP;//吹净球阀未关闭保持定时器
	tp6:TP;//正在倒车中保持定时器
	
	flag:INT:=0;
END_VAR

//扫路工作模式限定条件,发动机工作&&非系统测试状态&&非倒车状态
//sweepModeCondition:= ((NOT systemStatus.systemTest) AND systemStatus.engineWork AND (NOT input24B.stopEngineLamp));
//洗扫工作模式限定条件，发动机工作&&非系统测试状态&&非倒车状态&&高压水泵啮合
washSweepModeCondition:=((NOT systemStatus.systemTest) AND  systemStatus.engineWork AND (NOT input24B.stopEngineLamp) AND systemStatus.waterPumpConnect);
//sweepModeCondition:=TRUE;
//washSweepModeCondition:=TRUE;
//全洗扫模式中间变量
dspModeInputTemp1:= (NOT dspSystemInput.dspLeftWashSweep) AND ( NOT dspSystemInput.dspRightWashSweep) AND (NOT dspSystemInput.dspAllSweep)
AND (NOT dspSystemInput.dspLeftSweep) AND (NOT dspSystemInput.dspRightSweep) AND ( NOT dspSystemInput.dspAllWash)
 AND (NOT dspSystemInput.dspLeftWash) AND (NOT dspSystemInput.dspRightWash) AND (NOT dspSystemInput.dspStopWash);
//左洗扫模式中间变量
dspModeInputTemp2:= (NOT dspSystemInput.dspAllWashSweep) AND ( NOT dspSystemInput.dspRightWashSweep) AND (NOT dspSystemInput.dspAllSweep)
AND (NOT dspSystemInput.dspLeftSweep) AND (NOT dspSystemInput.dspRightSweep) AND ( NOT dspSystemInput.dspAllWash)
 AND (NOT dspSystemInput.dspLeftWash) AND (NOT dspSystemInput.dspRightWash) AND (NOT dspSystemInput.dspStopWash);
 //右洗扫模式中间变量
dspModeInputTemp3:= (NOT dspSystemInput.dspAllWashSweep) AND ( NOT dspSystemInput.dspLeftWashSweep) AND (NOT dspSystemInput.dspAllSweep)
AND (NOT dspSystemInput.dspLeftSweep) AND (NOT dspSystemInput.dspRightSweep) AND ( NOT dspSystemInput.dspAllWash)
 AND (NOT dspSystemInput.dspLeftWash) AND (NOT dspSystemInput.dspRightWash) AND (NOT dspSystemInput.dspStopWash);
 //全扫路模式中间变量
dspModeInputTemp4:= (NOT dspSystemInput.dspAllWashSweep) AND (NOT dspSystemInput.dspLeftWashSweep) AND ( NOT dspSystemInput.dspRightWashSweep) 
AND (NOT dspSystemInput.dspLeftSweep) AND (NOT dspSystemInput.dspRightSweep) AND ( NOT dspSystemInput.dspAllWash)
 AND (NOT dspSystemInput.dspLeftWash) AND (NOT dspSystemInput.dspRightWash) AND (NOT dspSystemInput.dspStopWash);
 //左扫路模式中间变量
dspModeInputTemp5:= (NOT dspSystemInput.dspAllWashSweep) AND (NOT dspSystemInput.dspLeftWashSweep) AND ( NOT dspSystemInput.dspRightWashSweep) 
AND (NOT dspSystemInput.dspAllSweep) AND (NOT dspSystemInput.dspRightSweep) AND ( NOT dspSystemInput.dspAllWash)
 AND (NOT dspSystemInput.dspLeftWash) AND (NOT dspSystemInput.dspRightWash) AND (NOT dspSystemInput.dspStopWash);
 //右扫路模式中间变量
dspModeInputTemp6:= (NOT dspSystemInput.dspAllWashSweep) AND (NOT dspSystemInput.dspLeftWashSweep) AND ( NOT dspSystemInput.dspRightWashSweep) 
AND (NOT dspSystemInput.dspAllSweep) AND (NOT dspSystemInput.dspLeftSweep) AND ( NOT dspSystemInput.dspAllWash)
 AND (NOT dspSystemInput.dspLeftWash) AND (NOT dspSystemInput.dspRightWash) AND (NOT dspSystemInput.dspStopWash);
 //全清洗模式中间变量
dspModeInputTemp7:= (NOT dspSystemInput.dspAllWashSweep) AND (NOT dspSystemInput.dspLeftWashSweep) AND ( NOT dspSystemInput.dspRightWashSweep) 
AND ( NOT dspSystemInput.dspAllSweep) AND (NOT dspSystemInput.dspLeftSweep) AND (NOT dspSystemInput.dspRightSweep) 
 AND (NOT dspSystemInput.dspLeftWash) AND (NOT dspSystemInput.dspRightWash) AND (NOT dspSystemInput.dspStopWash);
 //左清洗模式中间变量
dspModeInputTemp8:= (NOT dspSystemInput.dspAllWashSweep) AND (NOT dspSystemInput.dspLeftWashSweep) AND ( NOT dspSystemInput.dspRightWashSweep) 
AND ( NOT dspSystemInput.dspAllSweep) AND (NOT dspSystemInput.dspLeftSweep) AND (NOT dspSystemInput.dspRightSweep)
 AND (NOT dspSystemInput.dspAllWash) AND (NOT dspSystemInput.dspRightWash) AND (NOT dspSystemInput.dspStopWash);
 //右清洗模式中间变量
dspModeInputTemp9:= (NOT dspSystemInput.dspAllWashSweep) AND (NOT dspSystemInput.dspLeftWashSweep) AND ( NOT dspSystemInput.dspRightWashSweep) 
AND ( NOT dspSystemInput.dspAllSweep) AND (NOT dspSystemInput.dspLeftSweep) AND (NOT dspSystemInput.dspRightSweep)
 AND (NOT dspSystemInput.dspAllWash) AND (NOT dspSystemInput.dspLeftWash) AND (NOT dspSystemInput.dspStopWash);
//全洗扫工作模式
rTrigger1(CLK:=dspSystemInput.dspAllWashSweep);
IF rTrigger1.Q THEN
	flag:=4353;
END_IF
IF (rTrigger1.Q AND dspModeInputTemp1 AND washSweepModeCondition ) THEN
	systemStatus.AllWashSweep:=(NOT systemStatus.AllWashSweep);
	//如果全洗扫为真状态，其他模式复位，如果全洗扫为假，停扫模式置位
	IF  systemStatus.AllWashSweep THEN 
		systemStatus.LeftWashSweep:=FALSE;
		systemStatus.RightWashSweep:= FALSE;
		systemStatus.AllSweep:=FALSE;
		systemStatus.LeftSweep:=FALSE;
		systemStatus.RightSweep:=FALSE;
		systemStatus.AllWash:=FALSE;
		systemStatus.LeftWash:=FALSE;
		systemStatus.RightWash:=FALSE;
		systemStatus.StopWash:=FALSE;
	ELSE
		systemStatus.StopWash:=TRUE;
	END_IF
END_IF

//左洗扫工作模式
rTrigger2(CLK:=dspSystemInput.dspLeftWashSweep);
IF (rTrigger2.Q AND dspModeInputTemp2  AND washSweepModeCondition ) THEN
	systemStatus.LeftWashSweep:=(NOT systemStatus.LeftWashSweep);
	//如果左洗扫为真状态，其他模式复位，如果左洗扫为假，停扫模式置位
	IF systemStatus.LeftWashSweep THEN 
		systemStatus.AllWashSweep:=FALSE;
		systemStatus.RightWashSweep:= FALSE;
		systemStatus.AllSweep:=FALSE;
		systemStatus.LeftSweep:=FALSE;
		systemStatus.RightSweep:=FALSE;
		systemStatus.AllWash:=FALSE;
		systemStatus.LeftWash:=FALSE;
		systemStatus.RightWash:=FALSE;
		systemStatus.StopWash:=FALSE;
	ELSE
		systemStatus.StopWash:=TRUE;
	END_IF
END_IF
//右洗扫工作模式
rTrigger3(CLK:=dspSystemInput.dspRightWashSweep);
IF (rTrigger3.Q AND dspModeInputTemp3  AND washSweepModeCondition ) THEN
	systemStatus.RightWashSweep:=(NOT systemStatus.RightWashSweep);
	//如果右洗扫为真状态，其他模式复位，如果右洗扫为假，停扫模式置位
	IF systemStatus.RightWashSweep THEN 
		systemStatus.AllWashSweep:=FALSE;
		systemStatus.LeftWashSweep:= FALSE;
		systemStatus.AllSweep:=FALSE;
		systemStatus.LeftSweep:=FALSE;
		systemStatus.RightSweep:=FALSE;
		systemStatus.AllWash:=FALSE;
		systemStatus.LeftWash:=FALSE;
		systemStatus.RightWash:=FALSE;
		systemStatus.StopWash:=FALSE;
	ELSE
		systemStatus.StopWash:=TRUE;
	END_IF
END_IF
//全扫路工作模式
rTrigger4(CLK:=dspSystemInput.dspAllSweep);
IF (rTrigger4.Q AND dspModeInputTemp4 AND sweepModeCondition ) THEN
	systemStatus.AllSweep:=(NOT systemStatus.AllSweep);
	//如果全扫路为真状态，其他模式复位，如果全扫路为假，停扫模式置位
	IF  systemStatus.AllSweep THEN 
		systemStatus.AllWashSweep:=FALSE;
		systemStatus.LeftWashSweep:=FALSE;
		systemStatus.RightWashSweep:= FALSE;
		systemStatus.LeftSweep:=FALSE;
		systemStatus.RightSweep:=FALSE;
		systemStatus.AllWash:=FALSE;
		systemStatus.LeftWash:=FALSE;
		systemStatus.RightWash:=FALSE;
		systemStatus.StopWash:=FALSE;
	ELSE
		systemStatus.StopWash:=TRUE;
	END_IF
END_IF
//左扫路工作模式
rTrigger5(CLK:=dspSystemInput.dspLeftSweep);
IF (rTrigger5.Q AND dspModeInputTemp5 AND sweepModeCondition ) THEN
	systemStatus.LeftSweep:=(NOT systemStatus.LeftSweep);
	//如果左扫路为真状态，其他模式复位，如果左扫路为假，停扫模式置位
	IF  systemStatus.LeftSweep THEN 
		systemStatus.AllWashSweep:=FALSE;
		systemStatus.LeftWashSweep:=FALSE;
		systemStatus.RightWashSweep:= FALSE;
		systemStatus.AllSweep:=FALSE;
		systemStatus.RightSweep:=FALSE;
		systemStatus.AllWash:=FALSE;
		systemStatus.LeftWash:=FALSE;
		systemStatus.RightWash:=FALSE;
		systemStatus.StopWash:=FALSE;
	ELSE
		systemStatus.StopWash:=TRUE;
	END_IF
END_IF
//右扫路工作模式
rTrigger6(CLK:=dspSystemInput.dspRightSweep);
IF (rTrigger6.Q AND dspModeInputTemp6 AND sweepModeCondition ) THEN
	systemStatus.RightSweep:=(NOT systemStatus.RightSweep);
	//如果全洗扫为真状态，其他模式复位，如果全洗扫为假，停扫模式置位
	IF  systemStatus.RightSweep THEN 
		systemStatus.AllWashSweep:=FALSE;
		systemStatus.LeftWashSweep:=FALSE;
		systemStatus.RightWashSweep:= FALSE;
		systemStatus.AllSweep:=FALSE;
		systemStatus.LeftSweep:=FALSE;
		systemStatus.AllWash:=FALSE;
		systemStatus.LeftWash:=FALSE;
		systemStatus.RightWash:=FALSE;
		systemStatus.StopWash:=FALSE;
	ELSE
		systemStatus.StopWash:=TRUE;
	END_IF
END_IF
//全清洗工作模式
rTrigger7(CLK:=dspSystemInput.dspAllWash);
IF (rTrigger7.Q AND dspModeInputTemp7 AND washSweepModeCondition ) THEN
	systemStatus.AllWash:=(NOT systemStatus.AllWash);
	//如果全清洗为真状态，其他模式复位，如果全清洗为假，停扫模式置位
	IF  systemStatus.AllWash THEN 
		systemStatus.AllWashSweep:=FALSE;
		systemStatus.LeftWashSweep:=FALSE;
		systemStatus.RightWashSweep:= FALSE;
		systemStatus.AllSweep:=FALSE;
		systemStatus.LeftSweep:=FALSE;
		systemStatus.RightSweep:=FALSE;
		systemStatus.LeftWash:=FALSE;
		systemStatus.RightWash:=FALSE;
		systemStatus.StopWash:=FALSE;
	ELSE
		systemStatus.StopWash:=TRUE;
	END_IF
END_IF
//左清洗工作模式
rTrigger8(CLK:=dspSystemInput.dspLeftWash);
IF (rTrigger8.Q AND dspModeInputTemp8 AND washSweepModeCondition ) THEN
	systemStatus.LeftWash:=(NOT systemStatus.LeftWash);
	//如果左清洗为真状态，其他模式复位，如果左清洗为假，停扫模式置位
	IF  systemStatus.LeftWash THEN 
		systemStatus.AllWashSweep:=FALSE;
		systemStatus.LeftWashSweep:=FALSE;
		systemStatus.RightWashSweep:= FALSE;
		systemStatus.AllSweep:=FALSE;
		systemStatus.LeftSweep:=FALSE;
		systemStatus.RightSweep:=FALSE;
		systemStatus.AllWash:=FALSE;
		systemStatus.RightWash:=FALSE;
		systemStatus.StopWash:=FALSE;
	ELSE
		systemStatus.StopWash:=TRUE;
	END_IF
END_IF
//右清洗工作模式
rTrigger9(CLK:=dspSystemInput.dspRightWash);
IF (rTrigger9.Q AND dspModeInputTemp9 AND washSweepModeCondition ) THEN
	systemStatus.RightWash:=(NOT systemStatus.RightWash);
	//如果右清洗为真状态，其他模式复位，如果右清洗为假，停扫模式置位
	IF  systemStatus.RightWash THEN 
		systemStatus.AllWashSweep:=FALSE;
		systemStatus.LeftWashSweep:=FALSE;
		systemStatus.RightWashSweep:= FALSE;
		systemStatus.AllSweep:=FALSE;
		systemStatus.LeftSweep:=FALSE;
		systemStatus.RightSweep:=FALSE;
		systemStatus.AllWash:=FALSE;
		systemStatus.LeftWash:=FALSE;
		systemStatus.StopWash:=FALSE;
	ELSE
		systemStatus.StopWash:=TRUE;
	END_IF
END_IF

//系统工作状态,处于全洗扫、左洗扫、右洗扫、全扫路、左扫路、右扫路、全清洗、左清洗、右清洗一种中
systemStatus.systemWork:= systemStatus.AllWashSweep OR systemStatus.LeftWashSweep OR systemStatus.RightWashSweep
OR systemStatus.AllSweep OR systemStatus.LeftSweep OR systemStatus.RightSweep 
OR systemStatus.AllWash OR systemStatus.LeftWash OR systemStatus.RightWash;

//按键、倒车、污水满触发停扫
rTrigger10(CLK:=dspSystemInput.dspStopWash); //按键触发
rTrigger11(CLK:=faultST.waterFullStop); //污水满触发
rTrigger12(CLK:=faultSt.reverseCarStop);//倒车触发
IF (rTrigger10.Q OR rTrigger11.Q OR rTrigger12.Q) THEN
	systemStatus.StopWash:=TRUE;
	systemStatus.AllWashSweep:=FALSE;
	systemStatus.LeftWashSweep:=FALSE;
	systemStatus.RightWashSweep:= FALSE;
	systemStatus.AllSweep:=FALSE;
	systemStatus.LeftSweep:=FALSE;
	systemStatus.RightSweep:=FALSE;
	systemStatus.AllWash:=FALSE;
	systemStatus.LeftWash:=FALSE;
	systemStatus.RightWash:=FALSE;
END_IF
//停扫状态持续14S
ton1(IN:=systemStatus.StopWash,PT:=T#14S);
IF ton1.Q THEN
	systemStatus.StopWash:=false;
END_IF

//提示信息
//请关闭测试
tp1(IN:=(rTrigger1.Q AND (NOT systemStatus.AllWashSweep) AND systemStatus.systemTest) OR
                   (rTrigger2.Q AND (NOT systemStatus.LeftWashSweep) AND systemStatus.systemTest) OR
				   (rTrigger3.Q AND (NOT systemStatus.RightWashSweep) AND systemStatus.systemTest) OR
				   (rTrigger4.Q AND (NOT systemStatus.AllSweep) AND systemStatus.systemTest) OR
				   (rTrigger5.Q AND (NOT systemStatus.LeftSweep) AND systemStatus.systemTest) OR
				   (rTrigger6.Q AND (NOT systemStatus.RightSweep) AND systemStatus.systemTest) OR
				   (rTrigger7.Q AND (NOT systemStatus.AllWash) AND systemStatus.systemTest) OR
				   (rTrigger8.Q AND (NOT systemStatus.LeftWash) AND systemStatus.systemTest) OR
				   (rTrigger9.Q AND (NOT systemStatus.RightWash) AND systemStatus.systemTest),PT:=T#1S);
tipsST.closeTest:= tp1.Q;
//请打开发动机
tp2(IN:=(rTrigger1.Q AND (NOT systemStatus.AllWashSweep) AND systemStatus.engineWork) OR
                   (rTrigger2.Q AND (NOT systemStatus.LeftWashSweep) AND NOT systemStatus.engineWork) OR
				   (rTrigger3.Q AND (NOT systemStatus.RightWashSweep) AND NOT systemStatus.engineWork) OR
				   (rTrigger4.Q AND (NOT systemStatus.AllSweep) AND NOT  systemStatus.engineWork) OR
				   (rTrigger5.Q AND (NOT systemStatus.LeftSweep) AND NOT systemStatus.engineWork) OR
				   (rTrigger6.Q AND (NOT systemStatus.RightSweep) AND NOT  systemStatus.engineWork) OR
				   (rTrigger7.Q AND (NOT systemStatus.AllWash) AND NOT systemStatus.engineWork) OR
				   (rTrigger8.Q AND (NOT systemStatus.LeftWash) AND NOT systemStatus.engineWork) OR
				   (rTrigger9.Q AND (NOT systemStatus.RightWash) AND NOT systemStatus.engineWork),PT:=T#1S);
tipsST.startEngineFirst:=tp2.Q;
//高压水泵未啮合
fTrigger1(CLK:= systemStatus.waterPumpConnect);
tp3(IN:=(rTrigger1.Q AND (NOT systemStatus.AllWashSweep) AND (NOT systemStatus.waterPumpConnect)) OR  //按全洗扫按钮，高压水泵未啮合，即提示
                   (rTrigger2.Q AND (NOT systemStatus.LeftWashSweep) AND (NOT systemStatus.waterPumpConnect)) OR //按左洗扫按钮，高压水泵未啮合，即提示
				   (rTrigger3.Q AND (NOT systemStatus.RightWashSweep) AND (NOT systemStatus.waterPumpConnect)) OR //按右洗扫按钮，高压水泵未啮合，即提示
				   (rTrigger7.Q AND (NOT systemStatus.allWash) AND (NOT systemStatus.waterPumpConnect)) OR //按全清洗按钮，高压水泵未啮合，即提示
				   (rTrigger8.Q AND (NOT systemStatus.leftWash) AND (NOT systemStatus.waterPumpConnect)) OR //按左清洗按钮，高压水泵未啮合，即提示
				   (rTrigger9.Q AND (NOT systemStatus.rightWash) AND (NOT systemStatus.waterPumpConnect)) OR //按右清洗按钮，高压水泵未啮合，即提示
				   (fTrigger1.Q  AND (NOT systemStatus.allSweep) AND (NOT systemStatus.leftSweep) AND (NOT systemStatus.leftSweep)) ,PT:=T#2S) ;//在非扫路模式下，高压水泵啮合后然后分离属于非正常分离，即提示
tipsST.highPressurePumpDisconnect1:=tp3.Q;//高压水泵未啮合判断
//总水阀未打开
//tp4(IN:= tipsST.highPressurePumpDisconnect1 AND (NOT input40A.mainWateraValve),PT:=T#1S);
//tipsST.mainWateraValveNotOpen1:= tp4.Q;  //总水阀未打开判断
//吹净球阀未关闭
//tp5(IN:= tipsST.highPressurePumpDisconnect1 AND (NOT input40A.mainWateraValve),PT:=T#1S);     
//tipsST.cleanValveNotClose1:= tp5.Q;       //吹净球阀未关闭判断   
//正在倒车中
tipsST.reverseCar:=input24B.reverseCar;
//备用动力打开
tipsST.backupMotorOpen:= systemStatus.backupMotorOpen;

END_PROGRAM

